(* CODESYS project CodesysTest
   Author: Ben Hess
   Company: Sharp Packaging
   CompiledLibraryCompatibilityVersion: CODESYS V3.5 SP16
   Version: 0.9.20.33
   VersionPostfix: -alpha/master

Project tree, tasks and I/O mapping:
  ElectricMachine : CODESYS Control RTE V3 x64, 3S - Smart Software Solutions GmbH, version 3.5.17.0
    application Application
    Customer_LAN_Adapter : Ethernet, 3S - Smart Software Solutions GmbH, version 3.5.16.0
        settings: IPAddress = [172,20,10,206]; SubnetMask = [255,255,255,0]; GatewayAddress = [172,20,10,1]; MACAddress = [16#D8,16#5E,16#D3,16#E1,16#78,16#F8]; NetworkInterfaceName = 'Customer LAN'; NetworkInterfaceName = "Customer LAN"; SaveCommunicationSettings = FALSE
      ModbusTCP_Slave_Device : ModbusTCP Slave Device, 3S - Smart Software Solutions GmbH, version 4.2.0.0
          input  Application.RemoteComms.modbusInputsToBagger.fillerTrigger : BOOL  // Holding Registers.Holding Registers.Bit0
          input  Application.RemoteComms.modbusInputsToBagger.baggerInhibit : BOOL  // Holding Registers.Holding Registers.Bit1
          input  Application.RemoteComms.modbusInputsToBagger.collisionDetection : BOOL  // Holding Registers.Holding Registers.Bit2
          input  Application.RemoteComms.modbusInputsToBagger.fillerOK : BOOL  // Holding Registers.Holding Registers.Bit3
          input  Application.RemoteComms.modbusInputsToBagger.reverseConveyor : BOOL  // Holding Registers.Holding Registers.Bit4
          input  Application.RemoteComms.modbusInputsToBagger.bagGrabbed : BOOL  // Holding Registers.Holding Registers.Bit5
          input  Application.RemoteComms.modbusInputsToBagger.heartbeat : BOOL  // Holding Registers.Holding Registers.Bit6
          output Application.RemoteComms.modbusOutputsFromBagger.baggerOK : BOOL  // Input Registers.Input Registers.Bit0
          output Application.RemoteComms.modbusOutputsFromBagger.readyForFiller : BOOL  // Input Registers.Input Registers.Bit1
          output Application.RemoteComms.modbusOutputsFromBagger.printerDataReady : BOOL  // Input Registers.Input Registers.Bit2
          output Application.RemoteComms.modbusOutputsFromBagger.waitingForPrinter : BOOL  // Input Registers.Input Registers.Bit3
          output Application.RemoteComms.modbusOutputsFromBagger.cycleComplete : BOOL  // Input Registers.Input Registers.Bit4
          output Application.RemoteComms.modbusOutputsFromBagger.bagMade : BOOL  // Input Registers.Input Registers.Bit5
          output Application.RemoteComms.modbusOutputsFromBagger.bagMadePlusLabelRequired : BOOL  // Input Registers.Input Registers.Bit6
          output Application.RemoteComms.modbusOutputsFromBagger.bagsLow : BOOL  // Input Registers.Input Registers.Bit7
          output Application.RemoteComms.modbusOutputsFromBagger.readyForGrab : BOOL  // Input Registers.Input Registers.Bit8
          output Application.RemoteComms.modbusOutputsFromBagger.runExternalExitConveyor : BOOL  // Input Registers.Input Registers.Bit9
          output Application.RemoteComms.modbusOutputsFromBagger.heartbeatResponse : BOOL  // Input Registers.Input Registers.Bit10
          unmapped channels: Holding Registers, Input Registers
    IO_Connection_Adapter : Ethernet, 3S - Smart Software Solutions GmbH, version 3.5.16.0
        settings: IPAddress = [192,168,10,21]; SubnetMask = [255,255,255,0]; GatewayAddress = [0,0,0,0]; MACAddress = [16#00,16#00,16#00,16#00,16#00,16#00]; NetworkInterfaceName = 'IO Connection'; NetworkInterfaceName = "IO Connection"; SaveCommunicationSettings = FALSE
      EtherNet_IP_Scanner : EtherNet/IP Scanner, 3S - Smart Software Solutions GmbH, order no. 1, version 3.5.16.10
    Machine_LAN_Adapter : Ethernet, 3S - Smart Software Solutions GmbH, version 3.5.16.0
        settings: IPAddress = [192,168,10,20]; SubnetMask = [255,255,255,0]; GatewayAddress = [192,168,10,254]; MACAddress = [16#00,16#00,16#00,16#00,16#00,16#00]; NetworkInterfaceName = 'Machine LAN'; NetworkInterfaceName = "Machine LAN"; SaveCommunicationSettings = FALSE
  Pro18_1174_CodesysDriver : CODESYS Control RTE V3 x64, 3S - Smart Software Solutions GmbH, version 3.5.17.0
    application Application
    Dual_LAN_Card : Ethernet, 3S - Smart Software Solutions GmbH, version 3.5.16.0
        settings: IPAddress = [192,168,10,21]; SubnetMask = [255,255,255,0]; GatewayAddress = [0,0,0,0]; MACAddress = [16#00,16#00,16#00,16#00,16#00,16#00]; NetworkInterfaceName = 'IO Connection'; NetworkInterfaceName = "IO Connection"; SaveCommunicationSettings = FALSE
      EtherNet_IP_Scanner : EtherNet/IP Scanner, 3S - Smart Software Solutions GmbH, order no. 1, version 3.5.16.10
    Ethernet : Ethernet, 3S - Smart Software Solutions GmbH, version 3.5.13.0
        settings: IPAddress = [192,168,10,20]; SubnetMask = [255,255,255,0]; GatewayAddress = [192,168,10,254]; NetworkInterfaceName = 'Machine LAN:2'; NetworkInterfaceName = "Machine LAN:2"; SaveCommunicationSettings = FALSE
      ModbusTCP_Slave_Device : ModbusTCP Slave Device, 3S - Smart Software Solutions GmbH, version 4.2.0.0 (disabled)
          input  Application.RemoteComms.modbusInputsToBagger.fillerTrigger : BOOL  // Holding Registers.Holding Registers.Bit0
          input  Application.RemoteComms.modbusInputsToBagger.baggerInhibit : BOOL  // Holding Registers.Holding Registers.Bit1
          input  Application.RemoteComms.modbusInputsToBagger.collisionDetection : BOOL  // Holding Registers.Holding Registers.Bit2
          input  Application.RemoteComms.modbusInputsToBagger.fillerOK : BOOL  // Holding Registers.Holding Registers.Bit3
          input  Application.RemoteComms.modbusInputsToBagger.reverseConveyor : BOOL  // Holding Registers.Holding Registers.Bit4
          input  Application.RemoteComms.modbusInputsToBagger.bagGrabbed : BOOL  // Holding Registers.Holding Registers.Bit5
          input  Application.RemoteComms.modbusInputsToBagger.heartbeat : BOOL  // Holding Registers.Holding Registers.Bit6
          output Application.RemoteComms.modbusOutputsFromBagger.baggerOK : BOOL  // Input Registers.Input Registers.Bit0
          output Application.RemoteComms.modbusOutputsFromBagger.readyForFiller : BOOL  // Input Registers.Input Registers.Bit1
          output Application.RemoteComms.modbusOutputsFromBagger.printerDataReady : BOOL  // Input Registers.Input Registers.Bit2
          output Application.RemoteComms.modbusOutputsFromBagger.waitingForPrinter : BOOL  // Input Registers.Input Registers.Bit3
          output Application.RemoteComms.modbusOutputsFromBagger.cycleComplete : BOOL  // Input Registers.Input Registers.Bit4
          output Application.RemoteComms.modbusOutputsFromBagger.bagMade : BOOL  // Input Registers.Input Registers.Bit5
          output Application.RemoteComms.modbusOutputsFromBagger.bagMadePlusLabelRequired : BOOL  // Input Registers.Input Registers.Bit6
          output Application.RemoteComms.modbusOutputsFromBagger.bagsLow : BOOL  // Input Registers.Input Registers.Bit7
          output Application.RemoteComms.modbusOutputsFromBagger.readyForGrab : BOOL  // Input Registers.Input Registers.Bit8
          output Application.RemoteComms.modbusOutputsFromBagger.runExternalExitConveyor : BOOL  // Input Registers.Input Registers.Bit9
          output Application.RemoteComms.modbusOutputsFromBagger.heartbeatResponse : BOOL  // Input Registers.Input Registers.Bit10
          unmapped channels: Holding Registers, Input Registers
  Pro18_1174_HilscherCard : Advantech Control x86 RTE V3, Advantech Co., Ltd., order no. 
      , version 3.5.13.0
    application Application
    CIFX_EIP : CIFX-EIP, 3S - Smart Software Solutions GmbH, order no. 1, version 3.5.12.0
        settings: IPAddress = [16#C0,16#A8,16#0A,16#15]; SubnetMask = [16#FF,16#FF,16#FF,16#00]; GatewayAddress = [16#00,16#00,16#00,16#00]; ConfigVersion = 50660608
      Bag_Delivery_EIP_Motor : TSM34IP, Applied Motion Products, Inc, order no. TSM34IP, version Major Revision=16#3, Minor Revision = 16#3
          settings: INITIALIZED = TRUE; IP address of Target = [16#C0,16#A8,16#0A,16#37]; Keying.Check Vendor Code = FALSE; Keying.Check Product Code = FALSE; Keying.Check Major Revision = FALSE; Keying.Check Minor Revision = FALSE; RequiredConfigVersion = 50660864; Number of Connections = 1; Connection Settings.Requested packet intervall = 10000 µs; Connection Settings.OT Connection Parameters = 18502; Connection Settings.TO Connection Parameters = 18490; Connection Settings.Connection Flags = 1056; Connection Settings.Connection Path Size = 8; Connection Settings.Large OT Connection Parameters = 1207959622; Connection Settings.Large TO Connection Parameters = 1207959610; Heartbeat Multiplier = 1; Status Code.ReadOnly = False; Status Code.BitSize = 32; Status Code.DataSize = 4; Alarm Code.ReadOnly = False; Alarm Code.BitSize = 32; Alarm Code.DataSize = 4; Supply Voltage.ReadOnly = False; Supply Voltage.BitSize = 32; Supply Voltage.DataSize = 4; Actual Current.ReadOnly = False; Actual Current.BitSize = 32; Actual Current.DataSize = 4; Drive Temperature.ReadOnly = False; Drive Temperature.BitSize = 32; Drive Temperature.DataSize = 4; Encoder Position.ReadOnly = False; Encoder Position.BitSize = 32; Encoder Position.DataSize = 4; Absolute Position.ReadOnly = False; Absolute Position.BitSize = 32; Absolute Position.DataSize = 4; Position Error.ReadOnly = False; Position Error.BitSize = 32; Position Error.DataSize = 4;
            Actual Velocity.ReadOnly = False; Actual Velocity.BitSize = 32; Actual Velocity.DataSize = 4; Input Status (extended).ReadOnly = False; Input Status (extended).BitSize = 32; Input Status (extended).DataSize = 4; Input Status (main).ReadOnly = False; Input Status (main).BitSize = 32; Input Status (main).DataSize = 4; Output Status.ReadOnly = False; Output Status.BitSize = 32; Output Status.DataSize = 4; Analog Input 1.ReadOnly = False; Analog Input 1.BitSize = 32; Analog Input 1.DataSize = 4; Analog Input 2.ReadOnly = False; Analog Input 2.BitSize = 32; Analog Input 2.DataSize = 4; Command Word.ReadOnly = False; Command Word.BitSize = 32; Command Word.DataSize = 4; Jog Speed.ReadOnly = False; Jog Speed.BitSize = 32; Jog Speed.DataSize = 4; Jog Accel.ReadOnly = False; Jog Accel.BitSize = 32; Jog Accel.DataSize = 4; Jog Decel.ReadOnly = False; Jog Decel.BitSize = 32; Jog Decel.DataSize = 4; Point-to-Point Velocity.ReadOnly = False; Point-to-Point Velocity.BitSize = 32; Point-to-Point Velocity.DataSize = 4; Point-to-Point Acceleration.ReadOnly = False; Point-to-Point Acceleration.BitSize = 32; Point-to-Point Acceleration.DataSize = 4; Point-to-Point Deceleration.ReadOnly = False; Point-to-Point Deceleration.BitSize = 32; Point-to-Point Deceleration.DataSize = 4; Point-to-Point Distance.ReadOnly = False;
            Point-to-Point Distance.BitSize = 32; Point-to-Point Distance.DataSize = 4; Current Command.ReadOnly = False; Current Command.BitSize = 32; Current Command.DataSize = 4; SCL Command Letters.ReadOnly = False; SCL Command Letters.BitSize = 32; SCL Command Letters.DataSize = 4; Data/SCL Register 1.ReadOnly = False; Data/SCL Register 1.BitSize = 32; Data/SCL Register 1.DataSize = 4; Data/SCL Register 2.ReadOnly = False; Data/SCL Register 2.BitSize = 32; Data/SCL Register 2.DataSize = 4; Reserved 1.ReadOnly = False; Reserved 1.BitSize = 32; Reserved 1.DataSize = 4; Reserved 2.ReadOnly = False; Reserved 2.BitSize = 32; Reserved 2.DataSize = 4; Reserved 3.ReadOnly = False; Reserved 3.BitSize = 32; Reserved 3.DataSize = 4; Reserved 4.ReadOnly = False; Reserved 4.BitSize = 32; Reserved 4.DataSize = 4; Status Code.Name = 'Status Code'; Status Code.HelpString = ''; Status Code.ReadOnly = False; Status Code.BitSize = 32; Status Code.DataSize = 4; Status Code.DataType = 'DINT'; Alarm Code.Name = 'Alarm Code'; Alarm Code.HelpString = ''; Alarm Code.ReadOnly = False; Alarm Code.BitSize = 32; Alarm Code.DataSize = 4; Alarm Code.DataType = 'DINT'; Supply Voltage.Name = 'Supply Voltage'; Supply Voltage.HelpString = '';
            Supply Voltage.ReadOnly = False; Supply Voltage.BitSize = 32; Supply Voltage.DataSize = 4; Supply Voltage.DataType = 'DINT'; Actual Current.Name = 'Actual Current'; Actual Current.HelpString = ''; Actual Current.ReadOnly = False; Actual Current.BitSize = 32; Actual Current.DataSize = 4; Actual Current.DataType = 'DINT'; Drive Temperature.Name = 'Drive Temperature'; Drive Temperature.HelpString = ''; Drive Temperature.ReadOnly = False; Drive Temperature.BitSize = 32; Drive Temperature.DataSize = 4; Drive Temperature.DataType = 'DINT'; Encoder Position.Name = 'Encoder Position'; Encoder Position.HelpString = ''; Encoder Position.ReadOnly = False; Encoder Position.BitSize = 32; Encoder Position.DataSize = 4; Encoder Position.DataType = 'DINT'; Absolute Position.Name = 'Absolute Position'; Absolute Position.HelpString = ''; Absolute Position.ReadOnly = False; Absolute Position.BitSize = 32; Absolute Position.DataSize = 4; Absolute Position.DataType = 'DINT'; Position Error.Name = 'Position Error'; Position Error.HelpString = ''; Position Error.ReadOnly = False; Position Error.BitSize = 32; Position Error.DataSize = 4; Position Error.DataType = 'DINT'; Actual Velocity.Name = 'Actual Velocity'; Actual Velocity.HelpString = ''; Actual Velocity.ReadOnly = False; Actual Velocity.BitSize = 32; Actual Velocity.DataSize = 4; Actual Velocity.DataType = 'DINT';
            Input Status (extended).Name = 'Input Status (extended)'; Input Status (extended).HelpString = ''; Input Status (extended).ReadOnly = False; Input Status (extended).BitSize = 32; Input Status (extended).DataSize = 4; Input Status (extended).DataType = 'DINT'; Input Status (main).Name = 'Input Status (main)'; Input Status (main).HelpString = ''; Input Status (main).ReadOnly = False; Input Status (main).BitSize = 32; Input Status (main).DataSize = 4; Input Status (main).DataType = 'DINT'; Output Status.Name = 'Output Status'; Output Status.HelpString = ''; Output Status.ReadOnly = False; Output Status.BitSize = 32; Output Status.DataSize = 4; Output Status.DataType = 'DINT'; Analog Input 1.Name = 'Analog Input 1'; Analog Input 1.HelpString = ''; Analog Input 1.ReadOnly = False; Analog Input 1.BitSize = 32; Analog Input 1.DataSize = 4; Analog Input 1.DataType = 'DINT'; Analog Input 2.Name = 'Analog Input 2'; Analog Input 2.HelpString = ''; Analog Input 2.ReadOnly = False; Analog Input 2.BitSize = 32; Analog Input 2.DataSize = 4; Analog Input 2.DataType = 'DINT'; Command Word.Name = 'Command Word'; Command Word.HelpString = ''; Command Word.ReadOnly = False; Command Word.BitSize = 32; Command Word.DataSize = 4; Command Word.DataType = 'DINT'; Jog Speed.Name = 'Jog Speed'; Jog Speed.HelpString = ''; Jog Speed.ReadOnly = False; Jog Speed.BitSize = 32;
            Jog Speed.DataSize = 4; Jog Speed.DataType = 'DINT'; Jog Accel.Name = 'Jog Accel'; Jog Accel.HelpString = ''; Jog Accel.ReadOnly = False; Jog Accel.BitSize = 32; Jog Accel.DataSize = 4; Jog Accel.DataType = 'DINT'; Jog Decel.Name = 'Jog Decel'; Jog Decel.HelpString = ''; Jog Decel.ReadOnly = False; Jog Decel.BitSize = 32; Jog Decel.DataSize = 4; Jog Decel.DataType = 'DINT'; Point-to-Point Velocity.Name = 'Point-to-Point Velocity'; Point-to-Point Velocity.HelpString = ''; Point-to-Point Velocity.ReadOnly = False; Point-to-Point Velocity.BitSize = 32; Point-to-Point Velocity.DataSize = 4; Point-to-Point Velocity.DataType = 'DINT'; Point-to-Point Acceleration.Name = 'Point-to-Point Acceleration'; Point-to-Point Acceleration.HelpString = ''; Point-to-Point Acceleration.ReadOnly = False; Point-to-Point Acceleration.BitSize = 32; Point-to-Point Acceleration.DataSize = 4; Point-to-Point Acceleration.DataType = 'DINT'; Point-to-Point Deceleration.Name = 'Point-to-Point Deceleration'; Point-to-Point Deceleration.HelpString = ''; Point-to-Point Deceleration.ReadOnly = False; Point-to-Point Deceleration.BitSize = 32; Point-to-Point Deceleration.DataSize = 4; Point-to-Point Deceleration.DataType = 'DINT'; Point-to-Point Distance.Name = 'Point-to-Point Distance'; Point-to-Point Distance.HelpString = ''; Point-to-Point Distance.ReadOnly = False; Point-to-Point Distance.BitSize = 32; Point-to-Point Distance.DataSize = 4; Point-to-Point Distance.DataType = 'DINT'; Current Command.Name = 'Current Command'; Current Command.HelpString = '';
            Current Command.ReadOnly = False; Current Command.BitSize = 32; Current Command.DataSize = 4; Current Command.DataType = 'DINT'; SCL Command Letters.Name = 'SCL Command Letters'; SCL Command Letters.HelpString = ''; SCL Command Letters.ReadOnly = False; SCL Command Letters.BitSize = 32; SCL Command Letters.DataSize = 4; SCL Command Letters.DataType = 'DINT'; Data/SCL Register 1.Name = 'Data/SCL Register 1'; Data/SCL Register 1.HelpString = ''; Data/SCL Register 1.ReadOnly = False; Data/SCL Register 1.BitSize = 32; Data/SCL Register 1.DataSize = 4; Data/SCL Register 1.DataType = 'DINT'; Data/SCL Register 2.Name = 'Data/SCL Register 2'; Data/SCL Register 2.HelpString = ''; Data/SCL Register 2.ReadOnly = False; Data/SCL Register 2.BitSize = 32; Data/SCL Register 2.DataSize = 4; Data/SCL Register 2.DataType = 'DINT'; Reserved 1.Name = 'Reserved 1'; Reserved 1.HelpString = ''; Reserved 1.ReadOnly = False; Reserved 1.BitSize = 32; Reserved 1.DataSize = 4; Reserved 1.DataType = 'DINT'; Reserved 2.Name = 'Reserved 2'; Reserved 2.HelpString = ''; Reserved 2.ReadOnly = False; Reserved 2.BitSize = 32; Reserved 2.DataSize = 4; Reserved 2.DataType = 'DINT'; Reserved 3.Name = 'Reserved 3'; Reserved 3.HelpString = ''; Reserved 3.ReadOnly = False; Reserved 3.BitSize = 32; Reserved 3.DataSize = 4; Reserved 3.DataType = 'DINT';
            Reserved 4.Name = 'Reserved 4'; Reserved 4.HelpString = ''; Reserved 4.ReadOnly = False; Reserved 4.BitSize = 32; Reserved 4.DataSize = 4; Reserved 4.DataType = 'DINT'; ConfigVersion = 50660864
          input  bagDeliveryMotorInputs : DINT  // Status Code
          input  iBagNotPresent : BOOL  // Input Status (main).Bit2
          output bagDeliveryMotorOutputs : DINT  // Command Word
          unmapped channels: Alarm Code, Supply Voltage, Actual Current, Drive Temperature, Encoder Position, Absolute Position, Position Error, Actual Velocity, Input Status (extended), Input Status (main), Output Status, Analog Input 1, Analog Input 2, Jog Speed, Jog Accel, Jog Decel, Point-to-Point Velocity, Point-to-Point Acceleration, Point-to-Point Deceleration, Point-to-Point Distance, Current Command, SCL Command Letters, Data/SCL Register 1, Data/SCL Register 2, Reserved 1, Reserved 2, Reserved 3, Reserved 4
      Bag_Delivery_Rear_Motor : TSM34IP, Applied Motion Products, Inc, order no. TSM34IP, version Major Revision=16#3, Minor Revision = 16#3
          settings: INITIALIZED = TRUE; IP address of Target = [16#C0,16#A8,16#0A,16#38]; MAC address of Target = [16#00,16#00,16#00,16#00,16#00,16#00]; Keying.Check Device Type = FALSE; Keying.Check Vendor Code = FALSE; Keying.Check Product Code = FALSE; Keying.Check Major Revision = FALSE; Keying.Check Minor Revision = FALSE; RequiredConfigVersion = 50660864; Number of Connections = 1; Connection Settings.Requested packet intervall = 10000 µs; Connection Settings.OT Connection Parameters = 18502; Connection Settings.TO Connection Parameters = 18490; Connection Settings.Connection Flags = 1056; Connection Settings.Connection Path Size = 8; Status Code.ReadOnly = False; Status Code.BitSize = 32; Status Code.DataSize = 4; Alarm Code.ReadOnly = False; Alarm Code.BitSize = 32; Alarm Code.DataSize = 4; Supply Voltage.ReadOnly = False; Supply Voltage.BitSize = 32; Supply Voltage.DataSize = 4; Actual Current.ReadOnly = False; Actual Current.BitSize = 32; Actual Current.DataSize = 4; Drive Temperature.ReadOnly = False; Drive Temperature.BitSize = 32; Drive Temperature.DataSize = 4; Encoder Position.ReadOnly = False; Encoder Position.BitSize = 32; Encoder Position.DataSize = 4; Absolute Position.ReadOnly = False; Absolute Position.BitSize = 32; Absolute Position.DataSize = 4; Position Error.ReadOnly = False; Position Error.BitSize = 32; Position Error.DataSize = 4; Actual Velocity.ReadOnly = False;
            Actual Velocity.BitSize = 32; Actual Velocity.DataSize = 4; Input Status (extended).ReadOnly = False; Input Status (extended).BitSize = 32; Input Status (extended).DataSize = 4; Input Status (main).ReadOnly = False; Input Status (main).BitSize = 32; Input Status (main).DataSize = 4; Output Status.ReadOnly = False; Output Status.BitSize = 32; Output Status.DataSize = 4; Analog Input 1.ReadOnly = False; Analog Input 1.BitSize = 32; Analog Input 1.DataSize = 4; Analog Input 2.ReadOnly = False; Analog Input 2.BitSize = 32; Analog Input 2.DataSize = 4; Command Word.ReadOnly = False; Command Word.BitSize = 32; Command Word.DataSize = 4; Jog Speed.ReadOnly = False; Jog Speed.BitSize = 32; Jog Speed.DataSize = 4; Jog Accel.ReadOnly = False; Jog Accel.BitSize = 32; Jog Accel.DataSize = 4; Jog Decel.ReadOnly = False; Jog Decel.BitSize = 32; Jog Decel.DataSize = 4; Point-to-Point Velocity.ReadOnly = False; Point-to-Point Velocity.BitSize = 32; Point-to-Point Velocity.DataSize = 4; Point-to-Point Acceleration.ReadOnly = False; Point-to-Point Acceleration.BitSize = 32; Point-to-Point Acceleration.DataSize = 4; Point-to-Point Deceleration.ReadOnly = False; Point-to-Point Deceleration.BitSize = 32; Point-to-Point Deceleration.DataSize = 4; Point-to-Point Distance.ReadOnly = False; Point-to-Point Distance.BitSize = 32;
            Point-to-Point Distance.DataSize = 4; Current Command.ReadOnly = False; Current Command.BitSize = 32; Current Command.DataSize = 4; SCL Command Letters.ReadOnly = False; SCL Command Letters.BitSize = 32; SCL Command Letters.DataSize = 4; Data/SCL Register 1.ReadOnly = False; Data/SCL Register 1.BitSize = 32; Data/SCL Register 1.DataSize = 4; Data/SCL Register 2.ReadOnly = False; Data/SCL Register 2.BitSize = 32; Data/SCL Register 2.DataSize = 4; Reserved 1.ReadOnly = False; Reserved 1.BitSize = 32; Reserved 1.DataSize = 4; Reserved 2.ReadOnly = False; Reserved 2.BitSize = 32; Reserved 2.DataSize = 4; Reserved 3.ReadOnly = False; Reserved 3.BitSize = 32; Reserved 3.DataSize = 4; Reserved 4.ReadOnly = False; Reserved 4.BitSize = 32; Reserved 4.DataSize = 4; Status Code.Name = 'Status Code'; Status Code.HelpString = ''; Status Code.ReadOnly = False; Status Code.BitSize = 32; Status Code.DataSize = 4; Status Code.DataType = 'DINT'; Alarm Code.Name = 'Alarm Code'; Alarm Code.HelpString = ''; Alarm Code.ReadOnly = False; Alarm Code.BitSize = 32; Alarm Code.DataSize = 4; Alarm Code.DataType = 'DINT'; Supply Voltage.Name = 'Supply Voltage'; Supply Voltage.HelpString = ''; Supply Voltage.ReadOnly = False;
            Supply Voltage.BitSize = 32; Supply Voltage.DataSize = 4; Supply Voltage.DataType = 'DINT'; Actual Current.Name = 'Actual Current'; Actual Current.HelpString = ''; Actual Current.ReadOnly = False; Actual Current.BitSize = 32; Actual Current.DataSize = 4; Actual Current.DataType = 'DINT'; Drive Temperature.Name = 'Drive Temperature'; Drive Temperature.HelpString = ''; Drive Temperature.ReadOnly = False; Drive Temperature.BitSize = 32; Drive Temperature.DataSize = 4; Drive Temperature.DataType = 'DINT'; Encoder Position.Name = 'Encoder Position'; Encoder Position.HelpString = ''; Encoder Position.ReadOnly = False; Encoder Position.BitSize = 32; Encoder Position.DataSize = 4; Encoder Position.DataType = 'DINT'; Absolute Position.Name = 'Absolute Position'; Absolute Position.HelpString = ''; Absolute Position.ReadOnly = False; Absolute Position.BitSize = 32; Absolute Position.DataSize = 4; Absolute Position.DataType = 'DINT'; Position Error.Name = 'Position Error'; Position Error.HelpString = ''; Position Error.ReadOnly = False; Position Error.BitSize = 32; Position Error.DataSize = 4; Position Error.DataType = 'DINT'; Actual Velocity.Name = 'Actual Velocity'; Actual Velocity.HelpString = ''; Actual Velocity.ReadOnly = False; Actual Velocity.BitSize = 32; Actual Velocity.DataSize = 4; Actual Velocity.DataType = 'DINT'; Input Status (extended).Name = 'Input Status (extended)';
            Input Status (extended).HelpString = ''; Input Status (extended).ReadOnly = False; Input Status (extended).BitSize = 32; Input Status (extended).DataSize = 4; Input Status (extended).DataType = 'DINT'; Input Status (main).Name = 'Input Status (main)'; Input Status (main).HelpString = ''; Input Status (main).ReadOnly = False; Input Status (main).BitSize = 32; Input Status (main).DataSize = 4; Input Status (main).DataType = 'DINT'; Output Status.Name = 'Output Status'; Output Status.HelpString = ''; Output Status.ReadOnly = False; Output Status.BitSize = 32; Output Status.DataSize = 4; Output Status.DataType = 'DINT'; Analog Input 1.Name = 'Analog Input 1'; Analog Input 1.HelpString = ''; Analog Input 1.ReadOnly = False; Analog Input 1.BitSize = 32; Analog Input 1.DataSize = 4; Analog Input 1.DataType = 'DINT'; Analog Input 2.Name = 'Analog Input 2'; Analog Input 2.HelpString = ''; Analog Input 2.ReadOnly = False; Analog Input 2.BitSize = 32; Analog Input 2.DataSize = 4; Analog Input 2.DataType = 'DINT'; Command Word.Name = 'Command Word'; Command Word.HelpString = ''; Command Word.ReadOnly = False; Command Word.BitSize = 32; Command Word.DataSize = 4; Command Word.DataType = 'DINT'; Jog Speed.Name = 'Jog Speed'; Jog Speed.HelpString = ''; Jog Speed.ReadOnly = False; Jog Speed.BitSize = 32; Jog Speed.DataSize = 4;
            Jog Speed.DataType = 'DINT'; Jog Accel.Name = 'Jog Accel'; Jog Accel.HelpString = ''; Jog Accel.ReadOnly = False; Jog Accel.BitSize = 32; Jog Accel.DataSize = 4; Jog Accel.DataType = 'DINT'; Jog Decel.Name = 'Jog Decel'; Jog Decel.HelpString = ''; Jog Decel.ReadOnly = False; Jog Decel.BitSize = 32; Jog Decel.DataSize = 4; Jog Decel.DataType = 'DINT'; Point-to-Point Velocity.Name = 'Point-to-Point Velocity'; Point-to-Point Velocity.HelpString = ''; Point-to-Point Velocity.ReadOnly = False; Point-to-Point Velocity.BitSize = 32; Point-to-Point Velocity.DataSize = 4; Point-to-Point Velocity.DataType = 'DINT'; Point-to-Point Acceleration.Name = 'Point-to-Point Acceleration'; Point-to-Point Acceleration.HelpString = ''; Point-to-Point Acceleration.ReadOnly = False; Point-to-Point Acceleration.BitSize = 32; Point-to-Point Acceleration.DataSize = 4; Point-to-Point Acceleration.DataType = 'DINT'; Point-to-Point Deceleration.Name = 'Point-to-Point Deceleration'; Point-to-Point Deceleration.HelpString = ''; Point-to-Point Deceleration.ReadOnly = False; Point-to-Point Deceleration.BitSize = 32; Point-to-Point Deceleration.DataSize = 4; Point-to-Point Deceleration.DataType = 'DINT'; Point-to-Point Distance.Name = 'Point-to-Point Distance'; Point-to-Point Distance.HelpString = ''; Point-to-Point Distance.ReadOnly = False; Point-to-Point Distance.BitSize = 32; Point-to-Point Distance.DataSize = 4; Point-to-Point Distance.DataType = 'DINT'; Current Command.Name = 'Current Command'; Current Command.HelpString = ''; Current Command.ReadOnly = False;
            Current Command.BitSize = 32; Current Command.DataSize = 4; Current Command.DataType = 'DINT'; SCL Command Letters.Name = 'SCL Command Letters'; SCL Command Letters.HelpString = ''; SCL Command Letters.ReadOnly = False; SCL Command Letters.BitSize = 32; SCL Command Letters.DataSize = 4; SCL Command Letters.DataType = 'DINT'; Data/SCL Register 1.Name = 'Data/SCL Register 1'; Data/SCL Register 1.HelpString = ''; Data/SCL Register 1.ReadOnly = False; Data/SCL Register 1.BitSize = 32; Data/SCL Register 1.DataSize = 4; Data/SCL Register 1.DataType = 'DINT'; Data/SCL Register 2.Name = 'Data/SCL Register 2'; Data/SCL Register 2.HelpString = ''; Data/SCL Register 2.ReadOnly = False; Data/SCL Register 2.BitSize = 32; Data/SCL Register 2.DataSize = 4; Data/SCL Register 2.DataType = 'DINT'; Reserved 1.Name = 'Reserved 1'; Reserved 1.HelpString = ''; Reserved 1.ReadOnly = False; Reserved 1.BitSize = 32; Reserved 1.DataSize = 4; Reserved 1.DataType = 'DINT'; Reserved 2.Name = 'Reserved 2'; Reserved 2.HelpString = ''; Reserved 2.ReadOnly = False; Reserved 2.BitSize = 32; Reserved 2.DataSize = 4; Reserved 2.DataType = 'DINT'; Reserved 3.Name = 'Reserved 3'; Reserved 3.HelpString = ''; Reserved 3.ReadOnly = False; Reserved 3.BitSize = 32; Reserved 3.DataSize = 4; Reserved 3.DataType = 'DINT'; Reserved 4.Name = 'Reserved 4';
            Reserved 4.HelpString = ''; Reserved 4.ReadOnly = False; Reserved 4.BitSize = 32; Reserved 4.DataSize = 4; Reserved 4.DataType = 'DINT'; ConfigVersion = 50660864
          input  bagRearMotorInputs AT %ID200 : DINT  // Status Code
          input  iBagTensionFault : BOOL  // Output Status.Bit3
          output bagRearMotorOutputs AT %QD200 : DINT  // Command Word
          unmapped channels: Alarm Code, Supply Voltage, Actual Current, Drive Temperature, Encoder Position, Absolute Position, Position Error, Actual Velocity, Input Status (extended), Input Status (main), Output Status, Analog Input 1, Analog Input 2, Jog Speed, Jog Accel, Jog Decel, Point-to-Point Velocity, Point-to-Point Acceleration, Point-to-Point Deceleration, Point-to-Point Distance, Current Command, SCL Command Letters, Data/SCL Register 1, Data/SCL Register 2, Reserved 1, Reserved 2, Reserved 3, Reserved 4
      DM374_BCV : DataMan 300 Series Reader, Cognex, order no. DMR-3XX-00, version Major Revision=16#1, Minor Revision = 16#5 (disabled)
          settings: INITIALIZED = TRUE; IP address of Target = [16#C0,16#A8,16#0A,16#A3]; Keying.Check Minor Revision = FALSE; RequiredConfigVersion = 50660864; Number of Connections = 1; Connection Settings.Requested packet intervall = 10000 µs; Connection Settings.OT Connection Parameters = 18448; Connection Settings.TO Connection Parameters = 18558; Connection Settings.Connection Flags = 1056; Connection Settings.Connection Path Size = 8; Heartbeat Multiplier = 1; output_param.Name = 'output_param'; output_param.HelpString = ''; output_param.ReadOnly = False; output_param.BitSize = 8; output_param.DataSize = 1; output_param.DataType = 'BYTE'; output_param.ReadOnly = False; output_param.BitSize = 8; output_param.DataSize = 1; input_param.ReadOnly = False; input_param.BitSize = 8; input_param.DataSize = 1; input_param.ReadOnly = False; input_param.BitSize = 8; input_param.DataSize = 1; input_param.ReadOnly = False; input_param.BitSize = 8; input_param.DataSize = 1; input_param.ReadOnly = False; input_param.BitSize = 8; input_param.DataSize = 1; input_param.ReadOnly = False; input_param.BitSize = 8; input_param.DataSize = 1; input_param.ReadOnly = False; input_param.BitSize = 8; input_param.DataSize = 1; input_param.ReadOnly = False; input_param.BitSize = 8;
            input_param.DataSize = 1; input_param.ReadOnly = False; input_param.BitSize = 8; input_param.DataSize = 1; input_param.ReadOnly = False; input_param.BitSize = 8; input_param.DataSize = 1; input_param.ReadOnly = False; input_param.BitSize = 8; input_param.DataSize = 1; input_param.ReadOnly = False; input_param.BitSize = 8; input_param.DataSize = 1; input_param.ReadOnly = False; input_param.BitSize = 8; input_param.DataSize = 1; input_param.ReadOnly = False; input_param.BitSize = 8; input_param.DataSize = 1; input_param.ReadOnly = False; input_param.BitSize = 8; input_param.DataSize = 1; input_param.ReadOnly = False; input_param.BitSize = 8; input_param.DataSize = 1; input_param.ReadOnly = False; input_param.BitSize = 8; input_param.DataSize = 1; input_param.ReadOnly = False; input_param.BitSize = 8; input_param.DataSize = 1; input_param.ReadOnly = False; input_param.BitSize = 8; input_param.DataSize = 1; input_param.ReadOnly = False; input_param.BitSize = 8; input_param.DataSize = 1; input_param.ReadOnly = False; input_param.BitSize = 8; input_param.DataSize = 1;
            input_param.ReadOnly = False; input_param.BitSize = 8; input_param.DataSize = 1; input_param.ReadOnly = False; input_param.BitSize = 8; input_param.DataSize = 1; input_param.ReadOnly = False; input_param.BitSize = 8; input_param.DataSize = 1; input_param.ReadOnly = False; input_param.BitSize = 8; input_param.DataSize = 1; input_param.ReadOnly = False; input_param.BitSize = 8; input_param.DataSize = 1; input_param.ReadOnly = False; input_param.BitSize = 8; input_param.DataSize = 1; input_param.ReadOnly = False; input_param.BitSize = 8; input_param.DataSize = 1; input_param.ReadOnly = False; input_param.BitSize = 8; input_param.DataSize = 1; input_param.ReadOnly = False; input_param.BitSize = 8; input_param.DataSize = 1; input_param.ReadOnly = False; input_param.BitSize = 8; input_param.DataSize = 1; input_param.ReadOnly = False; input_param.BitSize = 8; input_param.DataSize = 1; input_param.ReadOnly = False; input_param.BitSize = 8; input_param.DataSize = 1; input_param.ReadOnly = False; input_param.BitSize = 8; input_param.DataSize = 1; input_param.ReadOnly = False;
            input_param.BitSize = 8; input_param.DataSize = 1; input_param.ReadOnly = False; input_param.BitSize = 8; input_param.DataSize = 1; input_param.ReadOnly = False; input_param.BitSize = 8; input_param.DataSize = 1; input_param.ReadOnly = False; input_param.BitSize = 8; input_param.DataSize = 1; input_param.ReadOnly = False; input_param.BitSize = 8; input_param.DataSize = 1; input_param.ReadOnly = False; input_param.BitSize = 8; input_param.DataSize = 1; input_param.ReadOnly = False; input_param.BitSize = 8; input_param.DataSize = 1; input_param.ReadOnly = False; input_param.BitSize = 8; input_param.DataSize = 1; input_param.ReadOnly = False; input_param.BitSize = 8; input_param.DataSize = 1; input_param.ReadOnly = False; input_param.BitSize = 8; input_param.DataSize = 1; input_param.ReadOnly = False; input_param.BitSize = 8; input_param.DataSize = 1; input_param.ReadOnly = False; input_param.BitSize = 8; input_param.DataSize = 1; input_param.ReadOnly = False; input_param.BitSize = 8; input_param.DataSize = 1; input_param.ReadOnly = False; input_param.BitSize = 8;
            input_param.DataSize = 1; input_param.ReadOnly = False; input_param.BitSize = 8; input_param.DataSize = 1; input_param.ReadOnly = False; input_param.BitSize = 8; input_param.DataSize = 1; input_param.ReadOnly = False; input_param.BitSize = 8; input_param.DataSize = 1; input_param.ReadOnly = False; input_param.BitSize = 8; input_param.DataSize = 1; input_param.ReadOnly = False; input_param.BitSize = 8; input_param.DataSize = 1; input_param.ReadOnly = False; input_param.BitSize = 8; input_param.DataSize = 1; input_param.ReadOnly = False; input_param.BitSize = 8; input_param.DataSize = 1; input_param.ReadOnly = False; input_param.BitSize = 8; input_param.DataSize = 1; input_param.ReadOnly = False; input_param.BitSize = 8; input_param.DataSize = 1; input_param.ReadOnly = False; input_param.BitSize = 8; input_param.DataSize = 1; input_param.ReadOnly = False; input_param.BitSize = 8; input_param.DataSize = 1; input_param.ReadOnly = False; input_param.BitSize = 8; input_param.DataSize = 1; input_param.ReadOnly = False; input_param.BitSize = 8; input_param.DataSize = 1;
            input_param.ReadOnly = False; input_param.BitSize = 8; input_param.DataSize = 1; input_param.ReadOnly = False; input_param.BitSize = 8; input_param.DataSize = 1; input_param.ReadOnly = False; input_param.BitSize = 8; input_param.DataSize = 1; input_param.ReadOnly = False; input_param.BitSize = 8; input_param.DataSize = 1; input_param.ReadOnly = False; input_param.BitSize = 8; input_param.DataSize = 1; input_param.ReadOnly = False; input_param.BitSize = 8; input_param.DataSize = 1; input_param.ReadOnly = False; input_param.BitSize = 8; input_param.DataSize = 1; input_param.ReadOnly = False; input_param.BitSize = 8; input_param.DataSize = 1; input_param.ReadOnly = False; input_param.BitSize = 8; input_param.DataSize = 1; input_param.ReadOnly = False; input_param.BitSize = 8; input_param.DataSize = 1; input_param.ReadOnly = False; input_param.BitSize = 8; input_param.DataSize = 1; input_param.ReadOnly = False; input_param.BitSize = 8; input_param.DataSize = 1; input_param.ReadOnly = False; input_param.BitSize = 8; input_param.DataSize = 1; input_param.ReadOnly = False;
            input_param.BitSize = 8; input_param.DataSize = 1; input_param.ReadOnly = False; input_param.BitSize = 8; input_param.DataSize = 1; input_param.ReadOnly = False; input_param.BitSize = 8; input_param.DataSize = 1; input_param.ReadOnly = False; input_param.BitSize = 8; input_param.DataSize = 1; input_param.ReadOnly = False; input_param.BitSize = 8; input_param.DataSize = 1; input_param.ReadOnly = False; input_param.BitSize = 8; input_param.DataSize = 1; input_param.ReadOnly = False; input_param.BitSize = 8; input_param.DataSize = 1; input_param.ReadOnly = False; input_param.BitSize = 8; input_param.DataSize = 1; input_param.ReadOnly = False; input_param.BitSize = 8; input_param.DataSize = 1; input_param.ReadOnly = False; input_param.BitSize = 8; input_param.DataSize = 1; input_param.ReadOnly = False; input_param.BitSize = 8; input_param.DataSize = 1; input_param.ReadOnly = False; input_param.BitSize = 8; input_param.DataSize = 1; input_param.ReadOnly = False; input_param.BitSize = 8; input_param.DataSize = 1; input_param.ReadOnly = False; input_param.BitSize = 8;
            input_param.DataSize = 1; input_param.ReadOnly = False; input_param.BitSize = 8; input_param.DataSize = 1; input_param.ReadOnly = False; input_param.BitSize = 8; input_param.DataSize = 1; input_param.ReadOnly = False; input_param.BitSize = 8; input_param.DataSize = 1; input_param.ReadOnly = False; input_param.BitSize = 8; input_param.DataSize = 1; input_param.ReadOnly = False; input_param.BitSize = 8; input_param.DataSize = 1; input_param.ReadOnly = False; input_param.BitSize = 8; input_param.DataSize = 1; input_param.ReadOnly = False; input_param.BitSize = 8; input_param.DataSize = 1; input_param.ReadOnly = False; input_param.BitSize = 8; input_param.DataSize = 1; input_param.ReadOnly = False; input_param.BitSize = 8; input_param.DataSize = 1; input_param.ReadOnly = False; input_param.BitSize = 8; input_param.DataSize = 1; input_param.ReadOnly = False; input_param.BitSize = 8; input_param.DataSize = 1; input_param.ReadOnly = False; input_param.BitSize = 8; input_param.DataSize = 1; input_param.ReadOnly = False; input_param.BitSize = 8; input_param.DataSize = 1;
            input_param.ReadOnly = False; input_param.BitSize = 8; input_param.DataSize = 1; input_param.ReadOnly = False; input_param.BitSize = 8; input_param.DataSize = 1; input_param.ReadOnly = False; input_param.BitSize = 8; input_param.DataSize = 1; input_param.ReadOnly = False; input_param.BitSize = 8; input_param.DataSize = 1; input_param.ReadOnly = False; input_param.BitSize = 8; input_param.DataSize = 1; input_param.ReadOnly = False; input_param.BitSize = 8; input_param.DataSize = 1; input_param.ReadOnly = False; input_param.BitSize = 8; input_param.DataSize = 1; input_param.ReadOnly = False; input_param.BitSize = 8; input_param.DataSize = 1; input_param.ReadOnly = False; input_param.BitSize = 8; input_param.DataSize = 1; input_param.ReadOnly = False; input_param.BitSize = 8; input_param.DataSize = 1; input_param.ReadOnly = False; input_param.BitSize = 8; input_param.DataSize = 1; input_param.ReadOnly = False; input_param.BitSize = 8; input_param.DataSize = 1; input_param.ReadOnly = False; input_param.BitSize = 8; input_param.DataSize = 1; input_param.ReadOnly = False;
            input_param.BitSize = 8; input_param.DataSize = 1; input_param.ReadOnly = False; input_param.BitSize = 8; input_param.DataSize = 1; input_param.ReadOnly = False; input_param.BitSize = 8; input_param.DataSize = 1; input_param.ReadOnly = False; input_param.BitSize = 8; input_param.DataSize = 1; input_param.ReadOnly = False; input_param.BitSize = 8; input_param.DataSize = 1; input_param.ReadOnly = False; input_param.BitSize = 8; input_param.DataSize = 1; input_param.ReadOnly = False; input_param.BitSize = 8; input_param.DataSize = 1; input_param.ReadOnly = False; input_param.BitSize = 8; input_param.DataSize = 1; input_param.ReadOnly = False; input_param.BitSize = 8; input_param.DataSize = 1; input_param.ReadOnly = False; input_param.BitSize = 8; input_param.DataSize = 1; input_param.ReadOnly = False; input_param.BitSize = 8; input_param.DataSize = 1; output_param.ReadOnly = False; output_param.BitSize = 8; output_param.DataSize = 1; output_param.ReadOnly = False; output_param.BitSize = 8; output_param.DataSize = 1; output_param.ReadOnly = False; output_param.BitSize = 8;
            output_param.DataSize = 1; output_param.ReadOnly = False; output_param.BitSize = 8; output_param.DataSize = 1; output_param.ReadOnly = False; output_param.BitSize = 8; output_param.DataSize = 1; output_param.ReadOnly = False; output_param.BitSize = 8; output_param.DataSize = 1; output_param.ReadOnly = False; output_param.BitSize = 8; output_param.DataSize = 1; output_param.ReadOnly = False; output_param.BitSize = 8; output_param.DataSize = 1; output_param.ReadOnly = False; output_param.BitSize = 8; output_param.DataSize = 1; output_param.ReadOnly = False; output_param.BitSize = 8; output_param.DataSize = 1; input_param.Name = 'input_param'; input_param.HelpString = ''; input_param.ReadOnly = False; input_param.BitSize = 8; input_param.DataSize = 1; input_param.DataType = 'BYTE'; input_param.Name = 'input_param'; input_param.HelpString = ''; input_param.ReadOnly = False; input_param.BitSize = 8; input_param.DataSize = 1; input_param.DataType = 'BYTE'; input_param.Name = 'input_param'; input_param.HelpString = ''; input_param.ReadOnly = False; input_param.BitSize = 8; input_param.DataSize = 1; input_param.DataType = 'BYTE';
            input_param.Name = 'input_param'; input_param.HelpString = ''; input_param.ReadOnly = False; input_param.BitSize = 8; input_param.DataSize = 1; input_param.DataType = 'BYTE'; input_param.Name = 'input_param'; input_param.HelpString = ''; input_param.ReadOnly = False; input_param.BitSize = 8; input_param.DataSize = 1; input_param.DataType = 'BYTE'; input_param.Name = 'input_param'; input_param.HelpString = ''; input_param.ReadOnly = False; input_param.BitSize = 8; input_param.DataSize = 1; input_param.DataType = 'BYTE'; input_param.Name = 'input_param'; input_param.HelpString = ''; input_param.ReadOnly = False; input_param.BitSize = 8; input_param.DataSize = 1; input_param.DataType = 'BYTE'; input_param.Name = 'input_param'; input_param.HelpString = ''; input_param.ReadOnly = False; input_param.BitSize = 8; input_param.DataSize = 1; input_param.DataType = 'BYTE'; input_param.Name = 'input_param'; input_param.HelpString = ''; input_param.ReadOnly = False; input_param.BitSize = 8; input_param.DataSize = 1; input_param.DataType = 'BYTE'; input_param.Name = 'input_param'; input_param.HelpString = ''; input_param.ReadOnly = False; input_param.BitSize = 8;
            input_param.DataSize = 1; input_param.DataType = 'BYTE'; input_param.Name = 'input_param'; input_param.HelpString = ''; input_param.ReadOnly = False; input_param.BitSize = 8; input_param.DataSize = 1; input_param.DataType = 'BYTE'; input_param.Name = 'input_param'; input_param.HelpString = ''; input_param.ReadOnly = False; input_param.BitSize = 8; input_param.DataSize = 1; input_param.DataType = 'BYTE'; input_param.Name = 'input_param'; input_param.HelpString = ''; input_param.ReadOnly = False; input_param.BitSize = 8; input_param.DataSize = 1; input_param.DataType = 'BYTE'; input_param.Name = 'input_param'; input_param.HelpString = ''; input_param.ReadOnly = False; input_param.BitSize = 8; input_param.DataSize = 1; input_param.DataType = 'BYTE'; input_param.Name = 'input_param'; input_param.HelpString = ''; input_param.ReadOnly = False; input_param.BitSize = 8; input_param.DataSize = 1; input_param.DataType = 'BYTE'; input_param.Name = 'input_param'; input_param.HelpString = ''; input_param.ReadOnly = False; input_param.BitSize = 8; input_param.DataSize = 1; input_param.DataType = 'BYTE'; input_param.Name = 'input_param'; input_param.HelpString = '';
            input_param.ReadOnly = False; input_param.BitSize = 8; input_param.DataSize = 1; input_param.DataType = 'BYTE'; input_param.Name = 'input_param'; input_param.HelpString = ''; input_param.ReadOnly = False; input_param.BitSize = 8; input_param.DataSize = 1; input_param.DataType = 'BYTE'; input_param.Name = 'input_param'; input_param.HelpString = ''; input_param.ReadOnly = False; input_param.BitSize = 8; input_param.DataSize = 1; input_param.DataType = 'BYTE'; input_param.Name = 'input_param'; input_param.HelpString = ''; input_param.ReadOnly = False; input_param.BitSize = 8; input_param.DataSize = 1; input_param.DataType = 'BYTE'; input_param.Name = 'input_param'; input_param.HelpString = ''; input_param.ReadOnly = False; input_param.BitSize = 8; input_param.DataSize = 1; input_param.DataType = 'BYTE'; input_param.Name = 'input_param'; input_param.HelpString = ''; input_param.ReadOnly = False; input_param.BitSize = 8; input_param.DataSize = 1; input_param.DataType = 'BYTE'; input_param.Name = 'input_param'; input_param.HelpString = ''; input_param.ReadOnly = False; input_param.BitSize = 8; input_param.DataSize = 1; input_param.DataType = 'BYTE';
            input_param.Name = 'input_param'; input_param.HelpString = ''; input_param.ReadOnly = False; input_param.BitSize = 8; input_param.DataSize = 1; input_param.DataType = 'BYTE'; input_param.Name = 'input_param'; input_param.HelpString = ''; input_param.ReadOnly = False; input_param.BitSize = 8; input_param.DataSize = 1; input_param.DataType = 'BYTE'; input_param.Name = 'input_param'; input_param.HelpString = ''; input_param.ReadOnly = False; input_param.BitSize = 8; input_param.DataSize = 1; input_param.DataType = 'BYTE'; input_param.Name = 'input_param'; input_param.HelpString = ''; input_param.ReadOnly = False; input_param.BitSize = 8; input_param.DataSize = 1; input_param.DataType = 'BYTE'; input_param.Name = 'input_param'; input_param.HelpString = ''; input_param.ReadOnly = False; input_param.BitSize = 8; input_param.DataSize = 1; input_param.DataType = 'BYTE'; input_param.Name = 'input_param'; input_param.HelpString = ''; input_param.ReadOnly = False; input_param.BitSize = 8; input_param.DataSize = 1; input_param.DataType = 'BYTE'; input_param.Name = 'input_param'; input_param.HelpString = ''; input_param.ReadOnly = False; input_param.BitSize = 8;
            input_param.DataSize = 1; input_param.DataType = 'BYTE'; input_param.Name = 'input_param'; input_param.HelpString = ''; input_param.ReadOnly = False; input_param.BitSize = 8; input_param.DataSize = 1; input_param.DataType = 'BYTE'; input_param.Name = 'input_param'; input_param.HelpString = ''; input_param.ReadOnly = False; input_param.BitSize = 8; input_param.DataSize = 1; input_param.DataType = 'BYTE'; input_param.Name = 'input_param'; input_param.HelpString = ''; input_param.ReadOnly = False; input_param.BitSize = 8; input_param.DataSize = 1; input_param.DataType = 'BYTE'; input_param.Name = 'input_param'; input_param.HelpString = ''; input_param.ReadOnly = False; input_param.BitSize = 8; input_param.DataSize = 1; input_param.DataType = 'BYTE'; input_param.Name = 'input_param'; input_param.HelpString = ''; input_param.ReadOnly = False; input_param.BitSize = 8; input_param.DataSize = 1; input_param.DataType = 'BYTE'; input_param.Name = 'input_param'; input_param.HelpString = ''; input_param.ReadOnly = False; input_param.BitSize = 8; input_param.DataSize = 1; input_param.DataType = 'BYTE'; input_param.Name = 'input_param'; input_param.HelpString = '';
            input_param.ReadOnly = False; input_param.BitSize = 8; input_param.DataSize = 1; input_param.DataType = 'BYTE'; input_param.Name = 'input_param'; input_param.HelpString = ''; input_param.ReadOnly = False; input_param.BitSize = 8; input_param.DataSize = 1; input_param.DataType = 'BYTE'; input_param.Name = 'input_param'; input_param.HelpString = ''; input_param.ReadOnly = False; input_param.BitSize = 8; input_param.DataSize = 1; input_param.DataType = 'BYTE'; input_param.Name = 'input_param'; input_param.HelpString = ''; input_param.ReadOnly = False; input_param.BitSize = 8; input_param.DataSize = 1; input_param.DataType = 'BYTE'; input_param.Name = 'input_param'; input_param.HelpString = ''; input_param.ReadOnly = False; input_param.BitSize = 8; input_param.DataSize = 1; input_param.DataType = 'BYTE'; input_param.Name = 'input_param'; input_param.HelpString = ''; input_param.ReadOnly = False; input_param.BitSize = 8; input_param.DataSize = 1; input_param.DataType = 'BYTE'; input_param.Name = 'input_param'; input_param.HelpString = ''; input_param.ReadOnly = False; input_param.BitSize = 8; input_param.DataSize = 1; input_param.DataType = 'BYTE';
            input_param.Name = 'input_param'; input_param.HelpString = ''; input_param.ReadOnly = False; input_param.BitSize = 8; input_param.DataSize = 1; input_param.DataType = 'BYTE'; input_param.Name = 'input_param'; input_param.HelpString = ''; input_param.ReadOnly = False; input_param.BitSize = 8; input_param.DataSize = 1; input_param.DataType = 'BYTE'; input_param.Name = 'input_param'; input_param.HelpString = ''; input_param.ReadOnly = False; input_param.BitSize = 8; input_param.DataSize = 1; input_param.DataType = 'BYTE'; input_param.Name = 'input_param'; input_param.HelpString = ''; input_param.ReadOnly = False; input_param.BitSize = 8; input_param.DataSize = 1; input_param.DataType = 'BYTE'; input_param.Name = 'input_param'; input_param.HelpString = ''; input_param.ReadOnly = False; input_param.BitSize = 8; input_param.DataSize = 1; input_param.DataType = 'BYTE'; input_param.Name = 'input_param'; input_param.HelpString = ''; input_param.ReadOnly = False; input_param.BitSize = 8; input_param.DataSize = 1; input_param.DataType = 'BYTE'; input_param.Name = 'input_param'; input_param.HelpString = ''; input_param.ReadOnly = False; input_param.BitSize = 8;
            input_param.DataSize = 1; input_param.DataType = 'BYTE'; input_param.Name = 'input_param'; input_param.HelpString = ''; input_param.ReadOnly = False; input_param.BitSize = 8; input_param.DataSize = 1; input_param.DataType = 'BYTE'; input_param.Name = 'input_param'; input_param.HelpString = ''; input_param.ReadOnly = False; input_param.BitSize = 8; input_param.DataSize = 1; input_param.DataType = 'BYTE'; input_param.Name = 'input_param'; input_param.HelpString = ''; input_param.ReadOnly = False; input_param.BitSize = 8; input_param.DataSize = 1; input_param.DataType = 'BYTE'; input_param.Name = 'input_param'; input_param.HelpString = ''; input_param.ReadOnly = False; input_param.BitSize = 8; input_param.DataSize = 1; input_param.DataType = 'BYTE'; input_param.Name = 'input_param'; input_param.HelpString = ''; input_param.ReadOnly = False; input_param.BitSize = 8; input_param.DataSize = 1; input_param.DataType = 'BYTE'; input_param.Name = 'input_param'; input_param.HelpString = ''; input_param.ReadOnly = False; input_param.BitSize = 8; input_param.DataSize = 1; input_param.DataType = 'BYTE'; input_param.Name = 'input_param'; input_param.HelpString = '';
            input_param.ReadOnly = False; input_param.BitSize = 8; input_param.DataSize = 1; input_param.DataType = 'BYTE'; input_param.Name = 'input_param'; input_param.HelpString = ''; input_param.ReadOnly = False; input_param.BitSize = 8; input_param.DataSize = 1; input_param.DataType = 'BYTE'; input_param.Name = 'input_param'; input_param.HelpString = ''; input_param.ReadOnly = False; input_param.BitSize = 8; input_param.DataSize = 1; input_param.DataType = 'BYTE'; input_param.Name = 'input_param'; input_param.HelpString = ''; input_param.ReadOnly = False; input_param.BitSize = 8; input_param.DataSize = 1; input_param.DataType = 'BYTE'; input_param.Name = 'input_param'; input_param.HelpString = ''; input_param.ReadOnly = False; input_param.BitSize = 8; input_param.DataSize = 1; input_param.DataType = 'BYTE'; input_param.Name = 'input_param'; input_param.HelpString = ''; input_param.ReadOnly = False; input_param.BitSize = 8; input_param.DataSize = 1; input_param.DataType = 'BYTE'; input_param.Name = 'input_param'; input_param.HelpString = ''; input_param.ReadOnly = False; input_param.BitSize = 8; input_param.DataSize = 1; input_param.DataType = 'BYTE';
            input_param.Name = 'input_param'; input_param.HelpString = ''; input_param.ReadOnly = False; input_param.BitSize = 8; input_param.DataSize = 1; input_param.DataType = 'BYTE'; input_param.Name = 'input_param'; input_param.HelpString = ''; input_param.ReadOnly = False; input_param.BitSize = 8; input_param.DataSize = 1; input_param.DataType = 'BYTE'; input_param.Name = 'input_param'; input_param.HelpString = ''; input_param.ReadOnly = False; input_param.BitSize = 8; input_param.DataSize = 1; input_param.DataType = 'BYTE'; input_param.Name = 'input_param'; input_param.HelpString = ''; input_param.ReadOnly = False; input_param.BitSize = 8; input_param.DataSize = 1; input_param.DataType = 'BYTE'; input_param.Name = 'input_param'; input_param.HelpString = ''; input_param.ReadOnly = False; input_param.BitSize = 8; input_param.DataSize = 1; input_param.DataType = 'BYTE'; input_param.Name = 'input_param'; input_param.HelpString = ''; input_param.ReadOnly = False; input_param.BitSize = 8; input_param.DataSize = 1; input_param.DataType = 'BYTE'; input_param.Name = 'input_param'; input_param.HelpString = ''; input_param.ReadOnly = False; input_param.BitSize = 8;
            input_param.DataSize = 1; input_param.DataType = 'BYTE'; input_param.Name = 'input_param'; input_param.HelpString = ''; input_param.ReadOnly = False; input_param.BitSize = 8; input_param.DataSize = 1; input_param.DataType = 'BYTE'; input_param.Name = 'input_param'; input_param.HelpString = ''; input_param.ReadOnly = False; input_param.BitSize = 8; input_param.DataSize = 1; input_param.DataType = 'BYTE'; input_param.Name = 'input_param'; input_param.HelpString = ''; input_param.ReadOnly = False; input_param.BitSize = 8; input_param.DataSize = 1; input_param.DataType = 'BYTE'; input_param.Name = 'input_param'; input_param.HelpString = ''; input_param.ReadOnly = False; input_param.BitSize = 8; input_param.DataSize = 1; input_param.DataType = 'BYTE'; input_param.Name = 'input_param'; input_param.HelpString = ''; input_param.ReadOnly = False; input_param.BitSize = 8; input_param.DataSize = 1; input_param.DataType = 'BYTE'; input_param.Name = 'input_param'; input_param.HelpString = ''; input_param.ReadOnly = False; input_param.BitSize = 8; input_param.DataSize = 1; input_param.DataType = 'BYTE'; input_param.Name = 'input_param'; input_param.HelpString = '';
            input_param.ReadOnly = False; input_param.BitSize = 8; input_param.DataSize = 1; input_param.DataType = 'BYTE'; input_param.Name = 'input_param'; input_param.HelpString = ''; input_param.ReadOnly = False; input_param.BitSize = 8; input_param.DataSize = 1; input_param.DataType = 'BYTE'; input_param.Name = 'input_param'; input_param.HelpString = ''; input_param.ReadOnly = False; input_param.BitSize = 8; input_param.DataSize = 1; input_param.DataType = 'BYTE'; input_param.Name = 'input_param'; input_param.HelpString = ''; input_param.ReadOnly = False; input_param.BitSize = 8; input_param.DataSize = 1; input_param.DataType = 'BYTE'; input_param.Name = 'input_param'; input_param.HelpString = ''; input_param.ReadOnly = False; input_param.BitSize = 8; input_param.DataSize = 1; input_param.DataType = 'BYTE'; input_param.Name = 'input_param'; input_param.HelpString = ''; input_param.ReadOnly = False; input_param.BitSize = 8; input_param.DataSize = 1; input_param.DataType = 'BYTE'; input_param.Name = 'input_param'; input_param.HelpString = ''; input_param.ReadOnly = False; input_param.BitSize = 8; input_param.DataSize = 1; input_param.DataType = 'BYTE';
            input_param.Name = 'input_param'; input_param.HelpString = ''; input_param.ReadOnly = False; input_param.BitSize = 8; input_param.DataSize = 1; input_param.DataType = 'BYTE'; input_param.Name = 'input_param'; input_param.HelpString = ''; input_param.ReadOnly = False; input_param.BitSize = 8; input_param.DataSize = 1; input_param.DataType = 'BYTE'; input_param.Name = 'input_param'; input_param.HelpString = ''; input_param.ReadOnly = False; input_param.BitSize = 8; input_param.DataSize = 1; input_param.DataType = 'BYTE'; input_param.Name = 'input_param'; input_param.HelpString = ''; input_param.ReadOnly = False; input_param.BitSize = 8; input_param.DataSize = 1; input_param.DataType = 'BYTE'; input_param.Name = 'input_param'; input_param.HelpString = ''; input_param.ReadOnly = False; input_param.BitSize = 8; input_param.DataSize = 1; input_param.DataType = 'BYTE'; input_param.Name = 'input_param'; input_param.HelpString = ''; input_param.ReadOnly = False; input_param.BitSize = 8; input_param.DataSize = 1; input_param.DataType = 'BYTE'; input_param.Name = 'input_param'; input_param.HelpString = ''; input_param.ReadOnly = False; input_param.BitSize = 8;
            input_param.DataSize = 1; input_param.DataType = 'BYTE'; input_param.Name = 'input_param'; input_param.HelpString = ''; input_param.ReadOnly = False; input_param.BitSize = 8; input_param.DataSize = 1; input_param.DataType = 'BYTE'; input_param.Name = 'input_param'; input_param.HelpString = ''; input_param.ReadOnly = False; input_param.BitSize = 8; input_param.DataSize = 1; input_param.DataType = 'BYTE'; input_param.Name = 'input_param'; input_param.HelpString = ''; input_param.ReadOnly = False; input_param.BitSize = 8; input_param.DataSize = 1; input_param.DataType = 'BYTE'; input_param.Name = 'input_param'; input_param.HelpString = ''; input_param.ReadOnly = False; input_param.BitSize = 8; input_param.DataSize = 1; input_param.DataType = 'BYTE'; input_param.Name = 'input_param'; input_param.HelpString = ''; input_param.ReadOnly = False; input_param.BitSize = 8; input_param.DataSize = 1; input_param.DataType = 'BYTE'; input_param.Name = 'input_param'; input_param.HelpString = ''; input_param.ReadOnly = False; input_param.BitSize = 8; input_param.DataSize = 1; input_param.DataType = 'BYTE'; input_param.Name = 'input_param'; input_param.HelpString = '';
            input_param.ReadOnly = False; input_param.BitSize = 8; input_param.DataSize = 1; input_param.DataType = 'BYTE'; input_param.Name = 'input_param'; input_param.HelpString = ''; input_param.ReadOnly = False; input_param.BitSize = 8; input_param.DataSize = 1; input_param.DataType = 'BYTE'; input_param.Name = 'input_param'; input_param.HelpString = ''; input_param.ReadOnly = False; input_param.BitSize = 8; input_param.DataSize = 1; input_param.DataType = 'BYTE'; input_param.Name = 'input_param'; input_param.HelpString = ''; input_param.ReadOnly = False; input_param.BitSize = 8; input_param.DataSize = 1; input_param.DataType = 'BYTE'; input_param.Name = 'input_param'; input_param.HelpString = ''; input_param.ReadOnly = False; input_param.BitSize = 8; input_param.DataSize = 1; input_param.DataType = 'BYTE'; input_param.Name = 'input_param'; input_param.HelpString = ''; input_param.ReadOnly = False; input_param.BitSize = 8; input_param.DataSize = 1; input_param.DataType = 'BYTE'; input_param.Name = 'input_param'; input_param.HelpString = ''; input_param.ReadOnly = False; input_param.BitSize = 8; input_param.DataSize = 1; input_param.DataType = 'BYTE';
            input_param.Name = 'input_param'; input_param.HelpString = ''; input_param.ReadOnly = False; input_param.BitSize = 8; input_param.DataSize = 1; input_param.DataType = 'BYTE'; input_param.Name = 'input_param'; input_param.HelpString = ''; input_param.ReadOnly = False; input_param.BitSize = 8; input_param.DataSize = 1; input_param.DataType = 'BYTE'; input_param.Name = 'input_param'; input_param.HelpString = ''; input_param.ReadOnly = False; input_param.BitSize = 8; input_param.DataSize = 1; input_param.DataType = 'BYTE'; input_param.Name = 'input_param'; input_param.HelpString = ''; input_param.ReadOnly = False; input_param.BitSize = 8; input_param.DataSize = 1; input_param.DataType = 'BYTE'; input_param.Name = 'input_param'; input_param.HelpString = ''; input_param.ReadOnly = False; input_param.BitSize = 8; input_param.DataSize = 1; input_param.DataType = 'BYTE'; input_param.Name = 'input_param'; input_param.HelpString = ''; input_param.ReadOnly = False; input_param.BitSize = 8; input_param.DataSize = 1; input_param.DataType = 'BYTE'; input_param.Name = 'input_param'; input_param.HelpString = ''; input_param.ReadOnly = False; input_param.BitSize = 8;
            input_param.DataSize = 1; input_param.DataType = 'BYTE'; input_param.Name = 'input_param'; input_param.HelpString = ''; input_param.ReadOnly = False; input_param.BitSize = 8; input_param.DataSize = 1; input_param.DataType = 'BYTE'; input_param.Name = 'input_param'; input_param.HelpString = ''; input_param.ReadOnly = False; input_param.BitSize = 8; input_param.DataSize = 1; input_param.DataType = 'BYTE'; input_param.Name = 'input_param'; input_param.HelpString = ''; input_param.ReadOnly = False; input_param.BitSize = 8; input_param.DataSize = 1; input_param.DataType = 'BYTE'; input_param.Name = 'input_param'; input_param.HelpString = ''; input_param.ReadOnly = False; input_param.BitSize = 8; input_param.DataSize = 1; input_param.DataType = 'BYTE'; input_param.Name = 'input_param'; input_param.HelpString = ''; input_param.ReadOnly = False; input_param.BitSize = 8; input_param.DataSize = 1; input_param.DataType = 'BYTE'; input_param.Name = 'input_param'; input_param.HelpString = ''; input_param.ReadOnly = False; input_param.BitSize = 8; input_param.DataSize = 1; input_param.DataType = 'BYTE'; input_param.Name = 'input_param'; input_param.HelpString = '';
            input_param.ReadOnly = False; input_param.BitSize = 8; input_param.DataSize = 1; input_param.DataType = 'BYTE'; input_param.Name = 'input_param'; input_param.HelpString = ''; input_param.ReadOnly = False; input_param.BitSize = 8; input_param.DataSize = 1; input_param.DataType = 'BYTE'; input_param.Name = 'input_param'; input_param.HelpString = ''; input_param.ReadOnly = False; input_param.BitSize = 8; input_param.DataSize = 1; input_param.DataType = 'BYTE'; input_param.Name = 'input_param'; input_param.HelpString = ''; input_param.ReadOnly = False; input_param.BitSize = 8; input_param.DataSize = 1; input_param.DataType = 'BYTE'; input_param.Name = 'input_param'; input_param.HelpString = ''; input_param.ReadOnly = False; input_param.BitSize = 8; input_param.DataSize = 1; input_param.DataType = 'BYTE'; input_param.Name = 'input_param'; input_param.HelpString = ''; input_param.ReadOnly = False; input_param.BitSize = 8; input_param.DataSize = 1; input_param.DataType = 'BYTE'; input_param.Name = 'input_param'; input_param.HelpString = ''; input_param.ReadOnly = False; input_param.BitSize = 8; input_param.DataSize = 1; input_param.DataType = 'BYTE';
            input_param.Name = 'input_param'; input_param.HelpString = ''; input_param.ReadOnly = False; input_param.BitSize = 8; input_param.DataSize = 1; input_param.DataType = 'BYTE'; output_param.Name = 'output_param'; output_param.HelpString = ''; output_param.ReadOnly = False; output_param.BitSize = 8; output_param.DataSize = 1; output_param.DataType = 'BYTE'; output_param.Name = 'output_param'; output_param.HelpString = ''; output_param.ReadOnly = False; output_param.BitSize = 8; output_param.DataSize = 1; output_param.DataType = 'BYTE'; output_param.Name = 'output_param'; output_param.HelpString = ''; output_param.ReadOnly = False; output_param.BitSize = 8; output_param.DataSize = 1; output_param.DataType = 'BYTE'; output_param.Name = 'output_param'; output_param.HelpString = ''; output_param.ReadOnly = False; output_param.BitSize = 8; output_param.DataSize = 1; output_param.DataType = 'BYTE'; output_param.Name = 'output_param'; output_param.HelpString = ''; output_param.ReadOnly = False; output_param.BitSize = 8; output_param.DataSize = 1; output_param.DataType = 'BYTE'; output_param.Name = 'output_param'; output_param.HelpString = ''; output_param.ReadOnly = False; output_param.BitSize = 8;
            output_param.DataSize = 1; output_param.DataType = 'BYTE'; output_param.Name = 'output_param'; output_param.HelpString = ''; output_param.ReadOnly = False; output_param.BitSize = 8; output_param.DataSize = 1; output_param.DataType = 'BYTE'; output_param.Name = 'output_param'; output_param.HelpString = ''; output_param.ReadOnly = False; output_param.BitSize = 8; output_param.DataSize = 1; output_param.DataType = 'BYTE'; output_param.Name = 'output_param'; output_param.HelpString = ''; output_param.ReadOnly = False; output_param.BitSize = 8; output_param.DataSize = 1; output_param.DataType = 'BYTE'; output_param.Name = 'output_param'; output_param.HelpString = ''; output_param.ReadOnly = False; output_param.BitSize = 8; output_param.DataSize = 1; output_param.DataType = 'BYTE'; ConfigVersion = 50660864
          input  iBCVInputs : BYTE  // input_param
          output oBCVOutputs : BYTE  // output_param
          unmapped channels: input_param, input_param, input_param, input_param, input_param, input_param, input_param, input_param, input_param, input_param, input_param, input_param, input_param, input_param, input_param, input_param, input_param, input_param, input_param, input_param, input_param, input_param, input_param, input_param, input_param, input_param, input_param, input_param, input_param, input_param, input_param, input_param, input_param, input_param, input_param, input_param, input_param, input_param, input_param, input_param,
            input_param, input_param, input_param, input_param, input_param, input_param, input_param, input_param, input_param, input_param, input_param, input_param, input_param, input_param, input_param, input_param, input_param, input_param, input_param, input_param, input_param, input_param, input_param, input_param, input_param, input_param, input_param, input_param, input_param, input_param, input_param, input_param, input_param, input_param, input_param, input_param, input_param, input_param, input_param, input_param,
            input_param, input_param, input_param, input_param, input_param, input_param, input_param, input_param, input_param, input_param, input_param, input_param, input_param, input_param, input_param, input_param, input_param, input_param, input_param, input_param, input_param, input_param, input_param, input_param, input_param, input_param, input_param, input_param, input_param, input_param, input_param, input_param, input_param, input_param, input_param, input_param, input_param, input_param, input_param, input_param,
            input_param, input_param, input_param, output_param, output_param, output_param, output_param, output_param, output_param, output_param, output_param, output_param
      FestoManifold : CTEU-EP EtherNetIP bus node, Festo AG & Co. KG, order no. CTEU-EP, version Major Revision=16#2, Minor Revision = 16#2
          settings: INITIALIZED = TRUE; IP address of Target = [16#C0,16#A8,16#0A,16#6E]; Keying.Check Vendor Code = FALSE; Keying.Check Product Code = FALSE; Keying.Check Major Revision = FALSE; Keying.Check Minor Revision = FALSE; RequiredConfigVersion = 50660864; Number of Connections = 1; Connection Settings.Requested packet intervall = 10000 µs; Connection Settings.OT Connection Parameters = 18446; Connection Settings.TO Connection Parameters = 18442; Connection Settings.Connection Flags = 1056; Connection Settings.Connection Path Size = 8; Connection Settings.Config#2 Size = 38; Single Port Inputs 8 bytesParam8.ReadOnly = False; Single Port Inputs 8 bytesParam8.BitSize = 8; Single Port Inputs 8 bytesParam8.DataSize = 1; Single Port Inputs 8 bytesParam9.ReadOnly = False; Single Port Inputs 8 bytesParam9.BitSize = 8; Single Port Inputs 8 bytesParam9.DataSize = 1; Single Port Inputs 8 bytesParam10.ReadOnly = False; Single Port Inputs 8 bytesParam10.BitSize = 8; Single Port Inputs 8 bytesParam10.DataSize = 1; Single Port Inputs 8 bytesParam11.ReadOnly = False; Single Port Inputs 8 bytesParam11.BitSize = 8; Single Port Inputs 8 bytesParam11.DataSize = 1; Single Port Inputs 8 bytesParam12.ReadOnly = False; Single Port Inputs 8 bytesParam12.BitSize = 8; Single Port Inputs 8 bytesParam12.DataSize = 1; Single Port Inputs 8 bytesParam13.ReadOnly = False; Single Port Inputs 8 bytesParam13.BitSize = 8; Single Port Inputs 8 bytesParam13.DataSize = 1; Single Port Inputs 8 bytesParam14.ReadOnly = False; Single Port Inputs 8 bytesParam14.BitSize = 8; Single Port Inputs 8 bytesParam14.DataSize = 1; Single Port Inputs 8 bytesParam15.ReadOnly = False; Single Port Inputs 8 bytesParam15.BitSize = 8; Single Port Inputs 8 bytesParam15.DataSize = 1; Single Port Outputs 8bytesParam8.ReadOnly = False; Single Port Outputs 8bytesParam8.BitSize = 8;
            Single Port Outputs 8bytesParam8.DataSize = 1; Single Port Outputs 8bytesParam9.ReadOnly = False; Single Port Outputs 8bytesParam9.BitSize = 8; Single Port Outputs 8bytesParam9.DataSize = 1; Single Port Outputs 8bytesParam10.ReadOnly = False; Single Port Outputs 8bytesParam10.BitSize = 8; Single Port Outputs 8bytesParam10.DataSize = 1; Single Port Outputs 8bytesParam11.ReadOnly = False; Single Port Outputs 8bytesParam11.BitSize = 8; Single Port Outputs 8bytesParam11.DataSize = 1; Single Port Outputs 8bytesParam12.ReadOnly = False; Single Port Outputs 8bytesParam12.BitSize = 8; Single Port Outputs 8bytesParam12.DataSize = 1; Single Port Outputs 8bytesParam13.ReadOnly = False; Single Port Outputs 8bytesParam13.BitSize = 8; Single Port Outputs 8bytesParam13.DataSize = 1; Single Port Outputs 8bytesParam14.ReadOnly = False; Single Port Outputs 8bytesParam14.BitSize = 8; Single Port Outputs 8bytesParam14.DataSize = 1; Single Port Outputs 8bytesParam15.ReadOnly = False; Single Port Outputs 8bytesParam15.BitSize = 8; Single Port Outputs 8bytesParam15.DataSize = 1; Single Port Inputs 8 bytesParam8.Name = 'Single Port Inputs 8 bytesParam8'; Single Port Inputs 8 bytesParam8.HelpString = ''; Single Port Inputs 8 bytesParam8.ReadOnly = False; Single Port Inputs 8 bytesParam8.BitSize = 8; Single Port Inputs 8 bytesParam8.DataSize = 1; Single Port Inputs 8 bytesParam8.DataType = 'BYTE'; Single Port Inputs 8 bytesParam9.Name = 'Single Port Inputs 8 bytesParam9'; Single Port Inputs 8 bytesParam9.HelpString = ''; Single Port Inputs 8 bytesParam9.ReadOnly = False; Single Port Inputs 8 bytesParam9.BitSize = 8; Single Port Inputs 8 bytesParam9.DataSize = 1; Single Port Inputs 8 bytesParam9.DataType = 'BYTE'; Single Port Inputs 8 bytesParam10.Name = 'Single Port Inputs 8 bytesParam10'; Single Port Inputs 8 bytesParam10.HelpString = ''; Single Port Inputs 8 bytesParam10.ReadOnly = False; Single Port Inputs 8 bytesParam10.BitSize = 8; Single Port Inputs 8 bytesParam10.DataSize = 1; Single Port Inputs 8 bytesParam10.DataType = 'BYTE';
            Single Port Inputs 8 bytesParam11.Name = 'Single Port Inputs 8 bytesParam11'; Single Port Inputs 8 bytesParam11.HelpString = ''; Single Port Inputs 8 bytesParam11.ReadOnly = False; Single Port Inputs 8 bytesParam11.BitSize = 8; Single Port Inputs 8 bytesParam11.DataSize = 1; Single Port Inputs 8 bytesParam11.DataType = 'BYTE'; Single Port Inputs 8 bytesParam12.Name = 'Single Port Inputs 8 bytesParam12'; Single Port Inputs 8 bytesParam12.HelpString = ''; Single Port Inputs 8 bytesParam12.ReadOnly = False; Single Port Inputs 8 bytesParam12.BitSize = 8; Single Port Inputs 8 bytesParam12.DataSize = 1; Single Port Inputs 8 bytesParam12.DataType = 'BYTE'; Single Port Inputs 8 bytesParam13.Name = 'Single Port Inputs 8 bytesParam13'; Single Port Inputs 8 bytesParam13.HelpString = ''; Single Port Inputs 8 bytesParam13.ReadOnly = False; Single Port Inputs 8 bytesParam13.BitSize = 8; Single Port Inputs 8 bytesParam13.DataSize = 1; Single Port Inputs 8 bytesParam13.DataType = 'BYTE'; Single Port Inputs 8 bytesParam14.Name = 'Single Port Inputs 8 bytesParam14'; Single Port Inputs 8 bytesParam14.HelpString = ''; Single Port Inputs 8 bytesParam14.ReadOnly = False; Single Port Inputs 8 bytesParam14.BitSize = 8; Single Port Inputs 8 bytesParam14.DataSize = 1; Single Port Inputs 8 bytesParam14.DataType = 'BYTE'; Single Port Inputs 8 bytesParam15.Name = 'Single Port Inputs 8 bytesParam15'; Single Port Inputs 8 bytesParam15.HelpString = ''; Single Port Inputs 8 bytesParam15.ReadOnly = False; Single Port Inputs 8 bytesParam15.BitSize = 8; Single Port Inputs 8 bytesParam15.DataSize = 1; Single Port Inputs 8 bytesParam15.DataType = 'BYTE'; Single Port Outputs 8bytesParam8.Name = 'Single Port Outputs 8bytesParam8'; Single Port Outputs 8bytesParam8.HelpString = ''; Single Port Outputs 8bytesParam8.ReadOnly = False; Single Port Outputs 8bytesParam8.BitSize = 8; Single Port Outputs 8bytesParam8.DataSize = 1; Single Port Outputs 8bytesParam8.DataType = 'BYTE'; Single Port Outputs 8bytesParam9.Name = 'Single Port Outputs 8bytesParam9'; Single Port Outputs 8bytesParam9.HelpString = ''; Single Port Outputs 8bytesParam9.ReadOnly = False; Single Port Outputs 8bytesParam9.BitSize = 8;
            Single Port Outputs 8bytesParam9.DataSize = 1; Single Port Outputs 8bytesParam9.DataType = 'BYTE'; Single Port Outputs 8bytesParam10.Name = 'Single Port Outputs 8bytesParam10'; Single Port Outputs 8bytesParam10.HelpString = ''; Single Port Outputs 8bytesParam10.ReadOnly = False; Single Port Outputs 8bytesParam10.BitSize = 8; Single Port Outputs 8bytesParam10.DataSize = 1; Single Port Outputs 8bytesParam10.DataType = 'BYTE'; Single Port Outputs 8bytesParam11.Name = 'Single Port Outputs 8bytesParam11'; Single Port Outputs 8bytesParam11.HelpString = ''; Single Port Outputs 8bytesParam11.ReadOnly = False; Single Port Outputs 8bytesParam11.BitSize = 8; Single Port Outputs 8bytesParam11.DataSize = 1; Single Port Outputs 8bytesParam11.DataType = 'BYTE'; Single Port Outputs 8bytesParam12.Name = 'Single Port Outputs 8bytesParam12'; Single Port Outputs 8bytesParam12.HelpString = ''; Single Port Outputs 8bytesParam12.ReadOnly = False; Single Port Outputs 8bytesParam12.BitSize = 8; Single Port Outputs 8bytesParam12.DataSize = 1; Single Port Outputs 8bytesParam12.DataType = 'BYTE'; Single Port Outputs 8bytesParam13.Name = 'Single Port Outputs 8bytesParam13'; Single Port Outputs 8bytesParam13.HelpString = ''; Single Port Outputs 8bytesParam13.ReadOnly = False; Single Port Outputs 8bytesParam13.BitSize = 8; Single Port Outputs 8bytesParam13.DataSize = 1; Single Port Outputs 8bytesParam13.DataType = 'BYTE'; Single Port Outputs 8bytesParam14.Name = 'Single Port Outputs 8bytesParam14'; Single Port Outputs 8bytesParam14.HelpString = ''; Single Port Outputs 8bytesParam14.ReadOnly = False; Single Port Outputs 8bytesParam14.BitSize = 8; Single Port Outputs 8bytesParam14.DataSize = 1; Single Port Outputs 8bytesParam14.DataType = 'BYTE'; Single Port Outputs 8bytesParam15.Name = 'Single Port Outputs 8bytesParam15'; Single Port Outputs 8bytesParam15.HelpString = ''; Single Port Outputs 8bytesParam15.ReadOnly = False; Single Port Outputs 8bytesParam15.BitSize = 8; Single Port Outputs 8bytesParam15.DataSize = 1; Single Port Outputs 8bytesParam15.DataType = 'BYTE'; ConfigVersion = 50660864
          output oPBar1Extend : BOOL  // Single Port Outputs 8bytesParam8.Bit0
          output oPbar1Retract : BOOL  // Single Port Outputs 8bytesParam8.Bit1
          output opBar2Extend : BOOL  // Single Port Outputs 8bytesParam8.Bit2
          output opbar2Retract : BOOL  // Single Port Outputs 8bytesParam8.Bit3
          output oSealBarExtend : BOOL  // Single Port Outputs 8bytesParam8.Bit4
          output oSealBarRetract : BOOL  // Single Port Outputs 8bytesParam8.Bit5
          output oLPAOn : BOOL  // Single Port Outputs 8bytesParam8.Bit6
          output oHPAOn : BOOL  // Single Port Outputs 8bytesParam8.Bit7
          output oLoadPlateExtend : BOOL  // Single Port Outputs 8bytesParam9.Bit0
          output oLoadPlateRetract : BOOL  // Single Port Outputs 8bytesParam9.Bit1
          output oBOFUp : BOOL  // Single Port Outputs 8bytesParam9.Bit2
          output oBOFDown : BOOL  // Single Port Outputs 8bytesParam9.Bit3
          output oPrintHeadDown : BOOL  // Single Port Outputs 8bytesParam9.Bit4
          output oPrintHeadUp : BOOL  // Single Port Outputs 8bytesParam9.Bit5
          output oVacOn : BOOL  // Single Port Outputs 8bytesParam9.Bit6
          output oSealFlatUp : BOOL  // Single Port Outputs 8bytesParam10.Bit0
          output oSealFlatDown : BOOL  // Single Port Outputs 8bytesParam10.Bit1
          output oFrontLoadPlateToLoad : BOOL  // Single Port Outputs 8bytesParam10.Bit2
          output oFrontLoadPlateToDischarge : BOOL  // Single Port Outputs 8bytesParam10.Bit3
          output oLoadShelfUp : BOOL  // Single Port Outputs 8bytesParam10.Bit4
          output oLoadShelfDown : BOOL  // Single Port Outputs 8bytesParam10.Bit5
          output oIBDExtend : BOOL  // Single Port Outputs 8bytesParam10.Bit6
          output oIBDRetract : BOOL  // Single Port Outputs 8bytesParam10.Bit7
          output oFunnelOpen : BOOL  // Single Port Outputs 8bytesParam11.Bit0
          output oFunnelClose : BOOL  // Single Port Outputs 8bytesParam11.Bit1
          output oStagingFunnelOpen : BOOL  // Single Port Outputs 8bytesParam11.Bit2
          output oStagingFunnelClose : BOOL  // Single Port Outputs 8bytesParam11.Bit3
          output oIBDExtendWithFunnel : BOOL  // Single Port Outputs 8bytesParam11.Bit6
          output oIBDRetractWithFunnel : BOOL  // Single Port Outputs 8bytesParam11.Bit7
          unmapped channels: Single Port Inputs 8 bytesParam8, Single Port Inputs 8 bytesParam9, Single Port Inputs 8 bytesParam10, Single Port Inputs 8 bytesParam11, Single Port Inputs 8 bytesParam12, Single Port Inputs 8 bytesParam13, Single Port Inputs 8 bytesParam14, Single Port Inputs 8 bytesParam15, Single Port Outputs 8bytesParam8, Single Port Outputs 8bytesParam9, Single Port Outputs 8bytesParam10, Single Port Outputs 8bytesParam11, Single Port Outputs 8bytesParam12, Single Port Outputs 8bytesParam13, Single Port Outputs 8bytesParam14, Single Port Outputs 8bytesParam15
      IBD_Motor : SSM23IP-3EG, Applied Motion Products, Inc, order no. SSM23IP-3EG, version Major Revision=16#3, Minor Revision = 16#3 (disabled)
          settings: INITIALIZED = TRUE; IP address of Target = [16#C0,16#A8,16#0A,16#39]; MAC address of Target = [16#00,16#00,16#00,16#00,16#00,16#00]; Keying.Check Device Type = FALSE; Keying.Check Vendor Code = FALSE; Keying.Check Product Code = FALSE; Keying.Check Major Revision = FALSE; Keying.Check Minor Revision = FALSE; RequiredConfigVersion = 50660864; Number of Connections = 1; Connection Settings.Requested packet intervall = 10000 µs; Connection Settings.OT Connection Parameters = 18502; Connection Settings.TO Connection Parameters = 18490; Connection Settings.Connection Flags = 1056; Connection Settings.Connection Path Size = 8; Status Code.ReadOnly = False; Status Code.BitSize = 32; Status Code.DataSize = 4; Alarm Code.ReadOnly = False; Alarm Code.BitSize = 32; Alarm Code.DataSize = 4; Supply Voltage.ReadOnly = False; Supply Voltage.BitSize = 32; Supply Voltage.DataSize = 4; Actual Current.ReadOnly = False; Actual Current.BitSize = 32; Actual Current.DataSize = 4; Drive Temperature.ReadOnly = False; Drive Temperature.BitSize = 32; Drive Temperature.DataSize = 4; Encoder Position.ReadOnly = False; Encoder Position.BitSize = 32; Encoder Position.DataSize = 4; Absolute Position.ReadOnly = False; Absolute Position.BitSize = 32; Absolute Position.DataSize = 4; Position Error.ReadOnly = False; Position Error.BitSize = 32; Position Error.DataSize = 4; Actual Velocity.ReadOnly = False;
            Actual Velocity.BitSize = 32; Actual Velocity.DataSize = 4; Input Status (extended).ReadOnly = False; Input Status (extended).BitSize = 32; Input Status (extended).DataSize = 4; Input Status (main).ReadOnly = False; Input Status (main).BitSize = 32; Input Status (main).DataSize = 4; Output Status.ReadOnly = False; Output Status.BitSize = 32; Output Status.DataSize = 4; Analog Input 1.ReadOnly = False; Analog Input 1.BitSize = 32; Analog Input 1.DataSize = 4; Analog Input 2.ReadOnly = False; Analog Input 2.BitSize = 32; Analog Input 2.DataSize = 4; Command Word.ReadOnly = False; Command Word.BitSize = 32; Command Word.DataSize = 4; Jog Speed.ReadOnly = False; Jog Speed.BitSize = 32; Jog Speed.DataSize = 4; Jog Accel.ReadOnly = False; Jog Accel.BitSize = 32; Jog Accel.DataSize = 4; Jog Decel.ReadOnly = False; Jog Decel.BitSize = 32; Jog Decel.DataSize = 4; Point-to-Point Velocity.ReadOnly = False; Point-to-Point Velocity.BitSize = 32; Point-to-Point Velocity.DataSize = 4; Point-to-Point Acceleration.ReadOnly = False; Point-to-Point Acceleration.BitSize = 32; Point-to-Point Acceleration.DataSize = 4; Point-to-Point Deceleration.ReadOnly = False; Point-to-Point Deceleration.BitSize = 32; Point-to-Point Deceleration.DataSize = 4; Point-to-Point Distance.ReadOnly = False; Point-to-Point Distance.BitSize = 32;
            Point-to-Point Distance.DataSize = 4; Current Command.ReadOnly = False; Current Command.BitSize = 32; Current Command.DataSize = 4; SCL Command Letters.ReadOnly = False; SCL Command Letters.BitSize = 32; SCL Command Letters.DataSize = 4; Data/SCL Register 1.ReadOnly = False; Data/SCL Register 1.BitSize = 32; Data/SCL Register 1.DataSize = 4; Data/SCL Register 2.ReadOnly = False; Data/SCL Register 2.BitSize = 32; Data/SCL Register 2.DataSize = 4; Continuous Current.ReadOnly = False; Continuous Current.BitSize = 32; Continuous Current.DataSize = 4; Peak Current.ReadOnly = False; Peak Current.BitSize = 32; Peak Current.DataSize = 4; Reserved 3.ReadOnly = False; Reserved 3.BitSize = 32; Reserved 3.DataSize = 4; Reserved 4.ReadOnly = False; Reserved 4.BitSize = 32; Reserved 4.DataSize = 4; Status Code.Name = 'Status Code'; Status Code.HelpString = ''; Status Code.ReadOnly = False; Status Code.BitSize = 32; Status Code.DataSize = 4; Status Code.DataType = 'DINT'; Alarm Code.Name = 'Alarm Code'; Alarm Code.HelpString = ''; Alarm Code.ReadOnly = False; Alarm Code.BitSize = 32; Alarm Code.DataSize = 4; Alarm Code.DataType = 'DINT'; Supply Voltage.Name = 'Supply Voltage'; Supply Voltage.HelpString = ''; Supply Voltage.ReadOnly = False;
            Supply Voltage.BitSize = 32; Supply Voltage.DataSize = 4; Supply Voltage.DataType = 'DINT'; Actual Current.Name = 'Actual Current'; Actual Current.HelpString = ''; Actual Current.ReadOnly = False; Actual Current.BitSize = 32; Actual Current.DataSize = 4; Actual Current.DataType = 'DINT'; Drive Temperature.Name = 'Drive Temperature'; Drive Temperature.HelpString = ''; Drive Temperature.ReadOnly = False; Drive Temperature.BitSize = 32; Drive Temperature.DataSize = 4; Drive Temperature.DataType = 'DINT'; Encoder Position.Name = 'Encoder Position'; Encoder Position.HelpString = ''; Encoder Position.ReadOnly = False; Encoder Position.BitSize = 32; Encoder Position.DataSize = 4; Encoder Position.DataType = 'DINT'; Absolute Position.Name = 'Absolute Position'; Absolute Position.HelpString = ''; Absolute Position.ReadOnly = False; Absolute Position.BitSize = 32; Absolute Position.DataSize = 4; Absolute Position.DataType = 'DINT'; Position Error.Name = 'Position Error'; Position Error.HelpString = ''; Position Error.ReadOnly = False; Position Error.BitSize = 32; Position Error.DataSize = 4; Position Error.DataType = 'DINT'; Actual Velocity.Name = 'Actual Velocity'; Actual Velocity.HelpString = ''; Actual Velocity.ReadOnly = False; Actual Velocity.BitSize = 32; Actual Velocity.DataSize = 4; Actual Velocity.DataType = 'DINT'; Input Status (extended).Name = 'Input Status (extended)';
            Input Status (extended).HelpString = ''; Input Status (extended).ReadOnly = False; Input Status (extended).BitSize = 32; Input Status (extended).DataSize = 4; Input Status (extended).DataType = 'DINT'; Input Status (main).Name = 'Input Status (main)'; Input Status (main).HelpString = ''; Input Status (main).ReadOnly = False; Input Status (main).BitSize = 32; Input Status (main).DataSize = 4; Input Status (main).DataType = 'DINT'; Output Status.Name = 'Output Status'; Output Status.HelpString = ''; Output Status.ReadOnly = False; Output Status.BitSize = 32; Output Status.DataSize = 4; Output Status.DataType = 'DINT'; Analog Input 1.Name = 'Analog Input 1'; Analog Input 1.HelpString = ''; Analog Input 1.ReadOnly = False; Analog Input 1.BitSize = 32; Analog Input 1.DataSize = 4; Analog Input 1.DataType = 'DINT'; Analog Input 2.Name = 'Analog Input 2'; Analog Input 2.HelpString = ''; Analog Input 2.ReadOnly = False; Analog Input 2.BitSize = 32; Analog Input 2.DataSize = 4; Analog Input 2.DataType = 'DINT'; Command Word.Name = 'Command Word'; Command Word.HelpString = ''; Command Word.ReadOnly = False; Command Word.BitSize = 32; Command Word.DataSize = 4; Command Word.DataType = 'DINT'; Jog Speed.Name = 'Jog Speed'; Jog Speed.HelpString = ''; Jog Speed.ReadOnly = False; Jog Speed.BitSize = 32; Jog Speed.DataSize = 4;
            Jog Speed.DataType = 'DINT'; Jog Accel.Name = 'Jog Accel'; Jog Accel.HelpString = ''; Jog Accel.ReadOnly = False; Jog Accel.BitSize = 32; Jog Accel.DataSize = 4; Jog Accel.DataType = 'DINT'; Jog Decel.Name = 'Jog Decel'; Jog Decel.HelpString = ''; Jog Decel.ReadOnly = False; Jog Decel.BitSize = 32; Jog Decel.DataSize = 4; Jog Decel.DataType = 'DINT'; Point-to-Point Velocity.Name = 'Point-to-Point Velocity'; Point-to-Point Velocity.HelpString = ''; Point-to-Point Velocity.ReadOnly = False; Point-to-Point Velocity.BitSize = 32; Point-to-Point Velocity.DataSize = 4; Point-to-Point Velocity.DataType = 'DINT'; Point-to-Point Acceleration.Name = 'Point-to-Point Acceleration'; Point-to-Point Acceleration.HelpString = ''; Point-to-Point Acceleration.ReadOnly = False; Point-to-Point Acceleration.BitSize = 32; Point-to-Point Acceleration.DataSize = 4; Point-to-Point Acceleration.DataType = 'DINT'; Point-to-Point Deceleration.Name = 'Point-to-Point Deceleration'; Point-to-Point Deceleration.HelpString = ''; Point-to-Point Deceleration.ReadOnly = False; Point-to-Point Deceleration.BitSize = 32; Point-to-Point Deceleration.DataSize = 4; Point-to-Point Deceleration.DataType = 'DINT'; Point-to-Point Distance.Name = 'Point-to-Point Distance'; Point-to-Point Distance.HelpString = ''; Point-to-Point Distance.ReadOnly = False; Point-to-Point Distance.BitSize = 32; Point-to-Point Distance.DataSize = 4; Point-to-Point Distance.DataType = 'DINT'; Current Command.Name = 'Current Command'; Current Command.HelpString = ''; Current Command.ReadOnly = False;
            Current Command.BitSize = 32; Current Command.DataSize = 4; Current Command.DataType = 'DINT'; SCL Command Letters.Name = 'SCL Command Letters'; SCL Command Letters.HelpString = ''; SCL Command Letters.ReadOnly = False; SCL Command Letters.BitSize = 32; SCL Command Letters.DataSize = 4; SCL Command Letters.DataType = 'DINT'; Data/SCL Register 1.Name = 'Data/SCL Register 1'; Data/SCL Register 1.HelpString = ''; Data/SCL Register 1.ReadOnly = False; Data/SCL Register 1.BitSize = 32; Data/SCL Register 1.DataSize = 4; Data/SCL Register 1.DataType = 'DINT'; Data/SCL Register 2.Name = 'Data/SCL Register 2'; Data/SCL Register 2.HelpString = ''; Data/SCL Register 2.ReadOnly = False; Data/SCL Register 2.BitSize = 32; Data/SCL Register 2.DataSize = 4; Data/SCL Register 2.DataType = 'DINT'; Continuous Current.Name = 'Continuous Current'; Continuous Current.HelpString = ''; Continuous Current.ReadOnly = False; Continuous Current.BitSize = 32; Continuous Current.DataSize = 4; Continuous Current.DataType = 'DINT'; Peak Current.Name = 'Peak Current'; Peak Current.HelpString = ''; Peak Current.ReadOnly = False; Peak Current.BitSize = 32; Peak Current.DataSize = 4; Peak Current.DataType = 'DINT'; Reserved 3.Name = 'Reserved 3'; Reserved 3.HelpString = ''; Reserved 3.ReadOnly = False; Reserved 3.BitSize = 32; Reserved 3.DataSize = 4; Reserved 3.DataType = 'DINT'; Reserved 4.Name = 'Reserved 4';
            Reserved 4.HelpString = ''; Reserved 4.ReadOnly = False; Reserved 4.BitSize = 32; Reserved 4.DataSize = 4; Reserved 4.DataType = 'DINT'; ConfigVersion = 50660864
          input  iIBDMotorEIP : DINT  // Status Code
          output oIBDMotorEIP : DINT  // Command Word
          unmapped channels: Alarm Code, Supply Voltage, Actual Current, Drive Temperature, Encoder Position, Absolute Position, Position Error, Actual Velocity, Input Status (extended), Input Status (main), Output Status, Analog Input 1, Analog Input 2, Jog Speed, Jog Accel, Jog Decel, Point-to-Point Velocity, Point-to-Point Acceleration, Point-to-Point Deceleration, Point-to-Point Distance, Current Command, SCL Command Letters, Data/SCL Register 1, Data/SCL Register 2, Continuous Current, Peak Current, Reserved 3, Reserved 4
      Infeed_Conveyor_IO : Advantech - ADAM-6150EI, Advantech Co., Ltd., version Major Revision=16#1, Minor Revision = 16#1 (disabled)
          settings: INITIALIZED = TRUE; IP address of Target = [16#C0,16#A8,16#0A,16#46]; Keying.Check Minor Revision = FALSE; RequiredConfigVersion = 50660864; Number of Connections = 1; Connection Settings.Requested packet intervall (µs) = 10000; Connection Settings.OT Connection Parameters = 18440; Connection Settings.TO Connection Parameters = 18436; Connection Settings.Connection Flags = 1056; Connection Settings.Connection Path Size = 8; Heartbeat Multiplier = 1; IO Data (T->O)_Param0.ReadOnly = False; IO Data (T->O)_Param0.BitSize = 8; IO Data (T->O)_Param0.DataSize = 1; IO Data (T->O)_Param1.ReadOnly = False; IO Data (T->O)_Param1.BitSize = 8; IO Data (T->O)_Param1.DataSize = 1; IO Data (O->T)_Param0.ReadOnly = False; IO Data (O->T)_Param0.BitSize = 8; IO Data (O->T)_Param0.DataSize = 1; IO Data (O->T)_Param1.ReadOnly = False; IO Data (O->T)_Param1.BitSize = 8; IO Data (O->T)_Param1.DataSize = 1; IO Data (T->O)_Param0.Name = 'IO Data (T->O)_Param0'; IO Data (T->O)_Param0.HelpString = ''; IO Data (T->O)_Param0.ReadOnly = False; IO Data (T->O)_Param0.BitSize = 8; IO Data (T->O)_Param0.DataSize = 1; IO Data (T->O)_Param0.DataType = 'BYTE'; IO Data (T->O)_Param1.Name = 'IO Data (T->O)_Param1'; IO Data (T->O)_Param1.HelpString = ''; IO Data (T->O)_Param1.ReadOnly = False; IO Data (T->O)_Param1.BitSize = 8; IO Data (T->O)_Param1.DataSize = 1; IO Data (T->O)_Param1.DataType = 'BYTE'; IO Data (O->T)_Param0.Name = 'IO Data (O->T)_Param0'; IO Data (O->T)_Param0.HelpString = ''; IO Data (O->T)_Param0.ReadOnly = False; IO Data (O->T)_Param0.BitSize = 8; IO Data (O->T)_Param0.DataSize = 1;
            IO Data (O->T)_Param0.DataType = 'BYTE'; IO Data (O->T)_Param1.Name = 'IO Data (O->T)_Param1'; IO Data (O->T)_Param1.HelpString = ''; IO Data (O->T)_Param1.ReadOnly = False; IO Data (O->T)_Param1.BitSize = 8; IO Data (O->T)_Param1.DataSize = 1; IO Data (O->T)_Param1.DataType = 'BYTE'; ConfigVersion = 50660864
          input  iInfeedVFDRunning : BOOL  // IO Data (T->O)_Param0.Bit0
          input  iInfeedVFDNotFaulted : BOOL  // IO Data (T->O)_Param0.Bit1
          input  iInfeedFlightSensor : BOOL  // IO Data (T->O)_Param0.Bit4
          output oRunInfeedVFD : BOOL  // IO Data (O->T)_Param1.Bit0
          output oResetInfeedVFD : BOOL  // IO Data (O->T)_Param1.Bit1
          unmapped channels: IO Data (T->O)_Param0, IO Data (T->O)_Param1, IO Data (O->T)_Param0, IO Data (O->T)_Param1
      Keyence_BCV : Generic EtherNet/IP device, 3S - Smart Software Solutions GmbH, version 3.5.15.0 (disabled)
          settings: INITIALIZED = TRUE; IP address of Target = [16#C0,16#A8,16#0A,16#A1]; MAC address of Target = [16#00,16#00,16#00,16#00,16#00,16#00]; Keying.Compatibility Bit = FALSE; RequiredConfigVersion = 50660864; Number of Connections = 1; Connection Settings.Requested packet intervall (µs) = 10000; Connection Settings.OT Connection Parameters = 18514; Connection Settings.TO Connection Parameters = 18606; Connection Settings.Connection Flags = 1056; Connection Settings.Connection Path Size = 8; Connection Path = [16#20,16#04,16#24,16#01,16#2C,16#65,16#2C,16#64]; Input_Param0.ReadOnly = False; Input_Param0.BitSize = 8; Input_Param0.DataSize = 1; Input_Param1.ReadOnly = False; Input_Param1.BitSize = 8; Input_Param1.DataSize = 1; Input_Param2.ReadOnly = False; Input_Param2.BitSize = 8; Input_Param2.DataSize = 1; Input_Param3.ReadOnly = False; Input_Param3.BitSize = 8; Input_Param3.DataSize = 1; Input_Param4.ReadOnly = False; Input_Param4.BitSize = 8; Input_Param4.DataSize = 1; Input_Param5.ReadOnly = False; Input_Param5.BitSize = 8; Input_Param5.DataSize = 1; Input_Param6.ReadOnly = False; Input_Param6.BitSize = 8; Input_Param6.DataSize = 1; Input_Param7.ReadOnly = False; Input_Param7.BitSize = 8; Input_Param7.DataSize = 1; Input_Param8.ReadOnly = False; Input_Param8.BitSize = 8; Input_Param8.DataSize = 1; Input_Param9.ReadOnly = False;
            Input_Param9.BitSize = 8; Input_Param9.DataSize = 1; Input_Param10.ReadOnly = False; Input_Param10.BitSize = 8; Input_Param10.DataSize = 1; Input_Param11.ReadOnly = False; Input_Param11.BitSize = 8; Input_Param11.DataSize = 1; Input_Param12.ReadOnly = False; Input_Param12.BitSize = 8; Input_Param12.DataSize = 1; Input_Param13.ReadOnly = False; Input_Param13.BitSize = 8; Input_Param13.DataSize = 1; Input_Param14.ReadOnly = False; Input_Param14.BitSize = 8; Input_Param14.DataSize = 1; Input_Param15.ReadOnly = False; Input_Param15.BitSize = 8; Input_Param15.DataSize = 1; Input_Param16.ReadOnly = False; Input_Param16.BitSize = 8; Input_Param16.DataSize = 1; Input_Param17.ReadOnly = False; Input_Param17.BitSize = 8; Input_Param17.DataSize = 1; Input_Param18.ReadOnly = False; Input_Param18.BitSize = 8; Input_Param18.DataSize = 1; Input_Param19.ReadOnly = False; Input_Param19.BitSize = 8; Input_Param19.DataSize = 1; Input_Param20.ReadOnly = False; Input_Param20.BitSize = 8; Input_Param20.DataSize = 1; Input_Param21.ReadOnly = False; Input_Param21.BitSize = 8; Input_Param21.DataSize = 1; Input_Param22.ReadOnly = False; Input_Param22.BitSize = 8;
            Input_Param22.DataSize = 1; Input_Param23.ReadOnly = False; Input_Param23.BitSize = 8; Input_Param23.DataSize = 1; Input_Param24.ReadOnly = False; Input_Param24.BitSize = 8; Input_Param24.DataSize = 1; Input_Param25.ReadOnly = False; Input_Param25.BitSize = 8; Input_Param25.DataSize = 1; Input_Param26.ReadOnly = False; Input_Param26.BitSize = 8; Input_Param26.DataSize = 1; Input_Param27.ReadOnly = False; Input_Param27.BitSize = 8; Input_Param27.DataSize = 1; Input_Param28.ReadOnly = False; Input_Param28.BitSize = 8; Input_Param28.DataSize = 1; Input_Param29.ReadOnly = False; Input_Param29.BitSize = 8; Input_Param29.DataSize = 1; Input_Param30.ReadOnly = False; Input_Param30.BitSize = 8; Input_Param30.DataSize = 1; Input_Param31.ReadOnly = False; Input_Param31.BitSize = 8; Input_Param31.DataSize = 1; Input_Param32.ReadOnly = False; Input_Param32.BitSize = 8; Input_Param32.DataSize = 1; Input_Param33.ReadOnly = False; Input_Param33.BitSize = 8; Input_Param33.DataSize = 1; Input_Param34.ReadOnly = False; Input_Param34.BitSize = 8; Input_Param34.DataSize = 1; Input_Param35.ReadOnly = False; Input_Param35.BitSize = 8; Input_Param35.DataSize = 1;
            Input_Param36.ReadOnly = False; Input_Param36.BitSize = 8; Input_Param36.DataSize = 1; Input_Param37.ReadOnly = False; Input_Param37.BitSize = 8; Input_Param37.DataSize = 1; Input_Param38.ReadOnly = False; Input_Param38.BitSize = 8; Input_Param38.DataSize = 1; Input_Param39.ReadOnly = False; Input_Param39.BitSize = 8; Input_Param39.DataSize = 1; Input_Param40.ReadOnly = False; Input_Param40.BitSize = 8; Input_Param40.DataSize = 1; Input_Param41.ReadOnly = False; Input_Param41.BitSize = 8; Input_Param41.DataSize = 1; Input_Param42.ReadOnly = False; Input_Param42.BitSize = 8; Input_Param42.DataSize = 1; Input_Param43.ReadOnly = False; Input_Param43.BitSize = 8; Input_Param43.DataSize = 1; Input_Param44.ReadOnly = False; Input_Param44.BitSize = 8; Input_Param44.DataSize = 1; Input_Param45.ReadOnly = False; Input_Param45.BitSize = 8; Input_Param45.DataSize = 1; Input_Param46.ReadOnly = False; Input_Param46.BitSize = 8; Input_Param46.DataSize = 1; Input_Param47.ReadOnly = False; Input_Param47.BitSize = 8; Input_Param47.DataSize = 1; Input_Param48.ReadOnly = False; Input_Param48.BitSize = 8; Input_Param48.DataSize = 1; Input_Param49.ReadOnly = False;
            Input_Param49.BitSize = 8; Input_Param49.DataSize = 1; Input_Param50.ReadOnly = False; Input_Param50.BitSize = 8; Input_Param50.DataSize = 1; Input_Param51.ReadOnly = False; Input_Param51.BitSize = 8; Input_Param51.DataSize = 1; Input_Param52.ReadOnly = False; Input_Param52.BitSize = 8; Input_Param52.DataSize = 1; Input_Param53.ReadOnly = False; Input_Param53.BitSize = 8; Input_Param53.DataSize = 1; Input_Param54.ReadOnly = False; Input_Param54.BitSize = 8; Input_Param54.DataSize = 1; Input_Param55.ReadOnly = False; Input_Param55.BitSize = 8; Input_Param55.DataSize = 1; Input_Param56.ReadOnly = False; Input_Param56.BitSize = 8; Input_Param56.DataSize = 1; Input_Param57.ReadOnly = False; Input_Param57.BitSize = 8; Input_Param57.DataSize = 1; Input_Param58.ReadOnly = False; Input_Param58.BitSize = 8; Input_Param58.DataSize = 1; Input_Param59.ReadOnly = False; Input_Param59.BitSize = 8; Input_Param59.DataSize = 1; Input_Param60.ReadOnly = False; Input_Param60.BitSize = 8; Input_Param60.DataSize = 1; Input_Param61.ReadOnly = False; Input_Param61.BitSize = 8; Input_Param61.DataSize = 1; Input_Param62.ReadOnly = False; Input_Param62.BitSize = 8;
            Input_Param62.DataSize = 1; Input_Param63.ReadOnly = False; Input_Param63.BitSize = 8; Input_Param63.DataSize = 1; Input_Param64.ReadOnly = False; Input_Param64.BitSize = 8; Input_Param64.DataSize = 1; Input_Param65.ReadOnly = False; Input_Param65.BitSize = 8; Input_Param65.DataSize = 1; Input_Param66.ReadOnly = False; Input_Param66.BitSize = 8; Input_Param66.DataSize = 1; Input_Param67.ReadOnly = False; Input_Param67.BitSize = 8; Input_Param67.DataSize = 1; Input_Param68.ReadOnly = False; Input_Param68.BitSize = 8; Input_Param68.DataSize = 1; Input_Param69.ReadOnly = False; Input_Param69.BitSize = 8; Input_Param69.DataSize = 1; Input_Param70.ReadOnly = False; Input_Param70.BitSize = 8; Input_Param70.DataSize = 1; Input_Param71.ReadOnly = False; Input_Param71.BitSize = 8; Input_Param71.DataSize = 1; Input_Param72.ReadOnly = False; Input_Param72.BitSize = 8; Input_Param72.DataSize = 1; Input_Param73.ReadOnly = False; Input_Param73.BitSize = 8; Input_Param73.DataSize = 1; Input_Param74.ReadOnly = False; Input_Param74.BitSize = 8; Input_Param74.DataSize = 1; Input_Param75.ReadOnly = False; Input_Param75.BitSize = 8; Input_Param75.DataSize = 1;
            Input_Param76.ReadOnly = False; Input_Param76.BitSize = 8; Input_Param76.DataSize = 1; Input_Param77.ReadOnly = False; Input_Param77.BitSize = 8; Input_Param77.DataSize = 1; Input_Param78.ReadOnly = False; Input_Param78.BitSize = 8; Input_Param78.DataSize = 1; Input_Param79.ReadOnly = False; Input_Param79.BitSize = 8; Input_Param79.DataSize = 1; Input_Param80.ReadOnly = False; Input_Param80.BitSize = 8; Input_Param80.DataSize = 1; Input_Param81.ReadOnly = False; Input_Param81.BitSize = 8; Input_Param81.DataSize = 1; Input_Param82.ReadOnly = False; Input_Param82.BitSize = 8; Input_Param82.DataSize = 1; Input_Param83.ReadOnly = False; Input_Param83.BitSize = 8; Input_Param83.DataSize = 1; Input_Param84.ReadOnly = False; Input_Param84.BitSize = 8; Input_Param84.DataSize = 1; Input_Param85.ReadOnly = False; Input_Param85.BitSize = 8; Input_Param85.DataSize = 1; Input_Param86.ReadOnly = False; Input_Param86.BitSize = 8; Input_Param86.DataSize = 1; Input_Param87.ReadOnly = False; Input_Param87.BitSize = 8; Input_Param87.DataSize = 1; Input_Param88.ReadOnly = False; Input_Param88.BitSize = 8; Input_Param88.DataSize = 1; Input_Param89.ReadOnly = False;
            Input_Param89.BitSize = 8; Input_Param89.DataSize = 1; Input_Param90.ReadOnly = False; Input_Param90.BitSize = 8; Input_Param90.DataSize = 1; Input_Param91.ReadOnly = False; Input_Param91.BitSize = 8; Input_Param91.DataSize = 1; Input_Param92.ReadOnly = False; Input_Param92.BitSize = 8; Input_Param92.DataSize = 1; Input_Param93.ReadOnly = False; Input_Param93.BitSize = 8; Input_Param93.DataSize = 1; Input_Param94.ReadOnly = False; Input_Param94.BitSize = 8; Input_Param94.DataSize = 1; Input_Param95.ReadOnly = False; Input_Param95.BitSize = 8; Input_Param95.DataSize = 1; Input_Param96.ReadOnly = False; Input_Param96.BitSize = 8; Input_Param96.DataSize = 1; Input_Param97.ReadOnly = False; Input_Param97.BitSize = 8; Input_Param97.DataSize = 1; Input_Param98.ReadOnly = False; Input_Param98.BitSize = 8; Input_Param98.DataSize = 1; Input_Param99.ReadOnly = False; Input_Param99.BitSize = 8; Input_Param99.DataSize = 1; Input_Param100.ReadOnly = False; Input_Param100.BitSize = 8; Input_Param100.DataSize = 1; Input_Param101.ReadOnly = False; Input_Param101.BitSize = 8; Input_Param101.DataSize = 1; Input_Param102.ReadOnly = False; Input_Param102.BitSize = 8;
            Input_Param102.DataSize = 1; Input_Param103.ReadOnly = False; Input_Param103.BitSize = 8; Input_Param103.DataSize = 1; Input_Param104.ReadOnly = False; Input_Param104.BitSize = 8; Input_Param104.DataSize = 1; Input_Param105.ReadOnly = False; Input_Param105.BitSize = 8; Input_Param105.DataSize = 1; Input_Param106.ReadOnly = False; Input_Param106.BitSize = 8; Input_Param106.DataSize = 1; Input_Param107.ReadOnly = False; Input_Param107.BitSize = 8; Input_Param107.DataSize = 1; Input_Param108.ReadOnly = False; Input_Param108.BitSize = 8; Input_Param108.DataSize = 1; Input_Param109.ReadOnly = False; Input_Param109.BitSize = 8; Input_Param109.DataSize = 1; Input_Param110.ReadOnly = False; Input_Param110.BitSize = 8; Input_Param110.DataSize = 1; Input_Param111.ReadOnly = False; Input_Param111.BitSize = 8; Input_Param111.DataSize = 1; Input_Param112.ReadOnly = False; Input_Param112.BitSize = 8; Input_Param112.DataSize = 1; Input_Param113.ReadOnly = False; Input_Param113.BitSize = 8; Input_Param113.DataSize = 1; Input_Param114.ReadOnly = False; Input_Param114.BitSize = 8; Input_Param114.DataSize = 1; Input_Param115.ReadOnly = False; Input_Param115.BitSize = 8; Input_Param115.DataSize = 1;
            Input_Param116.ReadOnly = False; Input_Param116.BitSize = 8; Input_Param116.DataSize = 1; Input_Param117.ReadOnly = False; Input_Param117.BitSize = 8; Input_Param117.DataSize = 1; Input_Param118.ReadOnly = False; Input_Param118.BitSize = 8; Input_Param118.DataSize = 1; Input_Param119.ReadOnly = False; Input_Param119.BitSize = 8; Input_Param119.DataSize = 1; Input_Param120.ReadOnly = False; Input_Param120.BitSize = 8; Input_Param120.DataSize = 1; Input_Param121.ReadOnly = False; Input_Param121.BitSize = 8; Input_Param121.DataSize = 1; Input_Param122.ReadOnly = False; Input_Param122.BitSize = 8; Input_Param122.DataSize = 1; Input_Param123.ReadOnly = False; Input_Param123.BitSize = 8; Input_Param123.DataSize = 1; Input_Param124.ReadOnly = False; Input_Param124.BitSize = 8; Input_Param124.DataSize = 1; Input_Param125.ReadOnly = False; Input_Param125.BitSize = 8; Input_Param125.DataSize = 1; Input_Param126.ReadOnly = False; Input_Param126.BitSize = 8; Input_Param126.DataSize = 1; Input_Param127.ReadOnly = False; Input_Param127.BitSize = 8; Input_Param127.DataSize = 1; Input_Param128.ReadOnly = False; Input_Param128.BitSize = 8; Input_Param128.DataSize = 1; Input_Param129.ReadOnly = False;
            Input_Param129.BitSize = 8; Input_Param129.DataSize = 1; Input_Param130.ReadOnly = False; Input_Param130.BitSize = 8; Input_Param130.DataSize = 1; Input_Param131.ReadOnly = False; Input_Param131.BitSize = 8; Input_Param131.DataSize = 1; Input_Param132.ReadOnly = False; Input_Param132.BitSize = 8; Input_Param132.DataSize = 1; Input_Param133.ReadOnly = False; Input_Param133.BitSize = 8; Input_Param133.DataSize = 1; Input_Param134.ReadOnly = False; Input_Param134.BitSize = 8; Input_Param134.DataSize = 1; Input_Param135.ReadOnly = False; Input_Param135.BitSize = 8; Input_Param135.DataSize = 1; Input_Param136.ReadOnly = False; Input_Param136.BitSize = 8; Input_Param136.DataSize = 1; Input_Param137.ReadOnly = False; Input_Param137.BitSize = 8; Input_Param137.DataSize = 1; Input_Param138.ReadOnly = False; Input_Param138.BitSize = 8; Input_Param138.DataSize = 1; Input_Param139.ReadOnly = False; Input_Param139.BitSize = 8; Input_Param139.DataSize = 1; Input_Param140.ReadOnly = False; Input_Param140.BitSize = 8; Input_Param140.DataSize = 1; Input_Param141.ReadOnly = False; Input_Param141.BitSize = 8; Input_Param141.DataSize = 1; Input_Param142.ReadOnly = False; Input_Param142.BitSize = 8;
            Input_Param142.DataSize = 1; Input_Param143.ReadOnly = False; Input_Param143.BitSize = 8; Input_Param143.DataSize = 1; Input_Param144.ReadOnly = False; Input_Param144.BitSize = 8; Input_Param144.DataSize = 1; Input_Param145.ReadOnly = False; Input_Param145.BitSize = 8; Input_Param145.DataSize = 1; Input_Param146.ReadOnly = False; Input_Param146.BitSize = 8; Input_Param146.DataSize = 1; Input_Param147.ReadOnly = False; Input_Param147.BitSize = 8; Input_Param147.DataSize = 1; Input_Param148.ReadOnly = False; Input_Param148.BitSize = 8; Input_Param148.DataSize = 1; Input_Param149.ReadOnly = False; Input_Param149.BitSize = 8; Input_Param149.DataSize = 1; Input_Param150.ReadOnly = False; Input_Param150.BitSize = 8; Input_Param150.DataSize = 1; Input_Param151.ReadOnly = False; Input_Param151.BitSize = 8; Input_Param151.DataSize = 1; Input_Param152.ReadOnly = False; Input_Param152.BitSize = 8; Input_Param152.DataSize = 1; Input_Param153.ReadOnly = False; Input_Param153.BitSize = 8; Input_Param153.DataSize = 1; Input_Param154.ReadOnly = False; Input_Param154.BitSize = 8; Input_Param154.DataSize = 1; Input_Param155.ReadOnly = False; Input_Param155.BitSize = 8; Input_Param155.DataSize = 1;
            Input_Param156.ReadOnly = False; Input_Param156.BitSize = 8; Input_Param156.DataSize = 1; Input_Param157.ReadOnly = False; Input_Param157.BitSize = 8; Input_Param157.DataSize = 1; Input_Param158.ReadOnly = False; Input_Param158.BitSize = 8; Input_Param158.DataSize = 1; Input_Param159.ReadOnly = False; Input_Param159.BitSize = 8; Input_Param159.DataSize = 1; Input_Param160.ReadOnly = False; Input_Param160.BitSize = 8; Input_Param160.DataSize = 1; Input_Param161.ReadOnly = False; Input_Param161.BitSize = 8; Input_Param161.DataSize = 1; Input_Param162.ReadOnly = False; Input_Param162.BitSize = 8; Input_Param162.DataSize = 1; Input_Param163.ReadOnly = False; Input_Param163.BitSize = 8; Input_Param163.DataSize = 1; Input_Param164.ReadOnly = False; Input_Param164.BitSize = 8; Input_Param164.DataSize = 1; Input_Param165.ReadOnly = False; Input_Param165.BitSize = 8; Input_Param165.DataSize = 1; Input_Param166.ReadOnly = False; Input_Param166.BitSize = 8; Input_Param166.DataSize = 1; Input_Param167.ReadOnly = False; Input_Param167.BitSize = 8; Input_Param167.DataSize = 1; Input_Param168.ReadOnly = False; Input_Param168.BitSize = 8; Input_Param168.DataSize = 1; Input_Param169.ReadOnly = False;
            Input_Param169.BitSize = 8; Input_Param169.DataSize = 1; Input_Param170.ReadOnly = False; Input_Param170.BitSize = 8; Input_Param170.DataSize = 1; Input_Param171.ReadOnly = False; Input_Param171.BitSize = 8; Input_Param171.DataSize = 1; Output_Param0.ReadOnly = False; Output_Param0.BitSize = 8; Output_Param0.DataSize = 1; Output_Param1.ReadOnly = False; Output_Param1.BitSize = 8; Output_Param1.DataSize = 1; Output_Param2.ReadOnly = False; Output_Param2.BitSize = 8; Output_Param2.DataSize = 1; Output_Param3.ReadOnly = False; Output_Param3.BitSize = 8; Output_Param3.DataSize = 1; Output_Param4.ReadOnly = False; Output_Param4.BitSize = 8; Output_Param4.DataSize = 1; Output_Param5.ReadOnly = False; Output_Param5.BitSize = 8; Output_Param5.DataSize = 1; Output_Param6.ReadOnly = False; Output_Param6.BitSize = 8; Output_Param6.DataSize = 1; Output_Param7.ReadOnly = False; Output_Param7.BitSize = 8; Output_Param7.DataSize = 1; Output_Param8.ReadOnly = False; Output_Param8.BitSize = 8; Output_Param8.DataSize = 1; Output_Param9.ReadOnly = False; Output_Param9.BitSize = 8; Output_Param9.DataSize = 1; Output_Param10.ReadOnly = False; Output_Param10.BitSize = 8;
            Output_Param10.DataSize = 1; Output_Param11.ReadOnly = False; Output_Param11.BitSize = 8; Output_Param11.DataSize = 1; Output_Param12.ReadOnly = False; Output_Param12.BitSize = 8; Output_Param12.DataSize = 1; Output_Param13.ReadOnly = False; Output_Param13.BitSize = 8; Output_Param13.DataSize = 1; Output_Param14.ReadOnly = False; Output_Param14.BitSize = 8; Output_Param14.DataSize = 1; Output_Param15.ReadOnly = False; Output_Param15.BitSize = 8; Output_Param15.DataSize = 1; Output_Param16.ReadOnly = False; Output_Param16.BitSize = 8; Output_Param16.DataSize = 1; Output_Param17.ReadOnly = False; Output_Param17.BitSize = 8; Output_Param17.DataSize = 1; Output_Param18.ReadOnly = False; Output_Param18.BitSize = 8; Output_Param18.DataSize = 1; Output_Param19.ReadOnly = False; Output_Param19.BitSize = 8; Output_Param19.DataSize = 1; Output_Param20.ReadOnly = False; Output_Param20.BitSize = 8; Output_Param20.DataSize = 1; Output_Param21.ReadOnly = False; Output_Param21.BitSize = 8; Output_Param21.DataSize = 1; Output_Param22.ReadOnly = False; Output_Param22.BitSize = 8; Output_Param22.DataSize = 1; Output_Param23.ReadOnly = False; Output_Param23.BitSize = 8; Output_Param23.DataSize = 1;
            Output_Param24.ReadOnly = False; Output_Param24.BitSize = 8; Output_Param24.DataSize = 1; Output_Param25.ReadOnly = False; Output_Param25.BitSize = 8; Output_Param25.DataSize = 1; Output_Param26.ReadOnly = False; Output_Param26.BitSize = 8; Output_Param26.DataSize = 1; Output_Param27.ReadOnly = False; Output_Param27.BitSize = 8; Output_Param27.DataSize = 1; Output_Param28.ReadOnly = False; Output_Param28.BitSize = 8; Output_Param28.DataSize = 1; Output_Param29.ReadOnly = False; Output_Param29.BitSize = 8; Output_Param29.DataSize = 1; Output_Param30.ReadOnly = False; Output_Param30.BitSize = 8; Output_Param30.DataSize = 1; Output_Param31.ReadOnly = False; Output_Param31.BitSize = 8; Output_Param31.DataSize = 1; Output_Param32.ReadOnly = False; Output_Param32.BitSize = 8; Output_Param32.DataSize = 1; Output_Param33.ReadOnly = False; Output_Param33.BitSize = 8; Output_Param33.DataSize = 1; Output_Param34.ReadOnly = False; Output_Param34.BitSize = 8; Output_Param34.DataSize = 1; Output_Param35.ReadOnly = False; Output_Param35.BitSize = 8; Output_Param35.DataSize = 1; Output_Param36.ReadOnly = False; Output_Param36.BitSize = 8; Output_Param36.DataSize = 1; Output_Param37.ReadOnly = False;
            Output_Param37.BitSize = 8; Output_Param37.DataSize = 1; Output_Param38.ReadOnly = False; Output_Param38.BitSize = 8; Output_Param38.DataSize = 1; Output_Param39.ReadOnly = False; Output_Param39.BitSize = 8; Output_Param39.DataSize = 1; Output_Param40.ReadOnly = False; Output_Param40.BitSize = 8; Output_Param40.DataSize = 1; Output_Param41.ReadOnly = False; Output_Param41.BitSize = 8; Output_Param41.DataSize = 1; Output_Param42.ReadOnly = False; Output_Param42.BitSize = 8; Output_Param42.DataSize = 1; Output_Param43.ReadOnly = False; Output_Param43.BitSize = 8; Output_Param43.DataSize = 1; Output_Param44.ReadOnly = False; Output_Param44.BitSize = 8; Output_Param44.DataSize = 1; Output_Param45.ReadOnly = False; Output_Param45.BitSize = 8; Output_Param45.DataSize = 1; Output_Param46.ReadOnly = False; Output_Param46.BitSize = 8; Output_Param46.DataSize = 1; Output_Param47.ReadOnly = False; Output_Param47.BitSize = 8; Output_Param47.DataSize = 1; Output_Param48.ReadOnly = False; Output_Param48.BitSize = 8; Output_Param48.DataSize = 1; Output_Param49.ReadOnly = False; Output_Param49.BitSize = 8; Output_Param49.DataSize = 1; Output_Param50.ReadOnly = False; Output_Param50.BitSize = 8;
            Output_Param50.DataSize = 1; Output_Param51.ReadOnly = False; Output_Param51.BitSize = 8; Output_Param51.DataSize = 1; Output_Param52.ReadOnly = False; Output_Param52.BitSize = 8; Output_Param52.DataSize = 1; Output_Param53.ReadOnly = False; Output_Param53.BitSize = 8; Output_Param53.DataSize = 1; Output_Param54.ReadOnly = False; Output_Param54.BitSize = 8; Output_Param54.DataSize = 1; Output_Param55.ReadOnly = False; Output_Param55.BitSize = 8; Output_Param55.DataSize = 1; Output_Param56.ReadOnly = False; Output_Param56.BitSize = 8; Output_Param56.DataSize = 1; Output_Param57.ReadOnly = False; Output_Param57.BitSize = 8; Output_Param57.DataSize = 1; Output_Param58.ReadOnly = False; Output_Param58.BitSize = 8; Output_Param58.DataSize = 1; Output_Param59.ReadOnly = False; Output_Param59.BitSize = 8; Output_Param59.DataSize = 1; Output_Param60.ReadOnly = False; Output_Param60.BitSize = 8; Output_Param60.DataSize = 1; Output_Param61.ReadOnly = False; Output_Param61.BitSize = 8; Output_Param61.DataSize = 1; Output_Param62.ReadOnly = False; Output_Param62.BitSize = 8; Output_Param62.DataSize = 1; Output_Param63.ReadOnly = False; Output_Param63.BitSize = 8; Output_Param63.DataSize = 1;
            Output_Param64.ReadOnly = False; Output_Param64.BitSize = 8; Output_Param64.DataSize = 1; Output_Param65.ReadOnly = False; Output_Param65.BitSize = 8; Output_Param65.DataSize = 1; Output_Param66.ReadOnly = False; Output_Param66.BitSize = 8; Output_Param66.DataSize = 1; Output_Param67.ReadOnly = False; Output_Param67.BitSize = 8; Output_Param67.DataSize = 1; Output_Param68.ReadOnly = False; Output_Param68.BitSize = 8; Output_Param68.DataSize = 1; Output_Param69.ReadOnly = False; Output_Param69.BitSize = 8; Output_Param69.DataSize = 1; Output_Param70.ReadOnly = False; Output_Param70.BitSize = 8; Output_Param70.DataSize = 1; Output_Param71.ReadOnly = False; Output_Param71.BitSize = 8; Output_Param71.DataSize = 1; Output_Param72.ReadOnly = False; Output_Param72.BitSize = 8; Output_Param72.DataSize = 1; Output_Param73.ReadOnly = False; Output_Param73.BitSize = 8; Output_Param73.DataSize = 1; Output_Param74.ReadOnly = False; Output_Param74.BitSize = 8; Output_Param74.DataSize = 1; Output_Param75.ReadOnly = False; Output_Param75.BitSize = 8; Output_Param75.DataSize = 1; Input_Param0.Name = 'Input_Param0'; Input_Param0.HelpString = ''; Input_Param0.ReadOnly = False; Input_Param0.BitSize = 8;
            Input_Param0.DataSize = 1; Input_Param0.DataType = 'BYTE'; Input_Param1.Name = 'Input_Param1'; Input_Param1.HelpString = ''; Input_Param1.ReadOnly = False; Input_Param1.BitSize = 8; Input_Param1.DataSize = 1; Input_Param1.DataType = 'BYTE'; Input_Param2.Name = 'Input_Param2'; Input_Param2.HelpString = ''; Input_Param2.ReadOnly = False; Input_Param2.BitSize = 8; Input_Param2.DataSize = 1; Input_Param2.DataType = 'BYTE'; Input_Param3.Name = 'Input_Param3'; Input_Param3.HelpString = ''; Input_Param3.ReadOnly = False; Input_Param3.BitSize = 8; Input_Param3.DataSize = 1; Input_Param3.DataType = 'BYTE'; Input_Param4.Name = 'Input_Param4'; Input_Param4.HelpString = ''; Input_Param4.ReadOnly = False; Input_Param4.BitSize = 8; Input_Param4.DataSize = 1; Input_Param4.DataType = 'BYTE'; Input_Param5.Name = 'Input_Param5'; Input_Param5.HelpString = ''; Input_Param5.ReadOnly = False; Input_Param5.BitSize = 8; Input_Param5.DataSize = 1; Input_Param5.DataType = 'BYTE'; Input_Param6.Name = 'Input_Param6'; Input_Param6.HelpString = ''; Input_Param6.ReadOnly = False; Input_Param6.BitSize = 8; Input_Param6.DataSize = 1; Input_Param6.DataType = 'BYTE'; Input_Param7.Name = 'Input_Param7'; Input_Param7.HelpString = '';
            Input_Param7.ReadOnly = False; Input_Param7.BitSize = 8; Input_Param7.DataSize = 1; Input_Param7.DataType = 'BYTE'; Input_Param8.Name = 'Input_Param8'; Input_Param8.HelpString = ''; Input_Param8.ReadOnly = False; Input_Param8.BitSize = 8; Input_Param8.DataSize = 1; Input_Param8.DataType = 'BYTE'; Input_Param9.Name = 'Input_Param9'; Input_Param9.HelpString = ''; Input_Param9.ReadOnly = False; Input_Param9.BitSize = 8; Input_Param9.DataSize = 1; Input_Param9.DataType = 'BYTE'; Input_Param10.Name = 'Input_Param10'; Input_Param10.HelpString = ''; Input_Param10.ReadOnly = False; Input_Param10.BitSize = 8; Input_Param10.DataSize = 1; Input_Param10.DataType = 'BYTE'; Input_Param11.Name = 'Input_Param11'; Input_Param11.HelpString = ''; Input_Param11.ReadOnly = False; Input_Param11.BitSize = 8; Input_Param11.DataSize = 1; Input_Param11.DataType = 'BYTE'; Input_Param12.Name = 'Input_Param12'; Input_Param12.HelpString = ''; Input_Param12.ReadOnly = False; Input_Param12.BitSize = 8; Input_Param12.DataSize = 1; Input_Param12.DataType = 'BYTE'; Input_Param13.Name = 'Input_Param13'; Input_Param13.HelpString = ''; Input_Param13.ReadOnly = False; Input_Param13.BitSize = 8; Input_Param13.DataSize = 1; Input_Param13.DataType = 'BYTE';
            Input_Param14.Name = 'Input_Param14'; Input_Param14.HelpString = ''; Input_Param14.ReadOnly = False; Input_Param14.BitSize = 8; Input_Param14.DataSize = 1; Input_Param14.DataType = 'BYTE'; Input_Param15.Name = 'Input_Param15'; Input_Param15.HelpString = ''; Input_Param15.ReadOnly = False; Input_Param15.BitSize = 8; Input_Param15.DataSize = 1; Input_Param15.DataType = 'BYTE'; Input_Param16.Name = 'Input_Param16'; Input_Param16.HelpString = ''; Input_Param16.ReadOnly = False; Input_Param16.BitSize = 8; Input_Param16.DataSize = 1; Input_Param16.DataType = 'BYTE'; Input_Param17.Name = 'Input_Param17'; Input_Param17.HelpString = ''; Input_Param17.ReadOnly = False; Input_Param17.BitSize = 8; Input_Param17.DataSize = 1; Input_Param17.DataType = 'BYTE'; Input_Param18.Name = 'Input_Param18'; Input_Param18.HelpString = ''; Input_Param18.ReadOnly = False; Input_Param18.BitSize = 8; Input_Param18.DataSize = 1; Input_Param18.DataType = 'BYTE'; Input_Param19.Name = 'Input_Param19'; Input_Param19.HelpString = ''; Input_Param19.ReadOnly = False; Input_Param19.BitSize = 8; Input_Param19.DataSize = 1; Input_Param19.DataType = 'BYTE'; Input_Param20.Name = 'Input_Param20'; Input_Param20.HelpString = ''; Input_Param20.ReadOnly = False; Input_Param20.BitSize = 8;
            Input_Param20.DataSize = 1; Input_Param20.DataType = 'BYTE'; Input_Param21.Name = 'Input_Param21'; Input_Param21.HelpString = ''; Input_Param21.ReadOnly = False; Input_Param21.BitSize = 8; Input_Param21.DataSize = 1; Input_Param21.DataType = 'BYTE'; Input_Param22.Name = 'Input_Param22'; Input_Param22.HelpString = ''; Input_Param22.ReadOnly = False; Input_Param22.BitSize = 8; Input_Param22.DataSize = 1; Input_Param22.DataType = 'BYTE'; Input_Param23.Name = 'Input_Param23'; Input_Param23.HelpString = ''; Input_Param23.ReadOnly = False; Input_Param23.BitSize = 8; Input_Param23.DataSize = 1; Input_Param23.DataType = 'BYTE'; Input_Param24.Name = 'Input_Param24'; Input_Param24.HelpString = ''; Input_Param24.ReadOnly = False; Input_Param24.BitSize = 8; Input_Param24.DataSize = 1; Input_Param24.DataType = 'BYTE'; Input_Param25.Name = 'Input_Param25'; Input_Param25.HelpString = ''; Input_Param25.ReadOnly = False; Input_Param25.BitSize = 8; Input_Param25.DataSize = 1; Input_Param25.DataType = 'BYTE'; Input_Param26.Name = 'Input_Param26'; Input_Param26.HelpString = ''; Input_Param26.ReadOnly = False; Input_Param26.BitSize = 8; Input_Param26.DataSize = 1; Input_Param26.DataType = 'BYTE'; Input_Param27.Name = 'Input_Param27'; Input_Param27.HelpString = '';
            Input_Param27.ReadOnly = False; Input_Param27.BitSize = 8; Input_Param27.DataSize = 1; Input_Param27.DataType = 'BYTE'; Input_Param28.Name = 'Input_Param28'; Input_Param28.HelpString = ''; Input_Param28.ReadOnly = False; Input_Param28.BitSize = 8; Input_Param28.DataSize = 1; Input_Param28.DataType = 'BYTE'; Input_Param29.Name = 'Input_Param29'; Input_Param29.HelpString = ''; Input_Param29.ReadOnly = False; Input_Param29.BitSize = 8; Input_Param29.DataSize = 1; Input_Param29.DataType = 'BYTE'; Input_Param30.Name = 'Input_Param30'; Input_Param30.HelpString = ''; Input_Param30.ReadOnly = False; Input_Param30.BitSize = 8; Input_Param30.DataSize = 1; Input_Param30.DataType = 'BYTE'; Input_Param31.Name = 'Input_Param31'; Input_Param31.HelpString = ''; Input_Param31.ReadOnly = False; Input_Param31.BitSize = 8; Input_Param31.DataSize = 1; Input_Param31.DataType = 'BYTE'; Input_Param32.Name = 'Input_Param32'; Input_Param32.HelpString = ''; Input_Param32.ReadOnly = False; Input_Param32.BitSize = 8; Input_Param32.DataSize = 1; Input_Param32.DataType = 'BYTE'; Input_Param33.Name = 'Input_Param33'; Input_Param33.HelpString = ''; Input_Param33.ReadOnly = False; Input_Param33.BitSize = 8; Input_Param33.DataSize = 1; Input_Param33.DataType = 'BYTE';
            Input_Param34.Name = 'Input_Param34'; Input_Param34.HelpString = ''; Input_Param34.ReadOnly = False; Input_Param34.BitSize = 8; Input_Param34.DataSize = 1; Input_Param34.DataType = 'BYTE'; Input_Param35.Name = 'Input_Param35'; Input_Param35.HelpString = ''; Input_Param35.ReadOnly = False; Input_Param35.BitSize = 8; Input_Param35.DataSize = 1; Input_Param35.DataType = 'BYTE'; Input_Param36.Name = 'Input_Param36'; Input_Param36.HelpString = ''; Input_Param36.ReadOnly = False; Input_Param36.BitSize = 8; Input_Param36.DataSize = 1; Input_Param36.DataType = 'BYTE'; Input_Param37.Name = 'Input_Param37'; Input_Param37.HelpString = ''; Input_Param37.ReadOnly = False; Input_Param37.BitSize = 8; Input_Param37.DataSize = 1; Input_Param37.DataType = 'BYTE'; Input_Param38.Name = 'Input_Param38'; Input_Param38.HelpString = ''; Input_Param38.ReadOnly = False; Input_Param38.BitSize = 8; Input_Param38.DataSize = 1; Input_Param38.DataType = 'BYTE'; Input_Param39.Name = 'Input_Param39'; Input_Param39.HelpString = ''; Input_Param39.ReadOnly = False; Input_Param39.BitSize = 8; Input_Param39.DataSize = 1; Input_Param39.DataType = 'BYTE'; Input_Param40.Name = 'Input_Param40'; Input_Param40.HelpString = ''; Input_Param40.ReadOnly = False; Input_Param40.BitSize = 8;
            Input_Param40.DataSize = 1; Input_Param40.DataType = 'BYTE'; Input_Param41.Name = 'Input_Param41'; Input_Param41.HelpString = ''; Input_Param41.ReadOnly = False; Input_Param41.BitSize = 8; Input_Param41.DataSize = 1; Input_Param41.DataType = 'BYTE'; Input_Param42.Name = 'Input_Param42'; Input_Param42.HelpString = ''; Input_Param42.ReadOnly = False; Input_Param42.BitSize = 8; Input_Param42.DataSize = 1; Input_Param42.DataType = 'BYTE'; Input_Param43.Name = 'Input_Param43'; Input_Param43.HelpString = ''; Input_Param43.ReadOnly = False; Input_Param43.BitSize = 8; Input_Param43.DataSize = 1; Input_Param43.DataType = 'BYTE'; Input_Param44.Name = 'Input_Param44'; Input_Param44.HelpString = ''; Input_Param44.ReadOnly = False; Input_Param44.BitSize = 8; Input_Param44.DataSize = 1; Input_Param44.DataType = 'BYTE'; Input_Param45.Name = 'Input_Param45'; Input_Param45.HelpString = ''; Input_Param45.ReadOnly = False; Input_Param45.BitSize = 8; Input_Param45.DataSize = 1; Input_Param45.DataType = 'BYTE'; Input_Param46.Name = 'Input_Param46'; Input_Param46.HelpString = ''; Input_Param46.ReadOnly = False; Input_Param46.BitSize = 8; Input_Param46.DataSize = 1; Input_Param46.DataType = 'BYTE'; Input_Param47.Name = 'Input_Param47'; Input_Param47.HelpString = '';
            Input_Param47.ReadOnly = False; Input_Param47.BitSize = 8; Input_Param47.DataSize = 1; Input_Param47.DataType = 'BYTE'; Input_Param48.Name = 'Input_Param48'; Input_Param48.HelpString = ''; Input_Param48.ReadOnly = False; Input_Param48.BitSize = 8; Input_Param48.DataSize = 1; Input_Param48.DataType = 'BYTE'; Input_Param49.Name = 'Input_Param49'; Input_Param49.HelpString = ''; Input_Param49.ReadOnly = False; Input_Param49.BitSize = 8; Input_Param49.DataSize = 1; Input_Param49.DataType = 'BYTE'; Input_Param50.Name = 'Input_Param50'; Input_Param50.HelpString = ''; Input_Param50.ReadOnly = False; Input_Param50.BitSize = 8; Input_Param50.DataSize = 1; Input_Param50.DataType = 'BYTE'; Input_Param51.Name = 'Input_Param51'; Input_Param51.HelpString = ''; Input_Param51.ReadOnly = False; Input_Param51.BitSize = 8; Input_Param51.DataSize = 1; Input_Param51.DataType = 'BYTE'; Input_Param52.Name = 'Input_Param52'; Input_Param52.HelpString = ''; Input_Param52.ReadOnly = False; Input_Param52.BitSize = 8; Input_Param52.DataSize = 1; Input_Param52.DataType = 'BYTE'; Input_Param53.Name = 'Input_Param53'; Input_Param53.HelpString = ''; Input_Param53.ReadOnly = False; Input_Param53.BitSize = 8; Input_Param53.DataSize = 1; Input_Param53.DataType = 'BYTE';
            Input_Param54.Name = 'Input_Param54'; Input_Param54.HelpString = ''; Input_Param54.ReadOnly = False; Input_Param54.BitSize = 8; Input_Param54.DataSize = 1; Input_Param54.DataType = 'BYTE'; Input_Param55.Name = 'Input_Param55'; Input_Param55.HelpString = ''; Input_Param55.ReadOnly = False; Input_Param55.BitSize = 8; Input_Param55.DataSize = 1; Input_Param55.DataType = 'BYTE'; Input_Param56.Name = 'Input_Param56'; Input_Param56.HelpString = ''; Input_Param56.ReadOnly = False; Input_Param56.BitSize = 8; Input_Param56.DataSize = 1; Input_Param56.DataType = 'BYTE'; Input_Param57.Name = 'Input_Param57'; Input_Param57.HelpString = ''; Input_Param57.ReadOnly = False; Input_Param57.BitSize = 8; Input_Param57.DataSize = 1; Input_Param57.DataType = 'BYTE'; Input_Param58.Name = 'Input_Param58'; Input_Param58.HelpString = ''; Input_Param58.ReadOnly = False; Input_Param58.BitSize = 8; Input_Param58.DataSize = 1; Input_Param58.DataType = 'BYTE'; Input_Param59.Name = 'Input_Param59'; Input_Param59.HelpString = ''; Input_Param59.ReadOnly = False; Input_Param59.BitSize = 8; Input_Param59.DataSize = 1; Input_Param59.DataType = 'BYTE'; Input_Param60.Name = 'Input_Param60'; Input_Param60.HelpString = ''; Input_Param60.ReadOnly = False; Input_Param60.BitSize = 8;
            Input_Param60.DataSize = 1; Input_Param60.DataType = 'BYTE'; Input_Param61.Name = 'Input_Param61'; Input_Param61.HelpString = ''; Input_Param61.ReadOnly = False; Input_Param61.BitSize = 8; Input_Param61.DataSize = 1; Input_Param61.DataType = 'BYTE'; Input_Param62.Name = 'Input_Param62'; Input_Param62.HelpString = ''; Input_Param62.ReadOnly = False; Input_Param62.BitSize = 8; Input_Param62.DataSize = 1; Input_Param62.DataType = 'BYTE'; Input_Param63.Name = 'Input_Param63'; Input_Param63.HelpString = ''; Input_Param63.ReadOnly = False; Input_Param63.BitSize = 8; Input_Param63.DataSize = 1; Input_Param63.DataType = 'BYTE'; Input_Param64.Name = 'Input_Param64'; Input_Param64.HelpString = ''; Input_Param64.ReadOnly = False; Input_Param64.BitSize = 8; Input_Param64.DataSize = 1; Input_Param64.DataType = 'BYTE'; Input_Param65.Name = 'Input_Param65'; Input_Param65.HelpString = ''; Input_Param65.ReadOnly = False; Input_Param65.BitSize = 8; Input_Param65.DataSize = 1; Input_Param65.DataType = 'BYTE'; Input_Param66.Name = 'Input_Param66'; Input_Param66.HelpString = ''; Input_Param66.ReadOnly = False; Input_Param66.BitSize = 8; Input_Param66.DataSize = 1; Input_Param66.DataType = 'BYTE'; Input_Param67.Name = 'Input_Param67'; Input_Param67.HelpString = '';
            Input_Param67.ReadOnly = False; Input_Param67.BitSize = 8; Input_Param67.DataSize = 1; Input_Param67.DataType = 'BYTE'; Input_Param68.Name = 'Input_Param68'; Input_Param68.HelpString = ''; Input_Param68.ReadOnly = False; Input_Param68.BitSize = 8; Input_Param68.DataSize = 1; Input_Param68.DataType = 'BYTE'; Input_Param69.Name = 'Input_Param69'; Input_Param69.HelpString = ''; Input_Param69.ReadOnly = False; Input_Param69.BitSize = 8; Input_Param69.DataSize = 1; Input_Param69.DataType = 'BYTE'; Input_Param70.Name = 'Input_Param70'; Input_Param70.HelpString = ''; Input_Param70.ReadOnly = False; Input_Param70.BitSize = 8; Input_Param70.DataSize = 1; Input_Param70.DataType = 'BYTE'; Input_Param71.Name = 'Input_Param71'; Input_Param71.HelpString = ''; Input_Param71.ReadOnly = False; Input_Param71.BitSize = 8; Input_Param71.DataSize = 1; Input_Param71.DataType = 'BYTE'; Input_Param72.Name = 'Input_Param72'; Input_Param72.HelpString = ''; Input_Param72.ReadOnly = False; Input_Param72.BitSize = 8; Input_Param72.DataSize = 1; Input_Param72.DataType = 'BYTE'; Input_Param73.Name = 'Input_Param73'; Input_Param73.HelpString = ''; Input_Param73.ReadOnly = False; Input_Param73.BitSize = 8; Input_Param73.DataSize = 1; Input_Param73.DataType = 'BYTE';
            Input_Param74.Name = 'Input_Param74'; Input_Param74.HelpString = ''; Input_Param74.ReadOnly = False; Input_Param74.BitSize = 8; Input_Param74.DataSize = 1; Input_Param74.DataType = 'BYTE'; Input_Param75.Name = 'Input_Param75'; Input_Param75.HelpString = ''; Input_Param75.ReadOnly = False; Input_Param75.BitSize = 8; Input_Param75.DataSize = 1; Input_Param75.DataType = 'BYTE'; Input_Param76.Name = 'Input_Param76'; Input_Param76.HelpString = ''; Input_Param76.ReadOnly = False; Input_Param76.BitSize = 8; Input_Param76.DataSize = 1; Input_Param76.DataType = 'BYTE'; Input_Param77.Name = 'Input_Param77'; Input_Param77.HelpString = ''; Input_Param77.ReadOnly = False; Input_Param77.BitSize = 8; Input_Param77.DataSize = 1; Input_Param77.DataType = 'BYTE'; Input_Param78.Name = 'Input_Param78'; Input_Param78.HelpString = ''; Input_Param78.ReadOnly = False; Input_Param78.BitSize = 8; Input_Param78.DataSize = 1; Input_Param78.DataType = 'BYTE'; Input_Param79.Name = 'Input_Param79'; Input_Param79.HelpString = ''; Input_Param79.ReadOnly = False; Input_Param79.BitSize = 8; Input_Param79.DataSize = 1; Input_Param79.DataType = 'BYTE'; Input_Param80.Name = 'Input_Param80'; Input_Param80.HelpString = ''; Input_Param80.ReadOnly = False; Input_Param80.BitSize = 8;
            Input_Param80.DataSize = 1; Input_Param80.DataType = 'BYTE'; Input_Param81.Name = 'Input_Param81'; Input_Param81.HelpString = ''; Input_Param81.ReadOnly = False; Input_Param81.BitSize = 8; Input_Param81.DataSize = 1; Input_Param81.DataType = 'BYTE'; Input_Param82.Name = 'Input_Param82'; Input_Param82.HelpString = ''; Input_Param82.ReadOnly = False; Input_Param82.BitSize = 8; Input_Param82.DataSize = 1; Input_Param82.DataType = 'BYTE'; Input_Param83.Name = 'Input_Param83'; Input_Param83.HelpString = ''; Input_Param83.ReadOnly = False; Input_Param83.BitSize = 8; Input_Param83.DataSize = 1; Input_Param83.DataType = 'BYTE'; Input_Param84.Name = 'Input_Param84'; Input_Param84.HelpString = ''; Input_Param84.ReadOnly = False; Input_Param84.BitSize = 8; Input_Param84.DataSize = 1; Input_Param84.DataType = 'BYTE'; Input_Param85.Name = 'Input_Param85'; Input_Param85.HelpString = ''; Input_Param85.ReadOnly = False; Input_Param85.BitSize = 8; Input_Param85.DataSize = 1; Input_Param85.DataType = 'BYTE'; Input_Param86.Name = 'Input_Param86'; Input_Param86.HelpString = ''; Input_Param86.ReadOnly = False; Input_Param86.BitSize = 8; Input_Param86.DataSize = 1; Input_Param86.DataType = 'BYTE'; Input_Param87.Name = 'Input_Param87'; Input_Param87.HelpString = '';
            Input_Param87.ReadOnly = False; Input_Param87.BitSize = 8; Input_Param87.DataSize = 1; Input_Param87.DataType = 'BYTE'; Input_Param88.Name = 'Input_Param88'; Input_Param88.HelpString = ''; Input_Param88.ReadOnly = False; Input_Param88.BitSize = 8; Input_Param88.DataSize = 1; Input_Param88.DataType = 'BYTE'; Input_Param89.Name = 'Input_Param89'; Input_Param89.HelpString = ''; Input_Param89.ReadOnly = False; Input_Param89.BitSize = 8; Input_Param89.DataSize = 1; Input_Param89.DataType = 'BYTE'; Input_Param90.Name = 'Input_Param90'; Input_Param90.HelpString = ''; Input_Param90.ReadOnly = False; Input_Param90.BitSize = 8; Input_Param90.DataSize = 1; Input_Param90.DataType = 'BYTE'; Input_Param91.Name = 'Input_Param91'; Input_Param91.HelpString = ''; Input_Param91.ReadOnly = False; Input_Param91.BitSize = 8; Input_Param91.DataSize = 1; Input_Param91.DataType = 'BYTE'; Input_Param92.Name = 'Input_Param92'; Input_Param92.HelpString = ''; Input_Param92.ReadOnly = False; Input_Param92.BitSize = 8; Input_Param92.DataSize = 1; Input_Param92.DataType = 'BYTE'; Input_Param93.Name = 'Input_Param93'; Input_Param93.HelpString = ''; Input_Param93.ReadOnly = False; Input_Param93.BitSize = 8; Input_Param93.DataSize = 1; Input_Param93.DataType = 'BYTE';
            Input_Param94.Name = 'Input_Param94'; Input_Param94.HelpString = ''; Input_Param94.ReadOnly = False; Input_Param94.BitSize = 8; Input_Param94.DataSize = 1; Input_Param94.DataType = 'BYTE'; Input_Param95.Name = 'Input_Param95'; Input_Param95.HelpString = ''; Input_Param95.ReadOnly = False; Input_Param95.BitSize = 8; Input_Param95.DataSize = 1; Input_Param95.DataType = 'BYTE'; Input_Param96.Name = 'Input_Param96'; Input_Param96.HelpString = ''; Input_Param96.ReadOnly = False; Input_Param96.BitSize = 8; Input_Param96.DataSize = 1; Input_Param96.DataType = 'BYTE'; Input_Param97.Name = 'Input_Param97'; Input_Param97.HelpString = ''; Input_Param97.ReadOnly = False; Input_Param97.BitSize = 8; Input_Param97.DataSize = 1; Input_Param97.DataType = 'BYTE'; Input_Param98.Name = 'Input_Param98'; Input_Param98.HelpString = ''; Input_Param98.ReadOnly = False; Input_Param98.BitSize = 8; Input_Param98.DataSize = 1; Input_Param98.DataType = 'BYTE'; Input_Param99.Name = 'Input_Param99'; Input_Param99.HelpString = ''; Input_Param99.ReadOnly = False; Input_Param99.BitSize = 8; Input_Param99.DataSize = 1; Input_Param99.DataType = 'BYTE'; Input_Param100.Name = 'Input_Param100'; Input_Param100.HelpString = ''; Input_Param100.ReadOnly = False; Input_Param100.BitSize = 8;
            Input_Param100.DataSize = 1; Input_Param100.DataType = 'BYTE'; Input_Param101.Name = 'Input_Param101'; Input_Param101.HelpString = ''; Input_Param101.ReadOnly = False; Input_Param101.BitSize = 8; Input_Param101.DataSize = 1; Input_Param101.DataType = 'BYTE'; Input_Param102.Name = 'Input_Param102'; Input_Param102.HelpString = ''; Input_Param102.ReadOnly = False; Input_Param102.BitSize = 8; Input_Param102.DataSize = 1; Input_Param102.DataType = 'BYTE'; Input_Param103.Name = 'Input_Param103'; Input_Param103.HelpString = ''; Input_Param103.ReadOnly = False; Input_Param103.BitSize = 8; Input_Param103.DataSize = 1; Input_Param103.DataType = 'BYTE'; Input_Param104.Name = 'Input_Param104'; Input_Param104.HelpString = ''; Input_Param104.ReadOnly = False; Input_Param104.BitSize = 8; Input_Param104.DataSize = 1; Input_Param104.DataType = 'BYTE'; Input_Param105.Name = 'Input_Param105'; Input_Param105.HelpString = ''; Input_Param105.ReadOnly = False; Input_Param105.BitSize = 8; Input_Param105.DataSize = 1; Input_Param105.DataType = 'BYTE'; Input_Param106.Name = 'Input_Param106'; Input_Param106.HelpString = ''; Input_Param106.ReadOnly = False; Input_Param106.BitSize = 8; Input_Param106.DataSize = 1; Input_Param106.DataType = 'BYTE'; Input_Param107.Name = 'Input_Param107'; Input_Param107.HelpString = '';
            Input_Param107.ReadOnly = False; Input_Param107.BitSize = 8; Input_Param107.DataSize = 1; Input_Param107.DataType = 'BYTE'; Input_Param108.Name = 'Input_Param108'; Input_Param108.HelpString = ''; Input_Param108.ReadOnly = False; Input_Param108.BitSize = 8; Input_Param108.DataSize = 1; Input_Param108.DataType = 'BYTE'; Input_Param109.Name = 'Input_Param109'; Input_Param109.HelpString = ''; Input_Param109.ReadOnly = False; Input_Param109.BitSize = 8; Input_Param109.DataSize = 1; Input_Param109.DataType = 'BYTE'; Input_Param110.Name = 'Input_Param110'; Input_Param110.HelpString = ''; Input_Param110.ReadOnly = False; Input_Param110.BitSize = 8; Input_Param110.DataSize = 1; Input_Param110.DataType = 'BYTE'; Input_Param111.Name = 'Input_Param111'; Input_Param111.HelpString = ''; Input_Param111.ReadOnly = False; Input_Param111.BitSize = 8; Input_Param111.DataSize = 1; Input_Param111.DataType = 'BYTE'; Input_Param112.Name = 'Input_Param112'; Input_Param112.HelpString = ''; Input_Param112.ReadOnly = False; Input_Param112.BitSize = 8; Input_Param112.DataSize = 1; Input_Param112.DataType = 'BYTE'; Input_Param113.Name = 'Input_Param113'; Input_Param113.HelpString = ''; Input_Param113.ReadOnly = False; Input_Param113.BitSize = 8; Input_Param113.DataSize = 1; Input_Param113.DataType = 'BYTE';
            Input_Param114.Name = 'Input_Param114'; Input_Param114.HelpString = ''; Input_Param114.ReadOnly = False; Input_Param114.BitSize = 8; Input_Param114.DataSize = 1; Input_Param114.DataType = 'BYTE'; Input_Param115.Name = 'Input_Param115'; Input_Param115.HelpString = ''; Input_Param115.ReadOnly = False; Input_Param115.BitSize = 8; Input_Param115.DataSize = 1; Input_Param115.DataType = 'BYTE'; Input_Param116.Name = 'Input_Param116'; Input_Param116.HelpString = ''; Input_Param116.ReadOnly = False; Input_Param116.BitSize = 8; Input_Param116.DataSize = 1; Input_Param116.DataType = 'BYTE'; Input_Param117.Name = 'Input_Param117'; Input_Param117.HelpString = ''; Input_Param117.ReadOnly = False; Input_Param117.BitSize = 8; Input_Param117.DataSize = 1; Input_Param117.DataType = 'BYTE'; Input_Param118.Name = 'Input_Param118'; Input_Param118.HelpString = ''; Input_Param118.ReadOnly = False; Input_Param118.BitSize = 8; Input_Param118.DataSize = 1; Input_Param118.DataType = 'BYTE'; Input_Param119.Name = 'Input_Param119'; Input_Param119.HelpString = ''; Input_Param119.ReadOnly = False; Input_Param119.BitSize = 8; Input_Param119.DataSize = 1; Input_Param119.DataType = 'BYTE'; Input_Param120.Name = 'Input_Param120'; Input_Param120.HelpString = ''; Input_Param120.ReadOnly = False; Input_Param120.BitSize = 8;
            Input_Param120.DataSize = 1; Input_Param120.DataType = 'BYTE'; Input_Param121.Name = 'Input_Param121'; Input_Param121.HelpString = ''; Input_Param121.ReadOnly = False; Input_Param121.BitSize = 8; Input_Param121.DataSize = 1; Input_Param121.DataType = 'BYTE'; Input_Param122.Name = 'Input_Param122'; Input_Param122.HelpString = ''; Input_Param122.ReadOnly = False; Input_Param122.BitSize = 8; Input_Param122.DataSize = 1; Input_Param122.DataType = 'BYTE'; Input_Param123.Name = 'Input_Param123'; Input_Param123.HelpString = ''; Input_Param123.ReadOnly = False; Input_Param123.BitSize = 8; Input_Param123.DataSize = 1; Input_Param123.DataType = 'BYTE'; Input_Param124.Name = 'Input_Param124'; Input_Param124.HelpString = ''; Input_Param124.ReadOnly = False; Input_Param124.BitSize = 8; Input_Param124.DataSize = 1; Input_Param124.DataType = 'BYTE'; Input_Param125.Name = 'Input_Param125'; Input_Param125.HelpString = ''; Input_Param125.ReadOnly = False; Input_Param125.BitSize = 8; Input_Param125.DataSize = 1; Input_Param125.DataType = 'BYTE'; Input_Param126.Name = 'Input_Param126'; Input_Param126.HelpString = ''; Input_Param126.ReadOnly = False; Input_Param126.BitSize = 8; Input_Param126.DataSize = 1; Input_Param126.DataType = 'BYTE'; Input_Param127.Name = 'Input_Param127'; Input_Param127.HelpString = '';
            Input_Param127.ReadOnly = False; Input_Param127.BitSize = 8; Input_Param127.DataSize = 1; Input_Param127.DataType = 'BYTE'; Input_Param128.Name = 'Input_Param128'; Input_Param128.HelpString = ''; Input_Param128.ReadOnly = False; Input_Param128.BitSize = 8; Input_Param128.DataSize = 1; Input_Param128.DataType = 'BYTE'; Input_Param129.Name = 'Input_Param129'; Input_Param129.HelpString = ''; Input_Param129.ReadOnly = False; Input_Param129.BitSize = 8; Input_Param129.DataSize = 1; Input_Param129.DataType = 'BYTE'; Input_Param130.Name = 'Input_Param130'; Input_Param130.HelpString = ''; Input_Param130.ReadOnly = False; Input_Param130.BitSize = 8; Input_Param130.DataSize = 1; Input_Param130.DataType = 'BYTE'; Input_Param131.Name = 'Input_Param131'; Input_Param131.HelpString = ''; Input_Param131.ReadOnly = False; Input_Param131.BitSize = 8; Input_Param131.DataSize = 1; Input_Param131.DataType = 'BYTE'; Input_Param132.Name = 'Input_Param132'; Input_Param132.HelpString = ''; Input_Param132.ReadOnly = False; Input_Param132.BitSize = 8; Input_Param132.DataSize = 1; Input_Param132.DataType = 'BYTE'; Input_Param133.Name = 'Input_Param133'; Input_Param133.HelpString = ''; Input_Param133.ReadOnly = False; Input_Param133.BitSize = 8; Input_Param133.DataSize = 1; Input_Param133.DataType = 'BYTE';
            Input_Param134.Name = 'Input_Param134'; Input_Param134.HelpString = ''; Input_Param134.ReadOnly = False; Input_Param134.BitSize = 8; Input_Param134.DataSize = 1; Input_Param134.DataType = 'BYTE'; Input_Param135.Name = 'Input_Param135'; Input_Param135.HelpString = ''; Input_Param135.ReadOnly = False; Input_Param135.BitSize = 8; Input_Param135.DataSize = 1; Input_Param135.DataType = 'BYTE'; Input_Param136.Name = 'Input_Param136'; Input_Param136.HelpString = ''; Input_Param136.ReadOnly = False; Input_Param136.BitSize = 8; Input_Param136.DataSize = 1; Input_Param136.DataType = 'BYTE'; Input_Param137.Name = 'Input_Param137'; Input_Param137.HelpString = ''; Input_Param137.ReadOnly = False; Input_Param137.BitSize = 8; Input_Param137.DataSize = 1; Input_Param137.DataType = 'BYTE'; Input_Param138.Name = 'Input_Param138'; Input_Param138.HelpString = ''; Input_Param138.ReadOnly = False; Input_Param138.BitSize = 8; Input_Param138.DataSize = 1; Input_Param138.DataType = 'BYTE'; Input_Param139.Name = 'Input_Param139'; Input_Param139.HelpString = ''; Input_Param139.ReadOnly = False; Input_Param139.BitSize = 8; Input_Param139.DataSize = 1; Input_Param139.DataType = 'BYTE'; Input_Param140.Name = 'Input_Param140'; Input_Param140.HelpString = ''; Input_Param140.ReadOnly = False; Input_Param140.BitSize = 8;
            Input_Param140.DataSize = 1; Input_Param140.DataType = 'BYTE'; Input_Param141.Name = 'Input_Param141'; Input_Param141.HelpString = ''; Input_Param141.ReadOnly = False; Input_Param141.BitSize = 8; Input_Param141.DataSize = 1; Input_Param141.DataType = 'BYTE'; Input_Param142.Name = 'Input_Param142'; Input_Param142.HelpString = ''; Input_Param142.ReadOnly = False; Input_Param142.BitSize = 8; Input_Param142.DataSize = 1; Input_Param142.DataType = 'BYTE'; Input_Param143.Name = 'Input_Param143'; Input_Param143.HelpString = ''; Input_Param143.ReadOnly = False; Input_Param143.BitSize = 8; Input_Param143.DataSize = 1; Input_Param143.DataType = 'BYTE'; Input_Param144.Name = 'Input_Param144'; Input_Param144.HelpString = ''; Input_Param144.ReadOnly = False; Input_Param144.BitSize = 8; Input_Param144.DataSize = 1; Input_Param144.DataType = 'BYTE'; Input_Param145.Name = 'Input_Param145'; Input_Param145.HelpString = ''; Input_Param145.ReadOnly = False; Input_Param145.BitSize = 8; Input_Param145.DataSize = 1; Input_Param145.DataType = 'BYTE'; Input_Param146.Name = 'Input_Param146'; Input_Param146.HelpString = ''; Input_Param146.ReadOnly = False; Input_Param146.BitSize = 8; Input_Param146.DataSize = 1; Input_Param146.DataType = 'BYTE'; Input_Param147.Name = 'Input_Param147'; Input_Param147.HelpString = '';
            Input_Param147.ReadOnly = False; Input_Param147.BitSize = 8; Input_Param147.DataSize = 1; Input_Param147.DataType = 'BYTE'; Input_Param148.Name = 'Input_Param148'; Input_Param148.HelpString = ''; Input_Param148.ReadOnly = False; Input_Param148.BitSize = 8; Input_Param148.DataSize = 1; Input_Param148.DataType = 'BYTE'; Input_Param149.Name = 'Input_Param149'; Input_Param149.HelpString = ''; Input_Param149.ReadOnly = False; Input_Param149.BitSize = 8; Input_Param149.DataSize = 1; Input_Param149.DataType = 'BYTE'; Input_Param150.Name = 'Input_Param150'; Input_Param150.HelpString = ''; Input_Param150.ReadOnly = False; Input_Param150.BitSize = 8; Input_Param150.DataSize = 1; Input_Param150.DataType = 'BYTE'; Input_Param151.Name = 'Input_Param151'; Input_Param151.HelpString = ''; Input_Param151.ReadOnly = False; Input_Param151.BitSize = 8; Input_Param151.DataSize = 1; Input_Param151.DataType = 'BYTE'; Input_Param152.Name = 'Input_Param152'; Input_Param152.HelpString = ''; Input_Param152.ReadOnly = False; Input_Param152.BitSize = 8; Input_Param152.DataSize = 1; Input_Param152.DataType = 'BYTE'; Input_Param153.Name = 'Input_Param153'; Input_Param153.HelpString = ''; Input_Param153.ReadOnly = False; Input_Param153.BitSize = 8; Input_Param153.DataSize = 1; Input_Param153.DataType = 'BYTE';
            Input_Param154.Name = 'Input_Param154'; Input_Param154.HelpString = ''; Input_Param154.ReadOnly = False; Input_Param154.BitSize = 8; Input_Param154.DataSize = 1; Input_Param154.DataType = 'BYTE'; Input_Param155.Name = 'Input_Param155'; Input_Param155.HelpString = ''; Input_Param155.ReadOnly = False; Input_Param155.BitSize = 8; Input_Param155.DataSize = 1; Input_Param155.DataType = 'BYTE'; Input_Param156.Name = 'Input_Param156'; Input_Param156.HelpString = ''; Input_Param156.ReadOnly = False; Input_Param156.BitSize = 8; Input_Param156.DataSize = 1; Input_Param156.DataType = 'BYTE'; Input_Param157.Name = 'Input_Param157'; Input_Param157.HelpString = ''; Input_Param157.ReadOnly = False; Input_Param157.BitSize = 8; Input_Param157.DataSize = 1; Input_Param157.DataType = 'BYTE'; Input_Param158.Name = 'Input_Param158'; Input_Param158.HelpString = ''; Input_Param158.ReadOnly = False; Input_Param158.BitSize = 8; Input_Param158.DataSize = 1; Input_Param158.DataType = 'BYTE'; Input_Param159.Name = 'Input_Param159'; Input_Param159.HelpString = ''; Input_Param159.ReadOnly = False; Input_Param159.BitSize = 8; Input_Param159.DataSize = 1; Input_Param159.DataType = 'BYTE'; Input_Param160.Name = 'Input_Param160'; Input_Param160.HelpString = ''; Input_Param160.ReadOnly = False; Input_Param160.BitSize = 8;
            Input_Param160.DataSize = 1; Input_Param160.DataType = 'BYTE'; Input_Param161.Name = 'Input_Param161'; Input_Param161.HelpString = ''; Input_Param161.ReadOnly = False; Input_Param161.BitSize = 8; Input_Param161.DataSize = 1; Input_Param161.DataType = 'BYTE'; Input_Param162.Name = 'Input_Param162'; Input_Param162.HelpString = ''; Input_Param162.ReadOnly = False; Input_Param162.BitSize = 8; Input_Param162.DataSize = 1; Input_Param162.DataType = 'BYTE'; Input_Param163.Name = 'Input_Param163'; Input_Param163.HelpString = ''; Input_Param163.ReadOnly = False; Input_Param163.BitSize = 8; Input_Param163.DataSize = 1; Input_Param163.DataType = 'BYTE'; Input_Param164.Name = 'Input_Param164'; Input_Param164.HelpString = ''; Input_Param164.ReadOnly = False; Input_Param164.BitSize = 8; Input_Param164.DataSize = 1; Input_Param164.DataType = 'BYTE'; Input_Param165.Name = 'Input_Param165'; Input_Param165.HelpString = ''; Input_Param165.ReadOnly = False; Input_Param165.BitSize = 8; Input_Param165.DataSize = 1; Input_Param165.DataType = 'BYTE'; Input_Param166.Name = 'Input_Param166'; Input_Param166.HelpString = ''; Input_Param166.ReadOnly = False; Input_Param166.BitSize = 8; Input_Param166.DataSize = 1; Input_Param166.DataType = 'BYTE'; Input_Param167.Name = 'Input_Param167'; Input_Param167.HelpString = '';
            Input_Param167.ReadOnly = False; Input_Param167.BitSize = 8; Input_Param167.DataSize = 1; Input_Param167.DataType = 'BYTE'; Input_Param168.Name = 'Input_Param168'; Input_Param168.HelpString = ''; Input_Param168.ReadOnly = False; Input_Param168.BitSize = 8; Input_Param168.DataSize = 1; Input_Param168.DataType = 'BYTE'; Input_Param169.Name = 'Input_Param169'; Input_Param169.HelpString = ''; Input_Param169.ReadOnly = False; Input_Param169.BitSize = 8; Input_Param169.DataSize = 1; Input_Param169.DataType = 'BYTE'; Input_Param170.Name = 'Input_Param170'; Input_Param170.HelpString = ''; Input_Param170.ReadOnly = False; Input_Param170.BitSize = 8; Input_Param170.DataSize = 1; Input_Param170.DataType = 'BYTE'; Input_Param171.Name = 'Input_Param171'; Input_Param171.HelpString = ''; Input_Param171.ReadOnly = False; Input_Param171.BitSize = 8; Input_Param171.DataSize = 1; Input_Param171.DataType = 'BYTE'; Output_Param0.Name = 'Output_Param0'; Output_Param0.HelpString = ''; Output_Param0.ReadOnly = False; Output_Param0.BitSize = 8; Output_Param0.DataSize = 1; Output_Param0.DataType = 'BYTE'; Output_Param1.Name = 'Output_Param1'; Output_Param1.HelpString = ''; Output_Param1.ReadOnly = False; Output_Param1.BitSize = 8; Output_Param1.DataSize = 1; Output_Param1.DataType = 'BYTE';
            Output_Param2.Name = 'Output_Param2'; Output_Param2.HelpString = ''; Output_Param2.ReadOnly = False; Output_Param2.BitSize = 8; Output_Param2.DataSize = 1; Output_Param2.DataType = 'BYTE'; Output_Param3.Name = 'Output_Param3'; Output_Param3.HelpString = ''; Output_Param3.ReadOnly = False; Output_Param3.BitSize = 8; Output_Param3.DataSize = 1; Output_Param3.DataType = 'BYTE'; Output_Param4.Name = 'Output_Param4'; Output_Param4.HelpString = ''; Output_Param4.ReadOnly = False; Output_Param4.BitSize = 8; Output_Param4.DataSize = 1; Output_Param4.DataType = 'BYTE'; Output_Param5.Name = 'Output_Param5'; Output_Param5.HelpString = ''; Output_Param5.ReadOnly = False; Output_Param5.BitSize = 8; Output_Param5.DataSize = 1; Output_Param5.DataType = 'BYTE'; Output_Param6.Name = 'Output_Param6'; Output_Param6.HelpString = ''; Output_Param6.ReadOnly = False; Output_Param6.BitSize = 8; Output_Param6.DataSize = 1; Output_Param6.DataType = 'BYTE'; Output_Param7.Name = 'Output_Param7'; Output_Param7.HelpString = ''; Output_Param7.ReadOnly = False; Output_Param7.BitSize = 8; Output_Param7.DataSize = 1; Output_Param7.DataType = 'BYTE'; Output_Param8.Name = 'Output_Param8'; Output_Param8.HelpString = ''; Output_Param8.ReadOnly = False; Output_Param8.BitSize = 8;
            Output_Param8.DataSize = 1; Output_Param8.DataType = 'BYTE'; Output_Param9.Name = 'Output_Param9'; Output_Param9.HelpString = ''; Output_Param9.ReadOnly = False; Output_Param9.BitSize = 8; Output_Param9.DataSize = 1; Output_Param9.DataType = 'BYTE'; Output_Param10.Name = 'Output_Param10'; Output_Param10.HelpString = ''; Output_Param10.ReadOnly = False; Output_Param10.BitSize = 8; Output_Param10.DataSize = 1; Output_Param10.DataType = 'BYTE'; Output_Param11.Name = 'Output_Param11'; Output_Param11.HelpString = ''; Output_Param11.ReadOnly = False; Output_Param11.BitSize = 8; Output_Param11.DataSize = 1; Output_Param11.DataType = 'BYTE'; Output_Param12.Name = 'Output_Param12'; Output_Param12.HelpString = ''; Output_Param12.ReadOnly = False; Output_Param12.BitSize = 8; Output_Param12.DataSize = 1; Output_Param12.DataType = 'BYTE'; Output_Param13.Name = 'Output_Param13'; Output_Param13.HelpString = ''; Output_Param13.ReadOnly = False; Output_Param13.BitSize = 8; Output_Param13.DataSize = 1; Output_Param13.DataType = 'BYTE'; Output_Param14.Name = 'Output_Param14'; Output_Param14.HelpString = ''; Output_Param14.ReadOnly = False; Output_Param14.BitSize = 8; Output_Param14.DataSize = 1; Output_Param14.DataType = 'BYTE'; Output_Param15.Name = 'Output_Param15'; Output_Param15.HelpString = '';
            Output_Param15.ReadOnly = False; Output_Param15.BitSize = 8; Output_Param15.DataSize = 1; Output_Param15.DataType = 'BYTE'; Output_Param16.Name = 'Output_Param16'; Output_Param16.HelpString = ''; Output_Param16.ReadOnly = False; Output_Param16.BitSize = 8; Output_Param16.DataSize = 1; Output_Param16.DataType = 'BYTE'; Output_Param17.Name = 'Output_Param17'; Output_Param17.HelpString = ''; Output_Param17.ReadOnly = False; Output_Param17.BitSize = 8; Output_Param17.DataSize = 1; Output_Param17.DataType = 'BYTE'; Output_Param18.Name = 'Output_Param18'; Output_Param18.HelpString = ''; Output_Param18.ReadOnly = False; Output_Param18.BitSize = 8; Output_Param18.DataSize = 1; Output_Param18.DataType = 'BYTE'; Output_Param19.Name = 'Output_Param19'; Output_Param19.HelpString = ''; Output_Param19.ReadOnly = False; Output_Param19.BitSize = 8; Output_Param19.DataSize = 1; Output_Param19.DataType = 'BYTE'; Output_Param20.Name = 'Output_Param20'; Output_Param20.HelpString = ''; Output_Param20.ReadOnly = False; Output_Param20.BitSize = 8; Output_Param20.DataSize = 1; Output_Param20.DataType = 'BYTE'; Output_Param21.Name = 'Output_Param21'; Output_Param21.HelpString = ''; Output_Param21.ReadOnly = False; Output_Param21.BitSize = 8; Output_Param21.DataSize = 1; Output_Param21.DataType = 'BYTE';
            Output_Param22.Name = 'Output_Param22'; Output_Param22.HelpString = ''; Output_Param22.ReadOnly = False; Output_Param22.BitSize = 8; Output_Param22.DataSize = 1; Output_Param22.DataType = 'BYTE'; Output_Param23.Name = 'Output_Param23'; Output_Param23.HelpString = ''; Output_Param23.ReadOnly = False; Output_Param23.BitSize = 8; Output_Param23.DataSize = 1; Output_Param23.DataType = 'BYTE'; Output_Param24.Name = 'Output_Param24'; Output_Param24.HelpString = ''; Output_Param24.ReadOnly = False; Output_Param24.BitSize = 8; Output_Param24.DataSize = 1; Output_Param24.DataType = 'BYTE'; Output_Param25.Name = 'Output_Param25'; Output_Param25.HelpString = ''; Output_Param25.ReadOnly = False; Output_Param25.BitSize = 8; Output_Param25.DataSize = 1; Output_Param25.DataType = 'BYTE'; Output_Param26.Name = 'Output_Param26'; Output_Param26.HelpString = ''; Output_Param26.ReadOnly = False; Output_Param26.BitSize = 8; Output_Param26.DataSize = 1; Output_Param26.DataType = 'BYTE'; Output_Param27.Name = 'Output_Param27'; Output_Param27.HelpString = ''; Output_Param27.ReadOnly = False; Output_Param27.BitSize = 8; Output_Param27.DataSize = 1; Output_Param27.DataType = 'BYTE'; Output_Param28.Name = 'Output_Param28'; Output_Param28.HelpString = ''; Output_Param28.ReadOnly = False; Output_Param28.BitSize = 8;
            Output_Param28.DataSize = 1; Output_Param28.DataType = 'BYTE'; Output_Param29.Name = 'Output_Param29'; Output_Param29.HelpString = ''; Output_Param29.ReadOnly = False; Output_Param29.BitSize = 8; Output_Param29.DataSize = 1; Output_Param29.DataType = 'BYTE'; Output_Param30.Name = 'Output_Param30'; Output_Param30.HelpString = ''; Output_Param30.ReadOnly = False; Output_Param30.BitSize = 8; Output_Param30.DataSize = 1; Output_Param30.DataType = 'BYTE'; Output_Param31.Name = 'Output_Param31'; Output_Param31.HelpString = ''; Output_Param31.ReadOnly = False; Output_Param31.BitSize = 8; Output_Param31.DataSize = 1; Output_Param31.DataType = 'BYTE'; Output_Param32.Name = 'Output_Param32'; Output_Param32.HelpString = ''; Output_Param32.ReadOnly = False; Output_Param32.BitSize = 8; Output_Param32.DataSize = 1; Output_Param32.DataType = 'BYTE'; Output_Param33.Name = 'Output_Param33'; Output_Param33.HelpString = ''; Output_Param33.ReadOnly = False; Output_Param33.BitSize = 8; Output_Param33.DataSize = 1; Output_Param33.DataType = 'BYTE'; Output_Param34.Name = 'Output_Param34'; Output_Param34.HelpString = ''; Output_Param34.ReadOnly = False; Output_Param34.BitSize = 8; Output_Param34.DataSize = 1; Output_Param34.DataType = 'BYTE'; Output_Param35.Name = 'Output_Param35'; Output_Param35.HelpString = '';
            Output_Param35.ReadOnly = False; Output_Param35.BitSize = 8; Output_Param35.DataSize = 1; Output_Param35.DataType = 'BYTE'; Output_Param36.Name = 'Output_Param36'; Output_Param36.HelpString = ''; Output_Param36.ReadOnly = False; Output_Param36.BitSize = 8; Output_Param36.DataSize = 1; Output_Param36.DataType = 'BYTE'; Output_Param37.Name = 'Output_Param37'; Output_Param37.HelpString = ''; Output_Param37.ReadOnly = False; Output_Param37.BitSize = 8; Output_Param37.DataSize = 1; Output_Param37.DataType = 'BYTE'; Output_Param38.Name = 'Output_Param38'; Output_Param38.HelpString = ''; Output_Param38.ReadOnly = False; Output_Param38.BitSize = 8; Output_Param38.DataSize = 1; Output_Param38.DataType = 'BYTE'; Output_Param39.Name = 'Output_Param39'; Output_Param39.HelpString = ''; Output_Param39.ReadOnly = False; Output_Param39.BitSize = 8; Output_Param39.DataSize = 1; Output_Param39.DataType = 'BYTE'; Output_Param40.Name = 'Output_Param40'; Output_Param40.HelpString = ''; Output_Param40.ReadOnly = False; Output_Param40.BitSize = 8; Output_Param40.DataSize = 1; Output_Param40.DataType = 'BYTE'; Output_Param41.Name = 'Output_Param41'; Output_Param41.HelpString = ''; Output_Param41.ReadOnly = False; Output_Param41.BitSize = 8; Output_Param41.DataSize = 1; Output_Param41.DataType = 'BYTE';
            Output_Param42.Name = 'Output_Param42'; Output_Param42.HelpString = ''; Output_Param42.ReadOnly = False; Output_Param42.BitSize = 8; Output_Param42.DataSize = 1; Output_Param42.DataType = 'BYTE'; Output_Param43.Name = 'Output_Param43'; Output_Param43.HelpString = ''; Output_Param43.ReadOnly = False; Output_Param43.BitSize = 8; Output_Param43.DataSize = 1; Output_Param43.DataType = 'BYTE'; Output_Param44.Name = 'Output_Param44'; Output_Param44.HelpString = ''; Output_Param44.ReadOnly = False; Output_Param44.BitSize = 8; Output_Param44.DataSize = 1; Output_Param44.DataType = 'BYTE'; Output_Param45.Name = 'Output_Param45'; Output_Param45.HelpString = ''; Output_Param45.ReadOnly = False; Output_Param45.BitSize = 8; Output_Param45.DataSize = 1; Output_Param45.DataType = 'BYTE'; Output_Param46.Name = 'Output_Param46'; Output_Param46.HelpString = ''; Output_Param46.ReadOnly = False; Output_Param46.BitSize = 8; Output_Param46.DataSize = 1; Output_Param46.DataType = 'BYTE'; Output_Param47.Name = 'Output_Param47'; Output_Param47.HelpString = ''; Output_Param47.ReadOnly = False; Output_Param47.BitSize = 8; Output_Param47.DataSize = 1; Output_Param47.DataType = 'BYTE'; Output_Param48.Name = 'Output_Param48'; Output_Param48.HelpString = ''; Output_Param48.ReadOnly = False; Output_Param48.BitSize = 8;
            Output_Param48.DataSize = 1; Output_Param48.DataType = 'BYTE'; Output_Param49.Name = 'Output_Param49'; Output_Param49.HelpString = ''; Output_Param49.ReadOnly = False; Output_Param49.BitSize = 8; Output_Param49.DataSize = 1; Output_Param49.DataType = 'BYTE'; Output_Param50.Name = 'Output_Param50'; Output_Param50.HelpString = ''; Output_Param50.ReadOnly = False; Output_Param50.BitSize = 8; Output_Param50.DataSize = 1; Output_Param50.DataType = 'BYTE'; Output_Param51.Name = 'Output_Param51'; Output_Param51.HelpString = ''; Output_Param51.ReadOnly = False; Output_Param51.BitSize = 8; Output_Param51.DataSize = 1; Output_Param51.DataType = 'BYTE'; Output_Param52.Name = 'Output_Param52'; Output_Param52.HelpString = ''; Output_Param52.ReadOnly = False; Output_Param52.BitSize = 8; Output_Param52.DataSize = 1; Output_Param52.DataType = 'BYTE'; Output_Param53.Name = 'Output_Param53'; Output_Param53.HelpString = ''; Output_Param53.ReadOnly = False; Output_Param53.BitSize = 8; Output_Param53.DataSize = 1; Output_Param53.DataType = 'BYTE'; Output_Param54.Name = 'Output_Param54'; Output_Param54.HelpString = ''; Output_Param54.ReadOnly = False; Output_Param54.BitSize = 8; Output_Param54.DataSize = 1; Output_Param54.DataType = 'BYTE'; Output_Param55.Name = 'Output_Param55'; Output_Param55.HelpString = '';
            Output_Param55.ReadOnly = False; Output_Param55.BitSize = 8; Output_Param55.DataSize = 1; Output_Param55.DataType = 'BYTE'; Output_Param56.Name = 'Output_Param56'; Output_Param56.HelpString = ''; Output_Param56.ReadOnly = False; Output_Param56.BitSize = 8; Output_Param56.DataSize = 1; Output_Param56.DataType = 'BYTE'; Output_Param57.Name = 'Output_Param57'; Output_Param57.HelpString = ''; Output_Param57.ReadOnly = False; Output_Param57.BitSize = 8; Output_Param57.DataSize = 1; Output_Param57.DataType = 'BYTE'; Output_Param58.Name = 'Output_Param58'; Output_Param58.HelpString = ''; Output_Param58.ReadOnly = False; Output_Param58.BitSize = 8; Output_Param58.DataSize = 1; Output_Param58.DataType = 'BYTE'; Output_Param59.Name = 'Output_Param59'; Output_Param59.HelpString = ''; Output_Param59.ReadOnly = False; Output_Param59.BitSize = 8; Output_Param59.DataSize = 1; Output_Param59.DataType = 'BYTE'; Output_Param60.Name = 'Output_Param60'; Output_Param60.HelpString = ''; Output_Param60.ReadOnly = False; Output_Param60.BitSize = 8; Output_Param60.DataSize = 1; Output_Param60.DataType = 'BYTE'; Output_Param61.Name = 'Output_Param61'; Output_Param61.HelpString = ''; Output_Param61.ReadOnly = False; Output_Param61.BitSize = 8; Output_Param61.DataSize = 1; Output_Param61.DataType = 'BYTE';
            Output_Param62.Name = 'Output_Param62'; Output_Param62.HelpString = ''; Output_Param62.ReadOnly = False; Output_Param62.BitSize = 8; Output_Param62.DataSize = 1; Output_Param62.DataType = 'BYTE'; Output_Param63.Name = 'Output_Param63'; Output_Param63.HelpString = ''; Output_Param63.ReadOnly = False; Output_Param63.BitSize = 8; Output_Param63.DataSize = 1; Output_Param63.DataType = 'BYTE'; Output_Param64.Name = 'Output_Param64'; Output_Param64.HelpString = ''; Output_Param64.ReadOnly = False; Output_Param64.BitSize = 8; Output_Param64.DataSize = 1; Output_Param64.DataType = 'BYTE'; Output_Param65.Name = 'Output_Param65'; Output_Param65.HelpString = ''; Output_Param65.ReadOnly = False; Output_Param65.BitSize = 8; Output_Param65.DataSize = 1; Output_Param65.DataType = 'BYTE'; Output_Param66.Name = 'Output_Param66'; Output_Param66.HelpString = ''; Output_Param66.ReadOnly = False; Output_Param66.BitSize = 8; Output_Param66.DataSize = 1; Output_Param66.DataType = 'BYTE'; Output_Param67.Name = 'Output_Param67'; Output_Param67.HelpString = ''; Output_Param67.ReadOnly = False; Output_Param67.BitSize = 8; Output_Param67.DataSize = 1; Output_Param67.DataType = 'BYTE'; Output_Param68.Name = 'Output_Param68'; Output_Param68.HelpString = ''; Output_Param68.ReadOnly = False; Output_Param68.BitSize = 8;
            Output_Param68.DataSize = 1; Output_Param68.DataType = 'BYTE'; Output_Param69.Name = 'Output_Param69'; Output_Param69.HelpString = ''; Output_Param69.ReadOnly = False; Output_Param69.BitSize = 8; Output_Param69.DataSize = 1; Output_Param69.DataType = 'BYTE'; Output_Param70.Name = 'Output_Param70'; Output_Param70.HelpString = ''; Output_Param70.ReadOnly = False; Output_Param70.BitSize = 8; Output_Param70.DataSize = 1; Output_Param70.DataType = 'BYTE'; Output_Param71.Name = 'Output_Param71'; Output_Param71.HelpString = ''; Output_Param71.ReadOnly = False; Output_Param71.BitSize = 8; Output_Param71.DataSize = 1; Output_Param71.DataType = 'BYTE'; Output_Param72.Name = 'Output_Param72'; Output_Param72.HelpString = ''; Output_Param72.ReadOnly = False; Output_Param72.BitSize = 8; Output_Param72.DataSize = 1; Output_Param72.DataType = 'BYTE'; Output_Param73.Name = 'Output_Param73'; Output_Param73.HelpString = ''; Output_Param73.ReadOnly = False; Output_Param73.BitSize = 8; Output_Param73.DataSize = 1; Output_Param73.DataType = 'BYTE'; Output_Param74.Name = 'Output_Param74'; Output_Param74.HelpString = ''; Output_Param74.ReadOnly = False; Output_Param74.BitSize = 8; Output_Param74.DataSize = 1; Output_Param74.DataType = 'BYTE'; Output_Param75.Name = 'Output_Param75'; Output_Param75.HelpString = '';
            Output_Param75.ReadOnly = False; Output_Param75.BitSize = 8; Output_Param75.DataSize = 1; Output_Param75.DataType = 'BYTE'; ConfigVersion = 50660864
          input  keyenceBCVInputs : BYTE  // Input_Param0
          output keyenceBCVOutputs : BYTE  // Output_Param0
          unmapped channels: Input_Param1, Input_Param2, Input_Param3, Input_Param4, Input_Param5, Input_Param6, Input_Param7, Input_Param8, Input_Param9, Input_Param10, Input_Param11, Input_Param12, Input_Param13, Input_Param14, Input_Param15, Input_Param16, Input_Param17, Input_Param18, Input_Param19, Input_Param20, Input_Param21, Input_Param22, Input_Param23, Input_Param24, Input_Param25, Input_Param26, Input_Param27, Input_Param28, Input_Param29, Input_Param30, Input_Param31, Input_Param32, Input_Param33, Input_Param34, Input_Param35, Input_Param36, Input_Param37, Input_Param38, Input_Param39, Input_Param40,
            Input_Param41, Input_Param42, Input_Param43, Input_Param44, Input_Param45, Input_Param46, Input_Param47, Input_Param48, Input_Param49, Input_Param50, Input_Param51, Input_Param52, Input_Param53, Input_Param54, Input_Param55, Input_Param56, Input_Param57, Input_Param58, Input_Param59, Input_Param60, Input_Param61, Input_Param62, Input_Param63, Input_Param64, Input_Param65, Input_Param66, Input_Param67, Input_Param68, Input_Param69, Input_Param70, Input_Param71, Input_Param72, Input_Param73, Input_Param74, Input_Param75, Input_Param76, Input_Param77, Input_Param78, Input_Param79, Input_Param80,
            Input_Param81, Input_Param82, Input_Param83, Input_Param84, Input_Param85, Input_Param86, Input_Param87, Input_Param88, Input_Param89, Input_Param90, Input_Param91, Input_Param92, Input_Param93, Input_Param94, Input_Param95, Input_Param96, Input_Param97, Input_Param98, Input_Param99, Input_Param100, Input_Param101, Input_Param102, Input_Param103, Input_Param104, Input_Param105, Input_Param106, Input_Param107, Input_Param108, Input_Param109, Input_Param110, Input_Param111, Input_Param112, Input_Param113, Input_Param114, Input_Param115, Input_Param116, Input_Param117, Input_Param118, Input_Param119, Input_Param120,
            Input_Param121, Input_Param122, Input_Param123, Input_Param124, Input_Param125, Input_Param126, Input_Param127, Input_Param128, Input_Param129, Input_Param130, Input_Param131, Input_Param132, Input_Param133, Input_Param134, Input_Param135, Input_Param136, Input_Param137, Input_Param138, Input_Param139, Input_Param140, Input_Param141, Input_Param142, Input_Param143, Input_Param144, Input_Param145, Input_Param146, Input_Param147, Input_Param148, Input_Param149, Input_Param150, Input_Param151, Input_Param152, Input_Param153, Input_Param154, Input_Param155, Input_Param156, Input_Param157, Input_Param158, Input_Param159, Input_Param160,
            Input_Param161, Input_Param162, Input_Param163, Input_Param164, Input_Param165, Input_Param166, Input_Param167, Input_Param168, Input_Param169, Input_Param170, Input_Param171, Output_Param1, Output_Param2, Output_Param3, Output_Param4, Output_Param5, Output_Param6, Output_Param7, Output_Param8, Output_Param9, Output_Param10, Output_Param11, Output_Param12, Output_Param13, Output_Param14, Output_Param15, Output_Param16, Output_Param17, Output_Param18, Output_Param19, Output_Param20, Output_Param21, Output_Param22, Output_Param23, Output_Param24, Output_Param25, Output_Param26, Output_Param27, Output_Param28, Output_Param29,
            Output_Param30, Output_Param31, Output_Param32, Output_Param33, Output_Param34, Output_Param35, Output_Param36, Output_Param37, Output_Param38, Output_Param39, Output_Param40, Output_Param41, Output_Param42, Output_Param43, Output_Param44, Output_Param45, Output_Param46, Output_Param47, Output_Param48, Output_Param49, Output_Param50, Output_Param51, Output_Param52, Output_Param53, Output_Param54, Output_Param55, Output_Param56, Output_Param57, Output_Param58, Output_Param59, Output_Param60, Output_Param61, Output_Param62, Output_Param63, Output_Param64, Output_Param65, Output_Param66, Output_Param67, Output_Param68, Output_Param69,
            Output_Param70, Output_Param71, Output_Param72, Output_Param73, Output_Param74, Output_Param75
      MSFMotor : SSM23IP-3EG, Applied Motion Products, Inc, order no. SSM23IP-3EG, version Major Revision=16#3, Minor Revision = 16#3
          settings: INITIALIZED = TRUE; IP address of Target = [16#C0,16#A8,16#0A,16#35]; Keying.Check Device Type = FALSE; Keying.Check Vendor Code = FALSE; Keying.Check Product Code = FALSE; Keying.Check Major Revision = FALSE; Keying.Check Minor Revision = FALSE; RequiredConfigVersion = 50660864; Number of Connections = 1; Connection Settings.Requested packet intervall = 10000 µs; Connection Settings.OT Connection Parameters = 18502; Connection Settings.TO Connection Parameters = 18490; Connection Settings.Connection Flags = 1056; Connection Settings.Connection Path Size = 8; Connection Settings.Large OT Connection Parameters = 1207959622; Connection Settings.Large TO Connection Parameters = 1207959610; Heartbeat Multiplier = 1; Status Code.ReadOnly = False; Status Code.BitSize = 32; Status Code.DataSize = 4; Alarm Code.ReadOnly = False; Alarm Code.BitSize = 32; Alarm Code.DataSize = 4; Supply Voltage.ReadOnly = False; Supply Voltage.BitSize = 32; Supply Voltage.DataSize = 4; Actual Current.ReadOnly = False; Actual Current.BitSize = 32; Actual Current.DataSize = 4; Drive Temperature.ReadOnly = False; Drive Temperature.BitSize = 32; Drive Temperature.DataSize = 4; Encoder Position.ReadOnly = False; Encoder Position.BitSize = 32; Encoder Position.DataSize = 4; Absolute Position.ReadOnly = False; Absolute Position.BitSize = 32; Absolute Position.DataSize = 4; Position Error.ReadOnly = False; Position Error.BitSize = 32;
            Position Error.DataSize = 4; Actual Velocity.ReadOnly = False; Actual Velocity.BitSize = 32; Actual Velocity.DataSize = 4; Input Status (extended).ReadOnly = False; Input Status (extended).BitSize = 32; Input Status (extended).DataSize = 4; Input Status (main).ReadOnly = False; Input Status (main).BitSize = 32; Input Status (main).DataSize = 4; Output Status.ReadOnly = False; Output Status.BitSize = 32; Output Status.DataSize = 4; Analog Input 1.ReadOnly = False; Analog Input 1.BitSize = 32; Analog Input 1.DataSize = 4; Analog Input 2.ReadOnly = False; Analog Input 2.BitSize = 32; Analog Input 2.DataSize = 4; Command Word.ReadOnly = False; Command Word.BitSize = 32; Command Word.DataSize = 4; Jog Speed.ReadOnly = False; Jog Speed.BitSize = 32; Jog Speed.DataSize = 4; Jog Accel.ReadOnly = False; Jog Accel.BitSize = 32; Jog Accel.DataSize = 4; Jog Decel.ReadOnly = False; Jog Decel.BitSize = 32; Jog Decel.DataSize = 4; Point-to-Point Velocity.ReadOnly = False; Point-to-Point Velocity.BitSize = 32; Point-to-Point Velocity.DataSize = 4; Point-to-Point Acceleration.ReadOnly = False; Point-to-Point Acceleration.BitSize = 32; Point-to-Point Acceleration.DataSize = 4; Point-to-Point Deceleration.ReadOnly = False; Point-to-Point Deceleration.BitSize = 32; Point-to-Point Deceleration.DataSize = 4;
            Point-to-Point Distance.ReadOnly = False; Point-to-Point Distance.BitSize = 32; Point-to-Point Distance.DataSize = 4; Current Command.ReadOnly = False; Current Command.BitSize = 32; Current Command.DataSize = 4; SCL Command Letters.ReadOnly = False; SCL Command Letters.BitSize = 32; SCL Command Letters.DataSize = 4; Data/SCL Register 1.ReadOnly = False; Data/SCL Register 1.BitSize = 32; Data/SCL Register 1.DataSize = 4; Data/SCL Register 2.ReadOnly = False; Data/SCL Register 2.BitSize = 32; Data/SCL Register 2.DataSize = 4; Reserved 1.ReadOnly = False; Reserved 1.BitSize = 32; Reserved 1.DataSize = 4; Reserved 2.ReadOnly = False; Reserved 2.BitSize = 32; Reserved 2.DataSize = 4; Reserved 3.ReadOnly = False; Reserved 3.BitSize = 32; Reserved 3.DataSize = 4; Reserved 4.ReadOnly = False; Reserved 4.BitSize = 32; Reserved 4.DataSize = 4; Status Code.Name = 'Status Code'; Status Code.HelpString = ''; Status Code.ReadOnly = False; Status Code.BitSize = 32; Status Code.DataSize = 4; Status Code.DataType = 'DINT'; Alarm Code.Name = 'Alarm Code'; Alarm Code.HelpString = ''; Alarm Code.ReadOnly = False; Alarm Code.BitSize = 32; Alarm Code.DataSize = 4; Alarm Code.DataType = 'DINT'; Supply Voltage.Name = 'Supply Voltage';
            Supply Voltage.HelpString = ''; Supply Voltage.ReadOnly = False; Supply Voltage.BitSize = 32; Supply Voltage.DataSize = 4; Supply Voltage.DataType = 'DINT'; Actual Current.Name = 'Actual Current'; Actual Current.HelpString = ''; Actual Current.ReadOnly = False; Actual Current.BitSize = 32; Actual Current.DataSize = 4; Actual Current.DataType = 'DINT'; Drive Temperature.Name = 'Drive Temperature'; Drive Temperature.HelpString = ''; Drive Temperature.ReadOnly = False; Drive Temperature.BitSize = 32; Drive Temperature.DataSize = 4; Drive Temperature.DataType = 'DINT'; Encoder Position.Name = 'Encoder Position'; Encoder Position.HelpString = ''; Encoder Position.ReadOnly = False; Encoder Position.BitSize = 32; Encoder Position.DataSize = 4; Encoder Position.DataType = 'DINT'; Absolute Position.Name = 'Absolute Position'; Absolute Position.HelpString = ''; Absolute Position.ReadOnly = False; Absolute Position.BitSize = 32; Absolute Position.DataSize = 4; Absolute Position.DataType = 'DINT'; Position Error.Name = 'Position Error'; Position Error.HelpString = ''; Position Error.ReadOnly = False; Position Error.BitSize = 32; Position Error.DataSize = 4; Position Error.DataType = 'DINT'; Actual Velocity.Name = 'Actual Velocity'; Actual Velocity.HelpString = ''; Actual Velocity.ReadOnly = False; Actual Velocity.BitSize = 32; Actual Velocity.DataSize = 4;
            Actual Velocity.DataType = 'DINT'; Input Status (extended).Name = 'Input Status (extended)'; Input Status (extended).HelpString = ''; Input Status (extended).ReadOnly = False; Input Status (extended).BitSize = 32; Input Status (extended).DataSize = 4; Input Status (extended).DataType = 'DINT'; Input Status (main).Name = 'Input Status (main)'; Input Status (main).HelpString = ''; Input Status (main).ReadOnly = False; Input Status (main).BitSize = 32; Input Status (main).DataSize = 4; Input Status (main).DataType = 'DINT'; Output Status.Name = 'Output Status'; Output Status.HelpString = ''; Output Status.ReadOnly = False; Output Status.BitSize = 32; Output Status.DataSize = 4; Output Status.DataType = 'DINT'; Analog Input 1.Name = 'Analog Input 1'; Analog Input 1.HelpString = ''; Analog Input 1.ReadOnly = False; Analog Input 1.BitSize = 32; Analog Input 1.DataSize = 4; Analog Input 1.DataType = 'DINT'; Analog Input 2.Name = 'Analog Input 2'; Analog Input 2.HelpString = ''; Analog Input 2.ReadOnly = False; Analog Input 2.BitSize = 32; Analog Input 2.DataSize = 4; Analog Input 2.DataType = 'DINT'; Command Word.Name = 'Command Word'; Command Word.HelpString = ''; Command Word.ReadOnly = False; Command Word.BitSize = 32; Command Word.DataSize = 4; Command Word.DataType = 'DINT'; Jog Speed.Name = 'Jog Speed'; Jog Speed.HelpString = ''; Jog Speed.ReadOnly = False;
            Jog Speed.BitSize = 32; Jog Speed.DataSize = 4; Jog Speed.DataType = 'DINT'; Jog Accel.Name = 'Jog Accel'; Jog Accel.HelpString = ''; Jog Accel.ReadOnly = False; Jog Accel.BitSize = 32; Jog Accel.DataSize = 4; Jog Accel.DataType = 'DINT'; Jog Decel.Name = 'Jog Decel'; Jog Decel.HelpString = ''; Jog Decel.ReadOnly = False; Jog Decel.BitSize = 32; Jog Decel.DataSize = 4; Jog Decel.DataType = 'DINT'; Point-to-Point Velocity.Name = 'Point-to-Point Velocity'; Point-to-Point Velocity.HelpString = ''; Point-to-Point Velocity.ReadOnly = False; Point-to-Point Velocity.BitSize = 32; Point-to-Point Velocity.DataSize = 4; Point-to-Point Velocity.DataType = 'DINT'; Point-to-Point Acceleration.Name = 'Point-to-Point Acceleration'; Point-to-Point Acceleration.HelpString = ''; Point-to-Point Acceleration.ReadOnly = False; Point-to-Point Acceleration.BitSize = 32; Point-to-Point Acceleration.DataSize = 4; Point-to-Point Acceleration.DataType = 'DINT'; Point-to-Point Deceleration.Name = 'Point-to-Point Deceleration'; Point-to-Point Deceleration.HelpString = ''; Point-to-Point Deceleration.ReadOnly = False; Point-to-Point Deceleration.BitSize = 32; Point-to-Point Deceleration.DataSize = 4; Point-to-Point Deceleration.DataType = 'DINT'; Point-to-Point Distance.Name = 'Point-to-Point Distance'; Point-to-Point Distance.HelpString = ''; Point-to-Point Distance.ReadOnly = False; Point-to-Point Distance.BitSize = 32; Point-to-Point Distance.DataSize = 4; Point-to-Point Distance.DataType = 'DINT'; Current Command.Name = 'Current Command';
            Current Command.HelpString = ''; Current Command.ReadOnly = False; Current Command.BitSize = 32; Current Command.DataSize = 4; Current Command.DataType = 'DINT'; SCL Command Letters.Name = 'SCL Command Letters'; SCL Command Letters.HelpString = ''; SCL Command Letters.ReadOnly = False; SCL Command Letters.BitSize = 32; SCL Command Letters.DataSize = 4; SCL Command Letters.DataType = 'DINT'; Data/SCL Register 1.Name = 'Data/SCL Register 1'; Data/SCL Register 1.HelpString = ''; Data/SCL Register 1.ReadOnly = False; Data/SCL Register 1.BitSize = 32; Data/SCL Register 1.DataSize = 4; Data/SCL Register 1.DataType = 'DINT'; Data/SCL Register 2.Name = 'Data/SCL Register 2'; Data/SCL Register 2.HelpString = ''; Data/SCL Register 2.ReadOnly = False; Data/SCL Register 2.BitSize = 32; Data/SCL Register 2.DataSize = 4; Data/SCL Register 2.DataType = 'DINT'; Reserved 1.Name = 'Reserved 1'; Reserved 1.HelpString = ''; Reserved 1.ReadOnly = False; Reserved 1.BitSize = 32; Reserved 1.DataSize = 4; Reserved 1.DataType = 'DINT'; Reserved 2.Name = 'Reserved 2'; Reserved 2.HelpString = ''; Reserved 2.ReadOnly = False; Reserved 2.BitSize = 32; Reserved 2.DataSize = 4; Reserved 2.DataType = 'DINT'; Reserved 3.Name = 'Reserved 3'; Reserved 3.HelpString = ''; Reserved 3.ReadOnly = False; Reserved 3.BitSize = 32; Reserved 3.DataSize = 4;
            Reserved 3.DataType = 'DINT'; Reserved 4.Name = 'Reserved 4'; Reserved 4.HelpString = ''; Reserved 4.ReadOnly = False; Reserved 4.BitSize = 32; Reserved 4.DataSize = 4; Reserved 4.DataType = 'DINT'; ConfigVersion = 50660864
          input  sealFlattenerHorizontalMotorInputs : DINT  // Status Code
          output sealFlattenerHorizontalMotorOutputs : DINT  // Command Word
          unmapped channels: Alarm Code, Supply Voltage, Actual Current, Drive Temperature, Encoder Position, Absolute Position, Position Error, Actual Velocity, Input Status (extended), Input Status (main), Output Status, Analog Input 1, Analog Input 2, Jog Speed, Jog Accel, Jog Decel, Point-to-Point Velocity, Point-to-Point Acceleration, Point-to-Point Deceleration, Point-to-Point Distance, Current Command, SCL Command Letters, Data/SCL Register 1, Data/SCL Register 2, Reserved 1, Reserved 2, Reserved 3, Reserved 4
      Panther_PA : WAGO 2759-101 ENIP, WAGO Kontakttechnik GmbH & Co. KG, order no. WagoAppEtherNetIP_Adapter, version Major Revision=16#1, Minor Revision = 16#1 (disabled)
          settings: INITIALIZED = TRUE; IP address of Target = [16#C0,16#A8,16#0A,16#A2]; Keying.Check Minor Revision = FALSE; RequiredConfigVersion = 50660864; Number of Connections = 1; Connection Settings.Requested packet intervall = 10000 µs; Connection Settings.OT Connection Parameters = 18470; Connection Settings.TO Connection Parameters = 18466; Connection Settings.Connection Flags = 1056; Connection Settings.Connection Path Size = 8; Connection Settings.Config#2 Size = 2; Connection Settings.Large OT Connection Parameters = 1207959590; Connection Settings.Large TO Connection Parameters = 1207959586; Configuration Data = [16#00,16#00]; Heartbeat Multiplier = 1; Port 1 Output Data_Param0.ReadOnly = False; Port 1 Output Data_Param0.BitSize = 8; Port 1 Output Data_Param0.DataSize = 1; Port 1 Output Data_Param1.ReadOnly = False; Port 1 Output Data_Param1.BitSize = 8; Port 1 Output Data_Param1.DataSize = 1; Port 1 Output Data_Param2.ReadOnly = False; Port 1 Output Data_Param2.BitSize = 8; Port 1 Output Data_Param2.DataSize = 1; Port 1 Output Data_Param3.ReadOnly = False; Port 1 Output Data_Param3.BitSize = 8; Port 1 Output Data_Param3.DataSize = 1; Port 1 Output Data_Param4.ReadOnly = False; Port 1 Output Data_Param4.BitSize = 8; Port 1 Output Data_Param4.DataSize = 1; Port 1 Output Data_Param5.ReadOnly = False; Port 1 Output Data_Param5.BitSize = 8; Port 1 Output Data_Param5.DataSize = 1; Port 1 Output Data_Param6.ReadOnly = False; Port 1 Output Data_Param6.BitSize = 8; Port 1 Output Data_Param6.DataSize = 1; Port 1 Output Data_Param7.ReadOnly = False; Port 1 Output Data_Param7.BitSize = 8; Port 1 Output Data_Param7.DataSize = 1; Port 1 Output Data_Param8.ReadOnly = False;
            Port 1 Output Data_Param8.BitSize = 8; Port 1 Output Data_Param8.DataSize = 1; Port 1 Output Data_Param9.ReadOnly = False; Port 1 Output Data_Param9.BitSize = 8; Port 1 Output Data_Param9.DataSize = 1; Port 1 Output Data_Param10.ReadOnly = False; Port 1 Output Data_Param10.BitSize = 8; Port 1 Output Data_Param10.DataSize = 1; Port 1 Output Data_Param11.ReadOnly = False; Port 1 Output Data_Param11.BitSize = 8; Port 1 Output Data_Param11.DataSize = 1; Port 1 Output Data_Param12.ReadOnly = False; Port 1 Output Data_Param12.BitSize = 8; Port 1 Output Data_Param12.DataSize = 1; Port 1 Output Data_Param13.ReadOnly = False; Port 1 Output Data_Param13.BitSize = 8; Port 1 Output Data_Param13.DataSize = 1; Port 1 Output Data_Param14.ReadOnly = False; Port 1 Output Data_Param14.BitSize = 8; Port 1 Output Data_Param14.DataSize = 1; Port 1 Output Data_Param15.ReadOnly = False; Port 1 Output Data_Param15.BitSize = 8; Port 1 Output Data_Param15.DataSize = 1; Port 1 Output Data_Param16.ReadOnly = False; Port 1 Output Data_Param16.BitSize = 8; Port 1 Output Data_Param16.DataSize = 1; Port 1 Output Data_Param17.ReadOnly = False; Port 1 Output Data_Param17.BitSize = 8; Port 1 Output Data_Param17.DataSize = 1; Port 1 Output Data_Param18.ReadOnly = False; Port 1 Output Data_Param18.BitSize = 8; Port 1 Output Data_Param18.DataSize = 1; Port 1 Output Data_Param19.ReadOnly = False; Port 1 Output Data_Param19.BitSize = 8; Port 1 Output Data_Param19.DataSize = 1; Port 1 Output Data_Param20.ReadOnly = False; Port 1 Output Data_Param20.BitSize = 8; Port 1 Output Data_Param20.DataSize = 1; Port 1 Output Data_Param21.ReadOnly = False; Port 1 Output Data_Param21.BitSize = 8;
            Port 1 Output Data_Param21.DataSize = 1; Port 1 Output Data_Param22.ReadOnly = False; Port 1 Output Data_Param22.BitSize = 8; Port 1 Output Data_Param22.DataSize = 1; Port 1 Output Data_Param23.ReadOnly = False; Port 1 Output Data_Param23.BitSize = 8; Port 1 Output Data_Param23.DataSize = 1; Port 1 Output Data_Param24.ReadOnly = False; Port 1 Output Data_Param24.BitSize = 8; Port 1 Output Data_Param24.DataSize = 1; Port 1 Output Data_Param25.ReadOnly = False; Port 1 Output Data_Param25.BitSize = 8; Port 1 Output Data_Param25.DataSize = 1; Port 1 Output Data_Param26.ReadOnly = False; Port 1 Output Data_Param26.BitSize = 8; Port 1 Output Data_Param26.DataSize = 1; Port 1 Output Data_Param27.ReadOnly = False; Port 1 Output Data_Param27.BitSize = 8; Port 1 Output Data_Param27.DataSize = 1; Port 1 Output Data_Param28.ReadOnly = False; Port 1 Output Data_Param28.BitSize = 8; Port 1 Output Data_Param28.DataSize = 1; Port 1 Output Data_Param29.ReadOnly = False; Port 1 Output Data_Param29.BitSize = 8; Port 1 Output Data_Param29.DataSize = 1; Port 1 Output Data_Param30.ReadOnly = False; Port 1 Output Data_Param30.BitSize = 8; Port 1 Output Data_Param30.DataSize = 1; Port 1 Output Data_Param31.ReadOnly = False; Port 1 Output Data_Param31.BitSize = 8; Port 1 Output Data_Param31.DataSize = 1; Port 1 Input Data_Param0.ReadOnly = False; Port 1 Input Data_Param0.BitSize = 8; Port 1 Input Data_Param0.DataSize = 1; Port 1 Input Data_Param1.ReadOnly = False; Port 1 Input Data_Param1.BitSize = 8; Port 1 Input Data_Param1.DataSize = 1; Port 1 Input Data_Param2.ReadOnly = False; Port 1 Input Data_Param2.BitSize = 8; Port 1 Input Data_Param2.DataSize = 1;
            Port 1 Input Data_Param3.ReadOnly = False; Port 1 Input Data_Param3.BitSize = 8; Port 1 Input Data_Param3.DataSize = 1; Port 1 Input Data_Param4.ReadOnly = False; Port 1 Input Data_Param4.BitSize = 8; Port 1 Input Data_Param4.DataSize = 1; Port 1 Input Data_Param5.ReadOnly = False; Port 1 Input Data_Param5.BitSize = 8; Port 1 Input Data_Param5.DataSize = 1; Port 1 Input Data_Param6.ReadOnly = False; Port 1 Input Data_Param6.BitSize = 8; Port 1 Input Data_Param6.DataSize = 1; Port 1 Input Data_Param7.ReadOnly = False; Port 1 Input Data_Param7.BitSize = 8; Port 1 Input Data_Param7.DataSize = 1; Port 1 Input Data_Param8.ReadOnly = False; Port 1 Input Data_Param8.BitSize = 8; Port 1 Input Data_Param8.DataSize = 1; Port 1 Input Data_Param9.ReadOnly = False; Port 1 Input Data_Param9.BitSize = 8; Port 1 Input Data_Param9.DataSize = 1; Port 1 Input Data_Param10.ReadOnly = False; Port 1 Input Data_Param10.BitSize = 8; Port 1 Input Data_Param10.DataSize = 1; Port 1 Input Data_Param11.ReadOnly = False; Port 1 Input Data_Param11.BitSize = 8; Port 1 Input Data_Param11.DataSize = 1; Port 1 Input Data_Param12.ReadOnly = False; Port 1 Input Data_Param12.BitSize = 8; Port 1 Input Data_Param12.DataSize = 1; Port 1 Input Data_Param13.ReadOnly = False; Port 1 Input Data_Param13.BitSize = 8; Port 1 Input Data_Param13.DataSize = 1; Port 1 Input Data_Param14.ReadOnly = False; Port 1 Input Data_Param14.BitSize = 8; Port 1 Input Data_Param14.DataSize = 1; Port 1 Input Data_Param15.ReadOnly = False; Port 1 Input Data_Param15.BitSize = 8; Port 1 Input Data_Param15.DataSize = 1; Port 1 Input Data_Param16.ReadOnly = False;
            Port 1 Input Data_Param16.BitSize = 8; Port 1 Input Data_Param16.DataSize = 1; Port 1 Input Data_Param17.ReadOnly = False; Port 1 Input Data_Param17.BitSize = 8; Port 1 Input Data_Param17.DataSize = 1; Port 1 Input Data_Param18.ReadOnly = False; Port 1 Input Data_Param18.BitSize = 8; Port 1 Input Data_Param18.DataSize = 1; Port 1 Input Data_Param19.ReadOnly = False; Port 1 Input Data_Param19.BitSize = 8; Port 1 Input Data_Param19.DataSize = 1; Port 1 Input Data_Param20.ReadOnly = False; Port 1 Input Data_Param20.BitSize = 8; Port 1 Input Data_Param20.DataSize = 1; Port 1 Input Data_Param21.ReadOnly = False; Port 1 Input Data_Param21.BitSize = 8; Port 1 Input Data_Param21.DataSize = 1; Port 1 Input Data_Param22.ReadOnly = False; Port 1 Input Data_Param22.BitSize = 8; Port 1 Input Data_Param22.DataSize = 1; Port 1 Input Data_Param23.ReadOnly = False; Port 1 Input Data_Param23.BitSize = 8; Port 1 Input Data_Param23.DataSize = 1; Port 1 Input Data_Param24.ReadOnly = False; Port 1 Input Data_Param24.BitSize = 8; Port 1 Input Data_Param24.DataSize = 1; Port 1 Input Data_Param25.ReadOnly = False; Port 1 Input Data_Param25.BitSize = 8; Port 1 Input Data_Param25.DataSize = 1; Port 1 Input Data_Param26.ReadOnly = False; Port 1 Input Data_Param26.BitSize = 8; Port 1 Input Data_Param26.DataSize = 1; Port 1 Input Data_Param27.ReadOnly = False; Port 1 Input Data_Param27.BitSize = 8; Port 1 Input Data_Param27.DataSize = 1; Port 1 Input Data_Param28.ReadOnly = False; Port 1 Input Data_Param28.BitSize = 8; Port 1 Input Data_Param28.DataSize = 1; Port 1 Input Data_Param29.ReadOnly = False; Port 1 Input Data_Param29.BitSize = 8;
            Port 1 Input Data_Param29.DataSize = 1; Port 1 Input Data_Param30.ReadOnly = False; Port 1 Input Data_Param30.BitSize = 8; Port 1 Input Data_Param30.DataSize = 1; Port 1 Input Data_Param31.ReadOnly = False; Port 1 Input Data_Param31.BitSize = 8; Port 1 Input Data_Param31.DataSize = 1; Port 1 Output Data_Param0.Name = 'Port 1 Output Data_Param0'; Port 1 Output Data_Param0.HelpString = ''; Port 1 Output Data_Param0.ReadOnly = False; Port 1 Output Data_Param0.BitSize = 8; Port 1 Output Data_Param0.DataSize = 1; Port 1 Output Data_Param0.DataType = 'BYTE'; Port 1 Output Data_Param1.Name = 'Port 1 Output Data_Param1'; Port 1 Output Data_Param1.HelpString = ''; Port 1 Output Data_Param1.ReadOnly = False; Port 1 Output Data_Param1.BitSize = 8; Port 1 Output Data_Param1.DataSize = 1; Port 1 Output Data_Param1.DataType = 'BYTE'; Port 1 Output Data_Param2.Name = 'Port 1 Output Data_Param2'; Port 1 Output Data_Param2.HelpString = ''; Port 1 Output Data_Param2.ReadOnly = False; Port 1 Output Data_Param2.BitSize = 8; Port 1 Output Data_Param2.DataSize = 1; Port 1 Output Data_Param2.DataType = 'BYTE'; Port 1 Output Data_Param3.Name = 'Port 1 Output Data_Param3'; Port 1 Output Data_Param3.HelpString = ''; Port 1 Output Data_Param3.ReadOnly = False; Port 1 Output Data_Param3.BitSize = 8; Port 1 Output Data_Param3.DataSize = 1; Port 1 Output Data_Param3.DataType = 'BYTE'; Port 1 Output Data_Param4.Name = 'Port 1 Output Data_Param4'; Port 1 Output Data_Param4.HelpString = ''; Port 1 Output Data_Param4.ReadOnly = False; Port 1 Output Data_Param4.BitSize = 8; Port 1 Output Data_Param4.DataSize = 1; Port 1 Output Data_Param4.DataType = 'BYTE'; Port 1 Output Data_Param5.Name = 'Port 1 Output Data_Param5'; Port 1 Output Data_Param5.HelpString = ''; Port 1 Output Data_Param5.ReadOnly = False;
            Port 1 Output Data_Param5.BitSize = 8; Port 1 Output Data_Param5.DataSize = 1; Port 1 Output Data_Param5.DataType = 'BYTE'; Port 1 Output Data_Param6.Name = 'Port 1 Output Data_Param6'; Port 1 Output Data_Param6.HelpString = ''; Port 1 Output Data_Param6.ReadOnly = False; Port 1 Output Data_Param6.BitSize = 8; Port 1 Output Data_Param6.DataSize = 1; Port 1 Output Data_Param6.DataType = 'BYTE'; Port 1 Output Data_Param7.Name = 'Port 1 Output Data_Param7'; Port 1 Output Data_Param7.HelpString = ''; Port 1 Output Data_Param7.ReadOnly = False; Port 1 Output Data_Param7.BitSize = 8; Port 1 Output Data_Param7.DataSize = 1; Port 1 Output Data_Param7.DataType = 'BYTE'; Port 1 Output Data_Param8.Name = 'Port 1 Output Data_Param8'; Port 1 Output Data_Param8.HelpString = ''; Port 1 Output Data_Param8.ReadOnly = False; Port 1 Output Data_Param8.BitSize = 8; Port 1 Output Data_Param8.DataSize = 1; Port 1 Output Data_Param8.DataType = 'BYTE'; Port 1 Output Data_Param9.Name = 'Port 1 Output Data_Param9'; Port 1 Output Data_Param9.HelpString = ''; Port 1 Output Data_Param9.ReadOnly = False; Port 1 Output Data_Param9.BitSize = 8; Port 1 Output Data_Param9.DataSize = 1; Port 1 Output Data_Param9.DataType = 'BYTE'; Port 1 Output Data_Param10.Name = 'Port 1 Output Data_Param10'; Port 1 Output Data_Param10.HelpString = ''; Port 1 Output Data_Param10.ReadOnly = False; Port 1 Output Data_Param10.BitSize = 8; Port 1 Output Data_Param10.DataSize = 1; Port 1 Output Data_Param10.DataType = 'BYTE'; Port 1 Output Data_Param11.Name = 'Port 1 Output Data_Param11'; Port 1 Output Data_Param11.HelpString = ''; Port 1 Output Data_Param11.ReadOnly = False; Port 1 Output Data_Param11.BitSize = 8; Port 1 Output Data_Param11.DataSize = 1; Port 1 Output Data_Param11.DataType = 'BYTE'; Port 1 Output Data_Param12.Name = 'Port 1 Output Data_Param12';
            Port 1 Output Data_Param12.HelpString = ''; Port 1 Output Data_Param12.ReadOnly = False; Port 1 Output Data_Param12.BitSize = 8; Port 1 Output Data_Param12.DataSize = 1; Port 1 Output Data_Param12.DataType = 'BYTE'; Port 1 Output Data_Param13.Name = 'Port 1 Output Data_Param13'; Port 1 Output Data_Param13.HelpString = ''; Port 1 Output Data_Param13.ReadOnly = False; Port 1 Output Data_Param13.BitSize = 8; Port 1 Output Data_Param13.DataSize = 1; Port 1 Output Data_Param13.DataType = 'BYTE'; Port 1 Output Data_Param14.Name = 'Port 1 Output Data_Param14'; Port 1 Output Data_Param14.HelpString = ''; Port 1 Output Data_Param14.ReadOnly = False; Port 1 Output Data_Param14.BitSize = 8; Port 1 Output Data_Param14.DataSize = 1; Port 1 Output Data_Param14.DataType = 'BYTE'; Port 1 Output Data_Param15.Name = 'Port 1 Output Data_Param15'; Port 1 Output Data_Param15.HelpString = ''; Port 1 Output Data_Param15.ReadOnly = False; Port 1 Output Data_Param15.BitSize = 8; Port 1 Output Data_Param15.DataSize = 1; Port 1 Output Data_Param15.DataType = 'BYTE'; Port 1 Output Data_Param16.Name = 'Port 1 Output Data_Param16'; Port 1 Output Data_Param16.HelpString = ''; Port 1 Output Data_Param16.ReadOnly = False; Port 1 Output Data_Param16.BitSize = 8; Port 1 Output Data_Param16.DataSize = 1; Port 1 Output Data_Param16.DataType = 'BYTE'; Port 1 Output Data_Param17.Name = 'Port 1 Output Data_Param17'; Port 1 Output Data_Param17.HelpString = ''; Port 1 Output Data_Param17.ReadOnly = False; Port 1 Output Data_Param17.BitSize = 8; Port 1 Output Data_Param17.DataSize = 1; Port 1 Output Data_Param17.DataType = 'BYTE'; Port 1 Output Data_Param18.Name = 'Port 1 Output Data_Param18'; Port 1 Output Data_Param18.HelpString = ''; Port 1 Output Data_Param18.ReadOnly = False; Port 1 Output Data_Param18.BitSize = 8; Port 1 Output Data_Param18.DataSize = 1;
            Port 1 Output Data_Param18.DataType = 'BYTE'; Port 1 Output Data_Param19.Name = 'Port 1 Output Data_Param19'; Port 1 Output Data_Param19.HelpString = ''; Port 1 Output Data_Param19.ReadOnly = False; Port 1 Output Data_Param19.BitSize = 8; Port 1 Output Data_Param19.DataSize = 1; Port 1 Output Data_Param19.DataType = 'BYTE'; Port 1 Output Data_Param20.Name = 'Port 1 Output Data_Param20'; Port 1 Output Data_Param20.HelpString = ''; Port 1 Output Data_Param20.ReadOnly = False; Port 1 Output Data_Param20.BitSize = 8; Port 1 Output Data_Param20.DataSize = 1; Port 1 Output Data_Param20.DataType = 'BYTE'; Port 1 Output Data_Param21.Name = 'Port 1 Output Data_Param21'; Port 1 Output Data_Param21.HelpString = ''; Port 1 Output Data_Param21.ReadOnly = False; Port 1 Output Data_Param21.BitSize = 8; Port 1 Output Data_Param21.DataSize = 1; Port 1 Output Data_Param21.DataType = 'BYTE'; Port 1 Output Data_Param22.Name = 'Port 1 Output Data_Param22'; Port 1 Output Data_Param22.HelpString = ''; Port 1 Output Data_Param22.ReadOnly = False; Port 1 Output Data_Param22.BitSize = 8; Port 1 Output Data_Param22.DataSize = 1; Port 1 Output Data_Param22.DataType = 'BYTE'; Port 1 Output Data_Param23.Name = 'Port 1 Output Data_Param23'; Port 1 Output Data_Param23.HelpString = ''; Port 1 Output Data_Param23.ReadOnly = False; Port 1 Output Data_Param23.BitSize = 8; Port 1 Output Data_Param23.DataSize = 1; Port 1 Output Data_Param23.DataType = 'BYTE'; Port 1 Output Data_Param24.Name = 'Port 1 Output Data_Param24'; Port 1 Output Data_Param24.HelpString = ''; Port 1 Output Data_Param24.ReadOnly = False; Port 1 Output Data_Param24.BitSize = 8; Port 1 Output Data_Param24.DataSize = 1; Port 1 Output Data_Param24.DataType = 'BYTE'; Port 1 Output Data_Param25.Name = 'Port 1 Output Data_Param25'; Port 1 Output Data_Param25.HelpString = ''; Port 1 Output Data_Param25.ReadOnly = False;
            Port 1 Output Data_Param25.BitSize = 8; Port 1 Output Data_Param25.DataSize = 1; Port 1 Output Data_Param25.DataType = 'BYTE'; Port 1 Output Data_Param26.Name = 'Port 1 Output Data_Param26'; Port 1 Output Data_Param26.HelpString = ''; Port 1 Output Data_Param26.ReadOnly = False; Port 1 Output Data_Param26.BitSize = 8; Port 1 Output Data_Param26.DataSize = 1; Port 1 Output Data_Param26.DataType = 'BYTE'; Port 1 Output Data_Param27.Name = 'Port 1 Output Data_Param27'; Port 1 Output Data_Param27.HelpString = ''; Port 1 Output Data_Param27.ReadOnly = False; Port 1 Output Data_Param27.BitSize = 8; Port 1 Output Data_Param27.DataSize = 1; Port 1 Output Data_Param27.DataType = 'BYTE'; Port 1 Output Data_Param28.Name = 'Port 1 Output Data_Param28'; Port 1 Output Data_Param28.HelpString = ''; Port 1 Output Data_Param28.ReadOnly = False; Port 1 Output Data_Param28.BitSize = 8; Port 1 Output Data_Param28.DataSize = 1; Port 1 Output Data_Param28.DataType = 'BYTE'; Port 1 Output Data_Param29.Name = 'Port 1 Output Data_Param29'; Port 1 Output Data_Param29.HelpString = ''; Port 1 Output Data_Param29.ReadOnly = False; Port 1 Output Data_Param29.BitSize = 8; Port 1 Output Data_Param29.DataSize = 1; Port 1 Output Data_Param29.DataType = 'BYTE'; Port 1 Output Data_Param30.Name = 'Port 1 Output Data_Param30'; Port 1 Output Data_Param30.HelpString = ''; Port 1 Output Data_Param30.ReadOnly = False; Port 1 Output Data_Param30.BitSize = 8; Port 1 Output Data_Param30.DataSize = 1; Port 1 Output Data_Param30.DataType = 'BYTE'; Port 1 Output Data_Param31.Name = 'Port 1 Output Data_Param31'; Port 1 Output Data_Param31.HelpString = ''; Port 1 Output Data_Param31.ReadOnly = False; Port 1 Output Data_Param31.BitSize = 8; Port 1 Output Data_Param31.DataSize = 1; Port 1 Output Data_Param31.DataType = 'BYTE'; Port 1 Input Data_Param0.Name = 'Port 1 Input Data_Param0';
            Port 1 Input Data_Param0.HelpString = ''; Port 1 Input Data_Param0.ReadOnly = False; Port 1 Input Data_Param0.BitSize = 8; Port 1 Input Data_Param0.DataSize = 1; Port 1 Input Data_Param0.DataType = 'BYTE'; Port 1 Input Data_Param1.Name = 'Port 1 Input Data_Param1'; Port 1 Input Data_Param1.HelpString = ''; Port 1 Input Data_Param1.ReadOnly = False; Port 1 Input Data_Param1.BitSize = 8; Port 1 Input Data_Param1.DataSize = 1; Port 1 Input Data_Param1.DataType = 'BYTE'; Port 1 Input Data_Param2.Name = 'Port 1 Input Data_Param2'; Port 1 Input Data_Param2.HelpString = ''; Port 1 Input Data_Param2.ReadOnly = False; Port 1 Input Data_Param2.BitSize = 8; Port 1 Input Data_Param2.DataSize = 1; Port 1 Input Data_Param2.DataType = 'BYTE'; Port 1 Input Data_Param3.Name = 'Port 1 Input Data_Param3'; Port 1 Input Data_Param3.HelpString = ''; Port 1 Input Data_Param3.ReadOnly = False; Port 1 Input Data_Param3.BitSize = 8; Port 1 Input Data_Param3.DataSize = 1; Port 1 Input Data_Param3.DataType = 'BYTE'; Port 1 Input Data_Param4.Name = 'Port 1 Input Data_Param4'; Port 1 Input Data_Param4.HelpString = ''; Port 1 Input Data_Param4.ReadOnly = False; Port 1 Input Data_Param4.BitSize = 8; Port 1 Input Data_Param4.DataSize = 1; Port 1 Input Data_Param4.DataType = 'BYTE'; Port 1 Input Data_Param5.Name = 'Port 1 Input Data_Param5'; Port 1 Input Data_Param5.HelpString = ''; Port 1 Input Data_Param5.ReadOnly = False; Port 1 Input Data_Param5.BitSize = 8; Port 1 Input Data_Param5.DataSize = 1; Port 1 Input Data_Param5.DataType = 'BYTE'; Port 1 Input Data_Param6.Name = 'Port 1 Input Data_Param6'; Port 1 Input Data_Param6.HelpString = ''; Port 1 Input Data_Param6.ReadOnly = False; Port 1 Input Data_Param6.BitSize = 8; Port 1 Input Data_Param6.DataSize = 1;
            Port 1 Input Data_Param6.DataType = 'BYTE'; Port 1 Input Data_Param7.Name = 'Port 1 Input Data_Param7'; Port 1 Input Data_Param7.HelpString = ''; Port 1 Input Data_Param7.ReadOnly = False; Port 1 Input Data_Param7.BitSize = 8; Port 1 Input Data_Param7.DataSize = 1; Port 1 Input Data_Param7.DataType = 'BYTE'; Port 1 Input Data_Param8.Name = 'Port 1 Input Data_Param8'; Port 1 Input Data_Param8.HelpString = ''; Port 1 Input Data_Param8.ReadOnly = False; Port 1 Input Data_Param8.BitSize = 8; Port 1 Input Data_Param8.DataSize = 1; Port 1 Input Data_Param8.DataType = 'BYTE'; Port 1 Input Data_Param9.Name = 'Port 1 Input Data_Param9'; Port 1 Input Data_Param9.HelpString = ''; Port 1 Input Data_Param9.ReadOnly = False; Port 1 Input Data_Param9.BitSize = 8; Port 1 Input Data_Param9.DataSize = 1; Port 1 Input Data_Param9.DataType = 'BYTE'; Port 1 Input Data_Param10.Name = 'Port 1 Input Data_Param10'; Port 1 Input Data_Param10.HelpString = ''; Port 1 Input Data_Param10.ReadOnly = False; Port 1 Input Data_Param10.BitSize = 8; Port 1 Input Data_Param10.DataSize = 1; Port 1 Input Data_Param10.DataType = 'BYTE'; Port 1 Input Data_Param11.Name = 'Port 1 Input Data_Param11'; Port 1 Input Data_Param11.HelpString = ''; Port 1 Input Data_Param11.ReadOnly = False; Port 1 Input Data_Param11.BitSize = 8; Port 1 Input Data_Param11.DataSize = 1; Port 1 Input Data_Param11.DataType = 'BYTE'; Port 1 Input Data_Param12.Name = 'Port 1 Input Data_Param12'; Port 1 Input Data_Param12.HelpString = ''; Port 1 Input Data_Param12.ReadOnly = False; Port 1 Input Data_Param12.BitSize = 8; Port 1 Input Data_Param12.DataSize = 1; Port 1 Input Data_Param12.DataType = 'BYTE'; Port 1 Input Data_Param13.Name = 'Port 1 Input Data_Param13'; Port 1 Input Data_Param13.HelpString = ''; Port 1 Input Data_Param13.ReadOnly = False;
            Port 1 Input Data_Param13.BitSize = 8; Port 1 Input Data_Param13.DataSize = 1; Port 1 Input Data_Param13.DataType = 'BYTE'; Port 1 Input Data_Param14.Name = 'Port 1 Input Data_Param14'; Port 1 Input Data_Param14.HelpString = ''; Port 1 Input Data_Param14.ReadOnly = False; Port 1 Input Data_Param14.BitSize = 8; Port 1 Input Data_Param14.DataSize = 1; Port 1 Input Data_Param14.DataType = 'BYTE'; Port 1 Input Data_Param15.Name = 'Port 1 Input Data_Param15'; Port 1 Input Data_Param15.HelpString = ''; Port 1 Input Data_Param15.ReadOnly = False; Port 1 Input Data_Param15.BitSize = 8; Port 1 Input Data_Param15.DataSize = 1; Port 1 Input Data_Param15.DataType = 'BYTE'; Port 1 Input Data_Param16.Name = 'Port 1 Input Data_Param16'; Port 1 Input Data_Param16.HelpString = ''; Port 1 Input Data_Param16.ReadOnly = False; Port 1 Input Data_Param16.BitSize = 8; Port 1 Input Data_Param16.DataSize = 1; Port 1 Input Data_Param16.DataType = 'BYTE'; Port 1 Input Data_Param17.Name = 'Port 1 Input Data_Param17'; Port 1 Input Data_Param17.HelpString = ''; Port 1 Input Data_Param17.ReadOnly = False; Port 1 Input Data_Param17.BitSize = 8; Port 1 Input Data_Param17.DataSize = 1; Port 1 Input Data_Param17.DataType = 'BYTE'; Port 1 Input Data_Param18.Name = 'Port 1 Input Data_Param18'; Port 1 Input Data_Param18.HelpString = ''; Port 1 Input Data_Param18.ReadOnly = False; Port 1 Input Data_Param18.BitSize = 8; Port 1 Input Data_Param18.DataSize = 1; Port 1 Input Data_Param18.DataType = 'BYTE'; Port 1 Input Data_Param19.Name = 'Port 1 Input Data_Param19'; Port 1 Input Data_Param19.HelpString = ''; Port 1 Input Data_Param19.ReadOnly = False; Port 1 Input Data_Param19.BitSize = 8; Port 1 Input Data_Param19.DataSize = 1; Port 1 Input Data_Param19.DataType = 'BYTE'; Port 1 Input Data_Param20.Name = 'Port 1 Input Data_Param20';
            Port 1 Input Data_Param20.HelpString = ''; Port 1 Input Data_Param20.ReadOnly = False; Port 1 Input Data_Param20.BitSize = 8; Port 1 Input Data_Param20.DataSize = 1; Port 1 Input Data_Param20.DataType = 'BYTE'; Port 1 Input Data_Param21.Name = 'Port 1 Input Data_Param21'; Port 1 Input Data_Param21.HelpString = ''; Port 1 Input Data_Param21.ReadOnly = False; Port 1 Input Data_Param21.BitSize = 8; Port 1 Input Data_Param21.DataSize = 1; Port 1 Input Data_Param21.DataType = 'BYTE'; Port 1 Input Data_Param22.Name = 'Port 1 Input Data_Param22'; Port 1 Input Data_Param22.HelpString = ''; Port 1 Input Data_Param22.ReadOnly = False; Port 1 Input Data_Param22.BitSize = 8; Port 1 Input Data_Param22.DataSize = 1; Port 1 Input Data_Param22.DataType = 'BYTE'; Port 1 Input Data_Param23.Name = 'Port 1 Input Data_Param23'; Port 1 Input Data_Param23.HelpString = ''; Port 1 Input Data_Param23.ReadOnly = False; Port 1 Input Data_Param23.BitSize = 8; Port 1 Input Data_Param23.DataSize = 1; Port 1 Input Data_Param23.DataType = 'BYTE'; Port 1 Input Data_Param24.Name = 'Port 1 Input Data_Param24'; Port 1 Input Data_Param24.HelpString = ''; Port 1 Input Data_Param24.ReadOnly = False; Port 1 Input Data_Param24.BitSize = 8; Port 1 Input Data_Param24.DataSize = 1; Port 1 Input Data_Param24.DataType = 'BYTE'; Port 1 Input Data_Param25.Name = 'Port 1 Input Data_Param25'; Port 1 Input Data_Param25.HelpString = ''; Port 1 Input Data_Param25.ReadOnly = False; Port 1 Input Data_Param25.BitSize = 8; Port 1 Input Data_Param25.DataSize = 1; Port 1 Input Data_Param25.DataType = 'BYTE'; Port 1 Input Data_Param26.Name = 'Port 1 Input Data_Param26'; Port 1 Input Data_Param26.HelpString = ''; Port 1 Input Data_Param26.ReadOnly = False; Port 1 Input Data_Param26.BitSize = 8; Port 1 Input Data_Param26.DataSize = 1;
            Port 1 Input Data_Param26.DataType = 'BYTE'; Port 1 Input Data_Param27.Name = 'Port 1 Input Data_Param27'; Port 1 Input Data_Param27.HelpString = ''; Port 1 Input Data_Param27.ReadOnly = False; Port 1 Input Data_Param27.BitSize = 8; Port 1 Input Data_Param27.DataSize = 1; Port 1 Input Data_Param27.DataType = 'BYTE'; Port 1 Input Data_Param28.Name = 'Port 1 Input Data_Param28'; Port 1 Input Data_Param28.HelpString = ''; Port 1 Input Data_Param28.ReadOnly = False; Port 1 Input Data_Param28.BitSize = 8; Port 1 Input Data_Param28.DataSize = 1; Port 1 Input Data_Param28.DataType = 'BYTE'; Port 1 Input Data_Param29.Name = 'Port 1 Input Data_Param29'; Port 1 Input Data_Param29.HelpString = ''; Port 1 Input Data_Param29.ReadOnly = False; Port 1 Input Data_Param29.BitSize = 8; Port 1 Input Data_Param29.DataSize = 1; Port 1 Input Data_Param29.DataType = 'BYTE'; Port 1 Input Data_Param30.Name = 'Port 1 Input Data_Param30'; Port 1 Input Data_Param30.HelpString = ''; Port 1 Input Data_Param30.ReadOnly = False; Port 1 Input Data_Param30.BitSize = 8; Port 1 Input Data_Param30.DataSize = 1; Port 1 Input Data_Param30.DataType = 'BYTE'; Port 1 Input Data_Param31.Name = 'Port 1 Input Data_Param31'; Port 1 Input Data_Param31.HelpString = ''; Port 1 Input Data_Param31.ReadOnly = False; Port 1 Input Data_Param31.BitSize = 8; Port 1 Input Data_Param31.DataSize = 1; Port 1 Input Data_Param31.DataType = 'BYTE'; ConfigVersion = 50660864
          input  iPAPrintEnginePower : BOOL  // Port 1 Output Data_Param0.Bit0
          input  iPAPrintEngineError : BOOL  // Port 1 Output Data_Param0.Bit1
          input  iPARibbonLow : BOOL  // Port 1 Output Data_Param0.Bit2
          input  iPALabelOut : BOOL  // Port 1 Output Data_Param0.Bit3
          input  iPAOnlineDataReady : BOOL  // Port 1 Output Data_Param0.Bit4
          input  iPARibbonOut : BOOL  // Port 1 Output Data_Param0.Bit5
          input  iPAFaulted : BOOL  // Port 1 Output Data_Param0.Bit7
          input  iPACycleComplete : BOOL  // Port 1 Output Data_Param1.Bit0
          input  iPAApplicatorHome : BOOL  // Port 1 Output Data_Param1.Bit1
          input  iPALowLabels : BOOL  // Port 1 Output Data_Param1.Bit2
          input  iPALOTAR : BOOL  // Port 1 Output Data_Param1.Bit3
          input  iPABypassOn : BOOL  // Port 1 Output Data_Param1.Bit6
          input  iPAHeartbeat : BOOL  // Port 1 Output Data_Param1.Bit7
          output oPATrigger1 : BOOL  // Port 1 Input Data_Param0.Bit0
          output oPAReset : BOOL  // Port 1 Input Data_Param0.Bit2
          output oPABypassEnable : BOOL  // Port 1 Input Data_Param0.Bit3
          unmapped channels: Port 1 Output Data_Param0, Port 1 Output Data_Param1, Port 1 Output Data_Param2, Port 1 Output Data_Param3, Port 1 Output Data_Param4, Port 1 Output Data_Param5, Port 1 Output Data_Param6, Port 1 Output Data_Param7, Port 1 Output Data_Param8, Port 1 Output Data_Param9, Port 1 Output Data_Param10, Port 1 Output Data_Param11, Port 1 Output Data_Param12, Port 1 Output Data_Param13, Port 1 Output Data_Param14, Port 1 Output Data_Param15, Port 1 Output Data_Param16, Port 1 Output Data_Param17, Port 1 Output Data_Param18, Port 1 Output Data_Param19, Port 1 Output Data_Param20, Port 1 Output Data_Param21, Port 1 Output Data_Param22, Port 1 Output Data_Param23, Port 1 Output Data_Param24, Port 1 Output Data_Param25, Port 1 Output Data_Param26, Port 1 Output Data_Param27, Port 1 Output Data_Param28, Port 1 Output Data_Param29, Port 1 Output Data_Param30, Port 1 Output Data_Param31, Port 1 Input Data_Param0, Port 1 Input Data_Param1, Port 1 Input Data_Param2, Port 1 Input Data_Param3, Port 1 Input Data_Param4, Port 1 Input Data_Param5, Port 1 Input Data_Param6, Port 1 Input Data_Param7,
            Port 1 Input Data_Param8, Port 1 Input Data_Param9, Port 1 Input Data_Param10, Port 1 Input Data_Param11, Port 1 Input Data_Param12, Port 1 Input Data_Param13, Port 1 Input Data_Param14, Port 1 Input Data_Param15, Port 1 Input Data_Param16, Port 1 Input Data_Param17, Port 1 Input Data_Param18, Port 1 Input Data_Param19, Port 1 Input Data_Param20, Port 1 Input Data_Param21, Port 1 Input Data_Param22, Port 1 Input Data_Param23, Port 1 Input Data_Param24, Port 1 Input Data_Param25, Port 1 Input Data_Param26, Port 1 Input Data_Param27, Port 1 Input Data_Param28, Port 1 Input Data_Param29, Port 1 Input Data_Param30, Port 1 Input Data_Param31
      Pbar_ServoEIP : SSM23IP-3EG, Applied Motion Products, Inc, order no. SSM23IP-3EG, version Major Revision=16#3, Minor Revision = 16#3
          settings: INITIALIZED = TRUE; IP address of Target = [16#C0,16#A8,16#0A,16#34]; Keying.Check Vendor Code = FALSE; Keying.Check Product Code = FALSE; Keying.Check Major Revision = FALSE; Keying.Check Minor Revision = FALSE; RequiredConfigVersion = 50660864; Number of Connections = 1; Connection Settings.Requested packet intervall = 10000 µs; Connection Settings.OT Connection Parameters = 18502; Connection Settings.TO Connection Parameters = 18490; Connection Settings.Connection Flags = 1056; Connection Settings.Connection Path Size = 8; Connection Settings.Large OT Connection Parameters = 1207959622; Connection Settings.Large TO Connection Parameters = 1207959610; Heartbeat Multiplier = 1; Status Code.ReadOnly = False; Status Code.BitSize = 32; Status Code.DataSize = 4; Alarm Code.ReadOnly = False; Alarm Code.BitSize = 32; Alarm Code.DataSize = 4; Supply Voltage.ReadOnly = False; Supply Voltage.BitSize = 32; Supply Voltage.DataSize = 4; Actual Current.ReadOnly = False; Actual Current.BitSize = 32; Actual Current.DataSize = 4; Drive Temperature.ReadOnly = False; Drive Temperature.BitSize = 32; Drive Temperature.DataSize = 4; Encoder Position.ReadOnly = False; Encoder Position.BitSize = 32; Encoder Position.DataSize = 4; Absolute Position.ReadOnly = False; Absolute Position.BitSize = 32; Absolute Position.DataSize = 4; Position Error.ReadOnly = False; Position Error.BitSize = 32; Position Error.DataSize = 4;
            Actual Velocity.ReadOnly = False; Actual Velocity.BitSize = 32; Actual Velocity.DataSize = 4; Input Status (extended).ReadOnly = False; Input Status (extended).BitSize = 32; Input Status (extended).DataSize = 4; Input Status (main).ReadOnly = False; Input Status (main).BitSize = 32; Input Status (main).DataSize = 4; Output Status.ReadOnly = False; Output Status.BitSize = 32; Output Status.DataSize = 4; Analog Input 1.ReadOnly = False; Analog Input 1.BitSize = 32; Analog Input 1.DataSize = 4; Analog Input 2.ReadOnly = False; Analog Input 2.BitSize = 32; Analog Input 2.DataSize = 4; Command Word.ReadOnly = False; Command Word.BitSize = 32; Command Word.DataSize = 4; Jog Speed.ReadOnly = False; Jog Speed.BitSize = 32; Jog Speed.DataSize = 4; Jog Accel.ReadOnly = False; Jog Accel.BitSize = 32; Jog Accel.DataSize = 4; Jog Decel.ReadOnly = False; Jog Decel.BitSize = 32; Jog Decel.DataSize = 4; Point-to-Point Velocity.ReadOnly = False; Point-to-Point Velocity.BitSize = 32; Point-to-Point Velocity.DataSize = 4; Point-to-Point Acceleration.ReadOnly = False; Point-to-Point Acceleration.BitSize = 32; Point-to-Point Acceleration.DataSize = 4; Point-to-Point Deceleration.ReadOnly = False; Point-to-Point Deceleration.BitSize = 32; Point-to-Point Deceleration.DataSize = 4; Point-to-Point Distance.ReadOnly = False;
            Point-to-Point Distance.BitSize = 32; Point-to-Point Distance.DataSize = 4; Current Command.ReadOnly = False; Current Command.BitSize = 32; Current Command.DataSize = 4; SCL Command Letters.ReadOnly = False; SCL Command Letters.BitSize = 32; SCL Command Letters.DataSize = 4; Data/SCL Register 1.ReadOnly = False; Data/SCL Register 1.BitSize = 32; Data/SCL Register 1.DataSize = 4; Data/SCL Register 2.ReadOnly = False; Data/SCL Register 2.BitSize = 32; Data/SCL Register 2.DataSize = 4; Reserved 1.ReadOnly = False; Reserved 1.BitSize = 32; Reserved 1.DataSize = 4; Reserved 2.ReadOnly = False; Reserved 2.BitSize = 32; Reserved 2.DataSize = 4; Reserved 3.ReadOnly = False; Reserved 3.BitSize = 32; Reserved 3.DataSize = 4; Reserved 4.ReadOnly = False; Reserved 4.BitSize = 32; Reserved 4.DataSize = 4; Status Code.Name = 'Status Code'; Status Code.HelpString = ''; Status Code.ReadOnly = False; Status Code.BitSize = 32; Status Code.DataSize = 4; Status Code.DataType = 'DINT'; Alarm Code.Name = 'Alarm Code'; Alarm Code.HelpString = ''; Alarm Code.ReadOnly = False; Alarm Code.BitSize = 32; Alarm Code.DataSize = 4; Alarm Code.DataType = 'DINT'; Supply Voltage.Name = 'Supply Voltage'; Supply Voltage.HelpString = '';
            Supply Voltage.ReadOnly = False; Supply Voltage.BitSize = 32; Supply Voltage.DataSize = 4; Supply Voltage.DataType = 'DINT'; Actual Current.Name = 'Actual Current'; Actual Current.HelpString = ''; Actual Current.ReadOnly = False; Actual Current.BitSize = 32; Actual Current.DataSize = 4; Actual Current.DataType = 'DINT'; Drive Temperature.Name = 'Drive Temperature'; Drive Temperature.HelpString = ''; Drive Temperature.ReadOnly = False; Drive Temperature.BitSize = 32; Drive Temperature.DataSize = 4; Drive Temperature.DataType = 'DINT'; Encoder Position.Name = 'Encoder Position'; Encoder Position.HelpString = ''; Encoder Position.ReadOnly = False; Encoder Position.BitSize = 32; Encoder Position.DataSize = 4; Encoder Position.DataType = 'DINT'; Absolute Position.Name = 'Absolute Position'; Absolute Position.HelpString = ''; Absolute Position.ReadOnly = False; Absolute Position.BitSize = 32; Absolute Position.DataSize = 4; Absolute Position.DataType = 'DINT'; Position Error.Name = 'Position Error'; Position Error.HelpString = ''; Position Error.ReadOnly = False; Position Error.BitSize = 32; Position Error.DataSize = 4; Position Error.DataType = 'DINT'; Actual Velocity.Name = 'Actual Velocity'; Actual Velocity.HelpString = ''; Actual Velocity.ReadOnly = False; Actual Velocity.BitSize = 32; Actual Velocity.DataSize = 4; Actual Velocity.DataType = 'DINT';
            Input Status (extended).Name = 'Input Status (extended)'; Input Status (extended).HelpString = ''; Input Status (extended).ReadOnly = False; Input Status (extended).BitSize = 32; Input Status (extended).DataSize = 4; Input Status (extended).DataType = 'DINT'; Input Status (main).Name = 'Input Status (main)'; Input Status (main).HelpString = ''; Input Status (main).ReadOnly = False; Input Status (main).BitSize = 32; Input Status (main).DataSize = 4; Input Status (main).DataType = 'DINT'; Output Status.Name = 'Output Status'; Output Status.HelpString = ''; Output Status.ReadOnly = False; Output Status.BitSize = 32; Output Status.DataSize = 4; Output Status.DataType = 'DINT'; Analog Input 1.Name = 'Analog Input 1'; Analog Input 1.HelpString = ''; Analog Input 1.ReadOnly = False; Analog Input 1.BitSize = 32; Analog Input 1.DataSize = 4; Analog Input 1.DataType = 'DINT'; Analog Input 2.Name = 'Analog Input 2'; Analog Input 2.HelpString = ''; Analog Input 2.ReadOnly = False; Analog Input 2.BitSize = 32; Analog Input 2.DataSize = 4; Analog Input 2.DataType = 'DINT'; Command Word.Name = 'Command Word'; Command Word.HelpString = ''; Command Word.ReadOnly = False; Command Word.BitSize = 32; Command Word.DataSize = 4; Command Word.DataType = 'DINT'; Jog Speed.Name = 'Jog Speed'; Jog Speed.HelpString = ''; Jog Speed.ReadOnly = False; Jog Speed.BitSize = 32;
            Jog Speed.DataSize = 4; Jog Speed.DataType = 'DINT'; Jog Accel.Name = 'Jog Accel'; Jog Accel.HelpString = ''; Jog Accel.ReadOnly = False; Jog Accel.BitSize = 32; Jog Accel.DataSize = 4; Jog Accel.DataType = 'DINT'; Jog Decel.Name = 'Jog Decel'; Jog Decel.HelpString = ''; Jog Decel.ReadOnly = False; Jog Decel.BitSize = 32; Jog Decel.DataSize = 4; Jog Decel.DataType = 'DINT'; Point-to-Point Velocity.Name = 'Point-to-Point Velocity'; Point-to-Point Velocity.HelpString = ''; Point-to-Point Velocity.ReadOnly = False; Point-to-Point Velocity.BitSize = 32; Point-to-Point Velocity.DataSize = 4; Point-to-Point Velocity.DataType = 'DINT'; Point-to-Point Acceleration.Name = 'Point-to-Point Acceleration'; Point-to-Point Acceleration.HelpString = ''; Point-to-Point Acceleration.ReadOnly = False; Point-to-Point Acceleration.BitSize = 32; Point-to-Point Acceleration.DataSize = 4; Point-to-Point Acceleration.DataType = 'DINT'; Point-to-Point Deceleration.Name = 'Point-to-Point Deceleration'; Point-to-Point Deceleration.HelpString = ''; Point-to-Point Deceleration.ReadOnly = False; Point-to-Point Deceleration.BitSize = 32; Point-to-Point Deceleration.DataSize = 4; Point-to-Point Deceleration.DataType = 'DINT'; Point-to-Point Distance.Name = 'Point-to-Point Distance'; Point-to-Point Distance.HelpString = ''; Point-to-Point Distance.ReadOnly = False; Point-to-Point Distance.BitSize = 32; Point-to-Point Distance.DataSize = 4; Point-to-Point Distance.DataType = 'DINT'; Current Command.Name = 'Current Command'; Current Command.HelpString = '';
            Current Command.ReadOnly = False; Current Command.BitSize = 32; Current Command.DataSize = 4; Current Command.DataType = 'DINT'; SCL Command Letters.Name = 'SCL Command Letters'; SCL Command Letters.HelpString = ''; SCL Command Letters.ReadOnly = False; SCL Command Letters.BitSize = 32; SCL Command Letters.DataSize = 4; SCL Command Letters.DataType = 'DINT'; Data/SCL Register 1.Name = 'Data/SCL Register 1'; Data/SCL Register 1.HelpString = ''; Data/SCL Register 1.ReadOnly = False; Data/SCL Register 1.BitSize = 32; Data/SCL Register 1.DataSize = 4; Data/SCL Register 1.DataType = 'DINT'; Data/SCL Register 2.Name = 'Data/SCL Register 2'; Data/SCL Register 2.HelpString = ''; Data/SCL Register 2.ReadOnly = False; Data/SCL Register 2.BitSize = 32; Data/SCL Register 2.DataSize = 4; Data/SCL Register 2.DataType = 'DINT'; Reserved 1.Name = 'Reserved 1'; Reserved 1.HelpString = ''; Reserved 1.ReadOnly = False; Reserved 1.BitSize = 32; Reserved 1.DataSize = 4; Reserved 1.DataType = 'DINT'; Reserved 2.Name = 'Reserved 2'; Reserved 2.HelpString = ''; Reserved 2.ReadOnly = False; Reserved 2.BitSize = 32; Reserved 2.DataSize = 4; Reserved 2.DataType = 'DINT'; Reserved 3.Name = 'Reserved 3'; Reserved 3.HelpString = ''; Reserved 3.ReadOnly = False; Reserved 3.BitSize = 32; Reserved 3.DataSize = 4; Reserved 3.DataType = 'DINT';
            Reserved 4.Name = 'Reserved 4'; Reserved 4.HelpString = ''; Reserved 4.ReadOnly = False; Reserved 4.BitSize = 32; Reserved 4.DataSize = 4; Reserved 4.DataType = 'DINT'; ConfigVersion = 50660864
          input  jawPasstrhoughMotorInputs : DINT  // Status Code
          input  iPassthroughHomeSensorClear : BOOL  // Input Status (main).Bit2
          output jawPasstrhoughMotorOutputs : DINT  // Command Word
          unmapped channels: Alarm Code, Supply Voltage, Actual Current, Drive Temperature, Encoder Position, Absolute Position, Position Error, Actual Velocity, Input Status (extended), Input Status (main), Output Status, Analog Input 1, Analog Input 2, Jog Speed, Jog Accel, Jog Decel, Point-to-Point Velocity, Point-to-Point Acceleration, Point-to-Point Deceleration, Point-to-Point Distance, Current Command, SCL Command Letters, Data/SCL Register 1, Data/SCL Register 2, Reserved 1, Reserved 2, Reserved 3, Reserved 4
    Ethernet : Ethernet, 3S - Smart Software Solutions GmbH, version 3.5.13.0
        settings: IPAddress = [192,168,10,20]; SubnetMask = [255,255,255,0]; GatewayAddress = [192,168,10,254]; NetworkInterfaceName = 'Machine LAN:2'; NetworkInterfaceName = "Machine LAN:2"; SaveCommunicationSettings = FALSE
      ModbusTCP_Slave_Device : ModbusTCP Slave Device, 3S - Smart Software Solutions GmbH, version 4.2.0.0 (disabled)
          input  Application.RemoteComms.modbusInputsToBagger.fillerTrigger : BOOL  // Holding Registers.Holding Registers.Bit0
          input  Application.RemoteComms.modbusInputsToBagger.baggerInhibit : BOOL  // Holding Registers.Holding Registers.Bit1
          input  Application.RemoteComms.modbusInputsToBagger.collisionDetection : BOOL  // Holding Registers.Holding Registers.Bit2
          input  Application.RemoteComms.modbusInputsToBagger.fillerOK : BOOL  // Holding Registers.Holding Registers.Bit3
          input  Application.RemoteComms.modbusInputsToBagger.reverseConveyor : BOOL  // Holding Registers.Holding Registers.Bit4
          input  Application.RemoteComms.modbusInputsToBagger.bagGrabbed : BOOL  // Holding Registers.Holding Registers.Bit5
          input  Application.RemoteComms.modbusInputsToBagger.heartbeat : BOOL  // Holding Registers.Holding Registers.Bit6
          output Application.RemoteComms.modbusOutputsFromBagger.baggerOK : BOOL  // Input Registers.Input Registers.Bit0
          output Application.RemoteComms.modbusOutputsFromBagger.readyForFiller : BOOL  // Input Registers.Input Registers.Bit1
          output Application.RemoteComms.modbusOutputsFromBagger.printerDataReady : BOOL  // Input Registers.Input Registers.Bit2
          output Application.RemoteComms.modbusOutputsFromBagger.waitingForPrinter : BOOL  // Input Registers.Input Registers.Bit3
          output Application.RemoteComms.modbusOutputsFromBagger.cycleComplete : BOOL  // Input Registers.Input Registers.Bit4
          output Application.RemoteComms.modbusOutputsFromBagger.bagMade : BOOL  // Input Registers.Input Registers.Bit5
          output Application.RemoteComms.modbusOutputsFromBagger.bagMadePlusLabelRequired : BOOL  // Input Registers.Input Registers.Bit6
          output Application.RemoteComms.modbusOutputsFromBagger.bagsLow : BOOL  // Input Registers.Input Registers.Bit7
          output Application.RemoteComms.modbusOutputsFromBagger.readyForGrab : BOOL  // Input Registers.Input Registers.Bit8
          output Application.RemoteComms.modbusOutputsFromBagger.runExternalExitConveyor : BOOL  // Input Registers.Input Registers.Bit9
          output Application.RemoteComms.modbusOutputsFromBagger.heartbeatResponse : BOOL  // Input Registers.Input Registers.Bit10
          unmapped channels: Holding Registers, Input Registers
    System_Diagnosis : System Diagnosis, Advantech Co., Ltd., version 3.5.13.0
        unmapped channels: System Information
  SX_1179_01 : CVS GN-9372(PIO), CREVIS CO.,LTD, order no. GN-9372,PIO, version 3.5.11.3
    application Application
    CVS_G_Series_Rack_ : CVS G-Series(Rack), CREVIS CO.,LTD, version 1.0.0.0
      <Empty>
      <Empty>
      <Empty>
      <Empty>
      <Empty>
      <Empty>
      <Empty>
      <Empty>
      <Empty>
      <Empty>
      <Empty>
      <Empty>
      <Empty>
      <Empty>
      <Empty>
      <Empty>
      <Empty>
      <Empty>
      <Empty>
      <Empty>
      <Empty>
      <Empty>
      <Empty>
      <Empty>
      <Empty>
      <Empty>
      <Empty>
      <Empty>
      <Empty>
      <Empty>
      <Empty>
      <Empty>
      <Empty>
      <Empty>
      <Empty>
      <Empty>
      <Empty>
      <Empty>
      <Empty>
      <Empty>
      <Empty>
      <Empty>
      <Empty>
      <Empty>
      <Empty>
      <Empty>
      <Empty>
      <Empty>
      <Empty>
      <Empty>
      <Empty>
      <Empty>
      <Empty>
      <Empty>
      <Empty>
      <Empty>
      <Empty>
      <Empty>
      <Empty>
      <Empty>
      GT_5231 : GT-5231, CREVIS CO.,LTD, order no. GT-5231, version 1.0.0.0
          settings: Serial Setting = 2#00000101; Data Bit Setting = 60
          input  serialInputs : BYTE  // IN0
          output serialOutputs : BYTE  // OUT0
          unmapped channels: IN1, IN2, IN3, IN4, IN5, IN6, IN7, IN8, IN9, IN10, IN11, IN12, IN13, IN14, IN15, IN16, IN17, IN18, IN19, IN20, IN21, IN22, IN23, IN24, IN25, IN26, IN27, IN28, IN29, IN30, IN31, IN32, IN33, IN34, IN35, IN36, IN37, IN38, IN39, IN40,
            IN41, IN42, IN43, IN44, IN45, IN46, IN47, IN48, IN49, IN50, IN51, IN52, IN53, IN54, IN55, IN56, IN57, IN58, IN59, IN60, IN61, IN62, OUT1, OUT2, OUT3, OUT4, OUT5, OUT6, OUT7, OUT8, OUT9, OUT10, OUT11, OUT12, OUT13, OUT14, OUT15, OUT16, OUT17, OUT18,
            OUT19, OUT20, OUT21, OUT22, OUT23, OUT24, OUT25, OUT26, OUT27, OUT28, OUT29, OUT30, OUT31, OUT32, OUT33, OUT34, OUT35, OUT36, OUT37, OUT38, OUT39, OUT40, OUT41, OUT42, OUT43, OUT44, OUT45, OUT46, OUT47, OUT48, OUT49, OUT50, OUT51, OUT52, OUT53, OUT54, OUT55, OUT56, OUT57, OUT58,
            OUT59, OUT60, OUT61, OUT62
      InputSlot0 : GT-12DF, CREVIS CO.,LTD, order no. GT-12DF, version 1.0.0.0
          input  iJawNotObstructed : BOOL  // IN0.BIT0
          input  iPrinterDataReady : BOOL  // IN0.BIT1
          input  iPrinterBusy : BOOL  // IN0.BIT2
          input  iBagEdgePhotoeye : BOOL  // IN0.BIT3
          input  iCycleStart : BOOL  // IN0.BIT4
          input  iPrintHeadLowered : BOOL  // IN0.BIT5
          input  iJawClosed : BOOL  // IN0.BIT6
          input  iJawNearClosed : BOOL  // IN0.BIT7
          input  iBarcodeOK : BOOL  // IN1.BIT0
          input  iBarcodeNG : BOOL  // IN1.BIT1
          input  iLightCurtain : BOOL  // IN1.BIT2
          input  iFillerTrigger : BOOL  // IN1.BIT3
          input  iLHPalmButton : BOOL  // IN1.BIT4
          input  iRHPalmButton : BOOL  // IN1.BIT5
          input  iTopCoverClosed : BOOL  // IN1.BIT6
          input  iPrinterRibbonEncoder : BOOL  // IN1.BIT7
          unmapped channels: IN0, IN1
      InputSlot2 : GT-12DF, CREVIS CO.,LTD, order no. GT-12DF, version 1.0.0.0
          input  iPrinterServiceRequired : BOOL  // IN0.BIT0
          unmapped channels: IN0, IN1
      OutputSlot1 : GT-226F, CREVIS CO.,LTD, order no. GT-226F, version 1.0.0.0
          output oSealWire : BOOL  // OUT0.BIT0
          output oLowerPrintHead : BOOL  // OUT0.BIT1
          output oRequestPrint : BOOL  // OUT0.BIT2
          output oPrinterRibbonUnwind : BOOL  // OUT0.BIT3
          output oTriggerBCV : BOOL  // OUT0.BIT4
          output oTeachPhotoeye : BOOL  // OUT0.BIT5
          output oRedStackLight : BOOL  // OUT0.BIT6
          output oGreenStackLight : BOOL  // OUT0.BIT7
          output oReadyForFiller : BOOL  // OUT1.BIT0
          output oPalmButton0 : BOOL  // OUT1.BIT1
          output oPalmButton1 : BOOL  // OUT1.BIT2
          unmapped channels: OUT0, OUT1
    Ethernet : Ethernet, 3S - Smart Software Solutions GmbH, version 3.5.11.0
        settings: IPAddress = [192,168,10,20]; SubnetMask = [255,255,255,0]; GatewayAddress = [0,0,0,0]; NetworkInterfaceName = 'Ethernet 0'; NetworkInterfaceName = "Ethernet 0"; SaveCommunicationSettings = TRUE
    Modbus_COM : Modbus COM, 3S - Smart Software Solutions GmbH, version 3.5.11.20
        settings: ComPort = 2
      MBMasterCOMPort : Modbus Master, COM Port, 3S - Smart Software Solutions GmbH, version 3.5.11.20
          settings: TimeBetweenFrames = 5; Auto-restart communication = TRUE
  SX_1179_02 : X2 control 4 - Powerfail, Beijer Electronics Products AB, order no. 
      , version 3.5.13.30
    application Application
    ECATMasterPort1 : EtherCAT Master, 3S - Smart Software Solutions GmbH, version 3.5.13.20
        settings: SlaveAutoRestart = True; NetworkName = 'LAN A'; NetworkName = "LAN A"; SelectNetworkByName = True; SrcAddress1 = 80; SrcAddress2 = 1812439021
      GL_9086_Crevis : GL-9086 EtherCAT Adapter, Crevis, Crevis Co.,Ltd, order no. GL-9086,Crevis, version Revision=16#00010000
          settings: ModularDevice = True; Number of Outputs = 0; Number of Inputs = 0; Number of Infos about Outputs = 0; Number of Infos about Inputs = 0; MDP_InputOffsets = [0,0,0,16]; MDP_OutputOffsets = [0,0,0,0]; Sync.Length = 2; Sync.Length = 4; FMMU.Length = 2; FMMU.Length = 4; Number of RxPDOs of the Slave = 1; Number of TxPDOs of the Slave = 2; DC sync0 cycletime = 4000; DC sync1 cycletime = 4000; RxTxPdo.NumberofExcludes = 0; RxTxPdo.NumberofEntries = 2; RxTxPdo.Index = 16#1601; RxTxPdo.Fixed = True; RxTxPdo.Mandatory = True; RxTxPdo.Virtual = False; RxTxPdo.Sm = 2; RxTxPdo.Su = 0; RxTxPdo.Name = 'Output(s)'; RxTxPdo.DependOnSlot = True; RxTxPdo.DependOnSlotGroup = False; RxTxPdo.OverwrittenByModule = True; Byte0.Index = 16#7010; Byte0.SubIndex = 1; Byte0.Size = 8; Byte0.Offset = 0; Byte0.DependOnSlot = True; Byte0.DependOnSlotGroup = False; Byte1.Index = 16#7010; Byte1.SubIndex = 2; Byte1.Size = 8; Byte1.Offset = 0; Byte1.DependOnSlot = True; Byte1.DependOnSlotGroup = False; RxTxPdo.NumberofExcludes = 0;
            RxTxPdo.NumberofEntries = 2; RxTxPdo.Index = 16#1A00; RxTxPdo.Fixed = True; RxTxPdo.Mandatory = True; RxTxPdo.Virtual = False; RxTxPdo.Sm = 3; RxTxPdo.Su = 0; RxTxPdo.Name = 'Input(s)'; RxTxPdo.DependOnSlot = True; RxTxPdo.DependOnSlotGroup = False; RxTxPdo.OverwrittenByModule = True; Byte0.Index = 16#6000; Byte0.SubIndex = 1; Byte0.Size = 8; Byte0.Offset = 0; Byte0.DependOnSlot = True; Byte0.DependOnSlotGroup = False; Byte1.Index = 16#6000; Byte1.SubIndex = 2; Byte1.Size = 8; Byte1.Offset = 0; Byte1.DependOnSlot = True; Byte1.DependOnSlotGroup = False; RxTxPdo.NumberofExcludes = 0; RxTxPdo.NumberofEntries = 2; RxTxPdo.Index = 16#1A02; RxTxPdo.Fixed = True; RxTxPdo.Mandatory = True; RxTxPdo.Virtual = False; RxTxPdo.Sm = 3; RxTxPdo.Su = 0; RxTxPdo.Name = 'Input(s)'; RxTxPdo.DependOnSlot = True; RxTxPdo.DependOnSlotGroup = False; RxTxPdo.OverwrittenByModule = True; Byte0.Index = 16#6020; Byte0.SubIndex = 1; Byte0.Size = 8; Byte0.Offset = 0; Byte0.DependOnSlot = True;
            Byte0.DependOnSlotGroup = False; Byte1.Index = 16#6020; Byte1.SubIndex = 2; Byte1.Size = 8; Byte1.Offset = 0; Byte1.DependOnSlot = True; Byte1.DependOnSlotGroup = False; Byte0.Name = 'Byte0'; Byte0.DataType = 'USINT'; Byte0.Default = ''; Byte0.Comment = ''; Byte1.Name = 'Byte1'; Byte1.DataType = 'USINT'; Byte1.Default = ''; Byte1.Comment = ''; Byte0.Name = 'Byte0'; Byte0.DataType = 'USINT'; Byte0.Default = ''; Byte0.Comment = ''; Byte1.Name = 'Byte1'; Byte1.DataType = 'USINT'; Byte1.Default = ''; Byte1.Comment = ''; Byte0.Name = 'Byte0'; Byte0.DataType = 'USINT'; Byte0.Default = ''; Byte0.Comment = ''; Byte1.Name = 'Byte1'; Byte1.DataType = 'USINT'; Byte1.Default = ''; Byte1.Comment = ''
    MBCOMPort2 : Modbus COM, 3S - Smart Software Solutions GmbH, version 3.5.11.20
        settings: DataBits = 8; StopBits = 1; ComPort = 2
      MBMasterCOMPort2 : Modbus Master, COM Port, 3S - Smart Software Solutions GmbH, version 3.5.11.20
          settings: Auto-restart communication = TRUE
    MBCOMPort3 : Modbus COM, 3S - Smart Software Solutions GmbH, version 3.5.11.20
        settings: DataBits = 8; StopBits = 1; ComPort = 3
      MBMasterCOMPort3 : Modbus Master, COM Port, 3S - Smart Software Solutions GmbH, version 3.5.11.20
          settings: TimeBetweenFrames = 5; Auto-restart communication = TRUE
  SX_1195 : X2 control 4 - Powerfail, Beijer Electronics Products AB, order no. 
      , version 3.5.13.30
    application Application
    Ethercat_Master : EtherCAT Master, 3S - Smart Software Solutions GmbH, version 3.5.11.10
        settings: SlaveAutoRestart = True; NetworkName = 'LAN A'; NetworkName = "LAN A"; SelectNetworkByName = True; SrcAddress1 = 80; SrcAddress2 = 1812439021
      AZD4A_KED : AZD2A-KED rev0301, ORIENTAL MOTOR CO.,LTD., order no. AZD2A-KED, version Revision=16#00110301
          settings: Number of Outputs = 18; Number of Inputs = 18; Number of Infos about Outputs = 18; Number of Infos about Inputs = 18; EnableExpertSettings = True; Sync.Length = 48; Sync.Length = 48; FMMU.Length = 48; FMMU.Length = 48; Number of RxPDOs of the Slave = 3; Number of TxPDOs of the Slave = 3; DC sync0 cycletime = 4000; DC sync1 cycletime = 4000; RxTxPdo.NumberofExcludes = 0; RxTxPdo.NumberofEntries = 8; RxTxPdo.Index = 16#1600; RxTxPdo.Fixed = False; RxTxPdo.Mandatory = False; RxTxPdo.Virtual = False; RxTxPdo.Sm = 2; RxTxPdo.Su = 0; RxTxPdo.Name = 'Axis1 Receive PDO Mapping 1'; RxTxPdo.DependOnSlot = False; RxTxPdo.DependOnSlotGroup = False; RxTxPdo.OverwrittenByModule = False; Controlword.Index = 16#6040; Controlword.SubIndex = 0; Controlword.Size = 16; Controlword.Offset = 0; Controlword.DependOnSlot = False; Controlword.DependOnSlotGroup = False; Target position.Index = 16#607A; Target position.SubIndex = 0; Target position.Size = 32; Target position.Offset = 0; Target position.DependOnSlot = False; Target position.DependOnSlotGroup = False; Modes of operation.Index = 16#6060; Modes of operation.SubIndex = 0; Modes of operation.Size = 8;
            Modes of operation.Offset = 0; Modes of operation.DependOnSlot = False; Modes of operation.DependOnSlotGroup = False; Profile velocity.Index = 16#6081; Profile velocity.SubIndex = 0; Profile velocity.Size = 32; Profile velocity.Offset = 0; Profile velocity.DependOnSlot = False; Profile velocity.DependOnSlotGroup = False; Profile acceleration.Index = 16#6083; Profile acceleration.SubIndex = 0; Profile acceleration.Size = 32; Profile acceleration.Offset = 0; Profile acceleration.DependOnSlot = False; Profile acceleration.DependOnSlotGroup = False; Profile deceleration.Index = 16#6084; Profile deceleration.SubIndex = 0; Profile deceleration.Size = 32; Profile deceleration.Offset = 0; Profile deceleration.DependOnSlot = False; Profile deceleration.DependOnSlotGroup = False; Axis1 push current.Index = 16#4121; Axis1 push current.SubIndex = 1; Axis1 push current.Size = 16; Axis1 push current.Offset = 0; Axis1 push current.DependOnSlot = False; Axis1 push current.DependOnSlotGroup = False; Axis1 base current.Index = 16#4126; Axis1 base current.SubIndex = 1; Axis1 base current.Size = 16; Axis1 base current.Offset = 0; Axis1 base current.DependOnSlot = False; Axis1 base current.DependOnSlotGroup = False; RxTxPdo.NumberofExcludes = 0; RxTxPdo.NumberofEntries = 8; RxTxPdo.Index = 16#1610; RxTxPdo.Fixed = False; RxTxPdo.Mandatory = False; RxTxPdo.Virtual = False; RxTxPdo.Sm = 2;
            RxTxPdo.Su = 0; RxTxPdo.Name = 'Axis2 Receive PDO Mapping 1'; RxTxPdo.DependOnSlot = False; RxTxPdo.DependOnSlotGroup = False; RxTxPdo.OverwrittenByModule = False; Controlword.Index = 16#6840; Controlword.SubIndex = 0; Controlword.Size = 16; Controlword.Offset = 0; Controlword.DependOnSlot = False; Controlword.DependOnSlotGroup = False; Target position.Index = 16#687A; Target position.SubIndex = 0; Target position.Size = 32; Target position.Offset = 0; Target position.DependOnSlot = False; Target position.DependOnSlotGroup = False; Modes of operation.Index = 16#6860; Modes of operation.SubIndex = 0; Modes of operation.Size = 8; Modes of operation.Offset = 0; Modes of operation.DependOnSlot = False; Modes of operation.DependOnSlotGroup = False; Profile velocity.Index = 16#6881; Profile velocity.SubIndex = 0; Profile velocity.Size = 32; Profile velocity.Offset = 0; Profile velocity.DependOnSlot = False; Profile velocity.DependOnSlotGroup = False; Profile acceleration.Index = 16#6883; Profile acceleration.SubIndex = 0; Profile acceleration.Size = 32; Profile acceleration.Offset = 0; Profile acceleration.DependOnSlot = False; Profile acceleration.DependOnSlotGroup = False; Profile deceleration.Index = 16#6884; Profile deceleration.SubIndex = 0; Profile deceleration.Size = 32; Profile deceleration.Offset = 0; Profile deceleration.DependOnSlot = False;
            Profile deceleration.DependOnSlotGroup = False; Axis2 push current.Index = 16#4121; Axis2 push current.SubIndex = 2; Axis2 push current.Size = 16; Axis2 push current.Offset = 0; Axis2 push current.DependOnSlot = False; Axis2 push current.DependOnSlotGroup = False; Axis2 base current.Index = 16#4126; Axis2 base current.SubIndex = 2; Axis2 base current.Size = 16; Axis2 base current.Offset = 0; Axis2 base current.DependOnSlot = False; Axis2 base current.DependOnSlotGroup = False; RxTxPdo.NumberofExcludes = 0; RxTxPdo.NumberofEntries = 2; RxTxPdo.Index = 16#1700; RxTxPdo.Fixed = False; RxTxPdo.Mandatory = False; RxTxPdo.Virtual = False; RxTxPdo.Sm = 2; RxTxPdo.Su = 0; RxTxPdo.Name = 'Controller Receive PDO Mapping'; RxTxPdo.DependOnSlot = False; RxTxPdo.DependOnSlotGroup = False; Controller command 1.Index = 16#2F01; Controller command 1.SubIndex = 0; Controller command 1.Size = 8; Controller command 1.Offset = 0; Controller command 1.DependOnSlot = False; Controller command 1.DependOnSlotGroup = False; Controller command 2.Index = 16#2F02; Controller command 2.SubIndex = 0; Controller command 2.Size = 8; Controller command 2.Offset = 0; Controller command 2.DependOnSlot = False; Controller command 2.DependOnSlotGroup = False; RxTxPdo.NumberofExcludes = 0; RxTxPdo.NumberofEntries = 8; RxTxPdo.Index = 16#1A00; RxTxPdo.Fixed = False;
            RxTxPdo.Mandatory = False; RxTxPdo.Virtual = False; RxTxPdo.Sm = 3; RxTxPdo.Su = 0; RxTxPdo.Name = 'Axis1 Transmit PDO Mapping 1'; RxTxPdo.DependOnSlot = False; RxTxPdo.DependOnSlotGroup = False; RxTxPdo.OverwrittenByModule = False; Error code.Index = 16#603F; Error code.SubIndex = 0; Error code.Size = 16; Error code.Offset = 0; Error code.DependOnSlot = False; Error code.DependOnSlotGroup = False; Statusword.Index = 16#6041; Statusword.SubIndex = 0; Statusword.Size = 16; Statusword.Offset = 0; Statusword.DependOnSlot = False; Statusword.DependOnSlotGroup = False; Position demand value.Index = 16#6062; Position demand value.SubIndex = 0; Position demand value.Size = 32; Position demand value.Offset = 0; Position demand value.DependOnSlot = False; Position demand value.DependOnSlotGroup = False; Position actual value.Index = 16#6064; Position actual value.SubIndex = 0; Position actual value.Size = 32; Position actual value.Offset = 0; Position actual value.DependOnSlot = False; Position actual value.DependOnSlotGroup = False; Velocity demand value.Index = 16#606B; Velocity demand value.SubIndex = 0; Velocity demand value.Size = 32; Velocity demand value.Offset = 0; Velocity demand value.DependOnSlot = False; Velocity demand value.DependOnSlotGroup = False; Velocity actual value.Index = 16#606C; Velocity actual value.SubIndex = 0;
            Velocity actual value.Size = 32; Velocity actual value.Offset = 0; Velocity actual value.DependOnSlot = False; Velocity actual value.DependOnSlotGroup = False; Modes of operation display.Index = 16#6061; Modes of operation display.SubIndex = 0; Modes of operation display.Size = 8; Modes of operation display.Offset = 0; Modes of operation display.DependOnSlot = False; Modes of operation display.DependOnSlotGroup = False; Axis1 motor temperature.Index = 16#407D; Axis1 motor temperature.SubIndex = 1; Axis1 motor temperature.Size = 16; Axis1 motor temperature.Offset = 0; Axis1 motor temperature.DependOnSlot = False; Axis1 motor temperature.DependOnSlotGroup = False; RxTxPdo.NumberofExcludes = 0; RxTxPdo.NumberofEntries = 8; RxTxPdo.Index = 16#1A10; RxTxPdo.Fixed = False; RxTxPdo.Mandatory = False; RxTxPdo.Virtual = False; RxTxPdo.Sm = 3; RxTxPdo.Su = 0; RxTxPdo.Name = 'Axis2 Transmit PDO Mapping 1'; RxTxPdo.DependOnSlot = False; RxTxPdo.DependOnSlotGroup = False; RxTxPdo.OverwrittenByModule = False; Error code.Index = 16#683F; Error code.SubIndex = 0; Error code.Size = 16; Error code.Offset = 0; Error code.DependOnSlot = False; Error code.DependOnSlotGroup = False; Statusword.Index = 16#6841; Statusword.SubIndex = 0; Statusword.Size = 16; Statusword.Offset = 0; Statusword.DependOnSlot = False; Statusword.DependOnSlotGroup = False;
            Position demand value.Index = 16#6862; Position demand value.SubIndex = 0; Position demand value.Size = 32; Position demand value.Offset = 0; Position demand value.DependOnSlot = False; Position demand value.DependOnSlotGroup = False; Position actual value.Index = 16#6864; Position actual value.SubIndex = 0; Position actual value.Size = 32; Position actual value.Offset = 0; Position actual value.DependOnSlot = False; Position actual value.DependOnSlotGroup = False; Velocity demand value.Index = 16#686B; Velocity demand value.SubIndex = 0; Velocity demand value.Size = 32; Velocity demand value.Offset = 0; Velocity demand value.DependOnSlot = False; Velocity demand value.DependOnSlotGroup = False; Velocity actual value.Index = 16#686C; Velocity actual value.SubIndex = 0; Velocity actual value.Size = 32; Velocity actual value.Offset = 0; Velocity actual value.DependOnSlot = False; Velocity actual value.DependOnSlotGroup = False; Modes of operation display.Index = 16#6861; Modes of operation display.SubIndex = 0; Modes of operation display.Size = 8; Modes of operation display.Offset = 0; Modes of operation display.DependOnSlot = False; Modes of operation display.DependOnSlotGroup = False; Axis2 motor temperature.Index = 16#407D; Axis2 motor temperature.SubIndex = 2; Axis2 motor temperature.Size = 16; Axis2 motor temperature.Offset = 0; Axis2 motor temperature.DependOnSlot = False; Axis2 motor temperature.DependOnSlotGroup = False; RxTxPdo.NumberofExcludes = 0; RxTxPdo.NumberofEntries = 2; RxTxPdo.Index = 16#1B00; RxTxPdo.Fixed = False;
            RxTxPdo.Mandatory = False; RxTxPdo.Virtual = False; RxTxPdo.Sm = 3; RxTxPdo.Su = 0; RxTxPdo.Name = 'Controller Transmit PDO Mapping'; RxTxPdo.DependOnSlot = False; RxTxPdo.DependOnSlotGroup = False; RxTxPdo.OverwrittenByModule = False; Controller status 1.Index = 16#2E31; Controller status 1.SubIndex = 0; Controller status 1.Size = 8; Controller status 1.Offset = 0; Controller status 1.DependOnSlot = False; Controller status 1.DependOnSlotGroup = False; Controller status 2.Index = 16#2E32; Controller status 2.SubIndex = 0; Controller status 2.Size = 8; Controller status 2.Offset = 0; Controller status 2.DependOnSlot = False; Controller status 2.DependOnSlotGroup = False; Controlword.Name = 'Controlword'; Controlword.DataType = 'UINT'; Controlword.Default = ''; Controlword.Comment = ''; Target position.Name = 'Target position'; Target position.DataType = 'DINT'; Target position.Default = ''; Target position.Comment = ''; Modes of operation.Name = 'Modes of operation'; Modes of operation.DataType = 'SINT'; Modes of operation.Default = ''; Modes of operation.Comment = ''; Profile velocity.Name = 'Profile velocity'; Profile velocity.DataType = 'UDINT'; Profile velocity.Default = ''; Profile velocity.Comment = ''; Profile acceleration.Name = 'Profile acceleration'; Profile acceleration.DataType = 'UDINT'; Profile acceleration.Default = ''; Profile acceleration.Comment = '';
            Profile deceleration.Name = 'Profile deceleration'; Profile deceleration.DataType = 'UDINT'; Profile deceleration.Default = ''; Profile deceleration.Comment = ''; Axis1 push current.Name = 'Axis1 push current'; Axis1 push current.DataType = 'INT'; Axis1 push current.Default = ''; Axis1 push current.Comment = ''; Axis1 base current.Name = 'Axis1 base current'; Axis1 base current.DataType = 'INT'; Axis1 base current.Default = ''; Axis1 base current.Comment = ''; Controlword.Name = 'Controlword'; Controlword.DataType = 'UINT'; Controlword.Default = ''; Controlword.Comment = ''; Target position.Name = 'Target position'; Target position.DataType = 'DINT'; Target position.Default = ''; Target position.Comment = ''; Modes of operation.Name = 'Modes of operation'; Modes of operation.DataType = 'SINT'; Modes of operation.Default = ''; Modes of operation.Comment = ''; Profile velocity.Name = 'Profile velocity'; Profile velocity.DataType = 'UDINT'; Profile velocity.Default = ''; Profile velocity.Comment = ''; Profile acceleration.Name = 'Profile acceleration'; Profile acceleration.DataType = 'UDINT'; Profile acceleration.Default = ''; Profile acceleration.Comment = ''; Profile deceleration.Name = 'Profile deceleration'; Profile deceleration.DataType = 'UDINT'; Profile deceleration.Default = ''; Profile deceleration.Comment = ''; Axis2 push current.Name = 'Axis2 push current'; Axis2 push current.DataType = 'INT'; Axis2 push current.Default = ''; Axis2 push current.Comment = '';
            Axis2 base current.Name = 'Axis2 base current'; Axis2 base current.DataType = 'INT'; Axis2 base current.Default = ''; Axis2 base current.Comment = ''; Controller command 1.Name = 'Controller command 1'; Controller command 1.DataType = 'USINT'; Controller command 1.Default = ''; Controller command 1.Comment = ''; Controller command 2.Name = 'Controller command 2'; Controller command 2.DataType = 'USINT'; Controller command 2.Default = ''; Controller command 2.Comment = ''; Error code.Name = 'Error code'; Error code.DataType = 'UINT'; Error code.Default = ''; Error code.Comment = ''; Statusword.Name = 'Statusword'; Statusword.DataType = 'UINT'; Statusword.Default = ''; Statusword.Comment = ''; Position demand value.Name = 'Position demand value'; Position demand value.DataType = 'DINT'; Position demand value.Default = ''; Position demand value.Comment = ''; Position actual value.Name = 'Position actual value'; Position actual value.DataType = 'DINT'; Position actual value.Default = ''; Position actual value.Comment = ''; Velocity demand value.Name = 'Velocity demand value'; Velocity demand value.DataType = 'DINT'; Velocity demand value.Default = ''; Velocity demand value.Comment = ''; Velocity actual value.Name = 'Velocity actual value'; Velocity actual value.DataType = 'DINT'; Velocity actual value.Default = ''; Velocity actual value.Comment = ''; Modes of operation display.Name = 'Modes of operation display'; Modes of operation display.DataType = 'SINT'; Modes of operation display.Default = ''; Modes of operation display.Comment = '';
            Axis1 motor temperature.Name = 'Axis1 motor temperature'; Axis1 motor temperature.DataType = 'INT'; Axis1 motor temperature.Default = ''; Axis1 motor temperature.Comment = ''; Error code.Name = 'Error code'; Error code.DataType = 'UINT'; Error code.Default = ''; Error code.Comment = ''; Statusword.Name = 'Statusword'; Statusword.DataType = 'UINT'; Statusword.Default = ''; Statusword.Comment = ''; Position demand value.Name = 'Position demand value'; Position demand value.DataType = 'DINT'; Position demand value.Default = ''; Position demand value.Comment = ''; Position actual value.Name = 'Position actual value'; Position actual value.DataType = 'DINT'; Position actual value.Default = ''; Position actual value.Comment = ''; Velocity demand value.Name = 'Velocity demand value'; Velocity demand value.DataType = 'DINT'; Velocity demand value.Default = ''; Velocity demand value.Comment = ''; Velocity actual value.Name = 'Velocity actual value'; Velocity actual value.DataType = 'DINT'; Velocity actual value.Default = ''; Velocity actual value.Comment = ''; Modes of operation display.Name = 'Modes of operation display'; Modes of operation display.DataType = 'SINT'; Modes of operation display.Default = ''; Modes of operation display.Comment = ''; Axis2 motor temperature.Name = 'Axis2 motor temperature'; Axis2 motor temperature.DataType = 'INT'; Axis2 motor temperature.Default = ''; Axis2 motor temperature.Comment = ''; Controller status 1.Name = 'Controller status 1'; Controller status 1.DataType = 'USINT'; Controller status 1.Default = ''; Controller status 1.Comment = '';
            Controller status 2.Name = 'Controller status 2'; Controller status 2.DataType = 'USINT'; Controller status 2.Default = ''; Controller status 2.Comment = ''
          output oFrontJawAxisControlword : UINT  // Controlword
          output oFrontJawAxisTargetPosition : DINT  // Target position
          output oFrontJawAxisModesOfOperation : SINT  // Modes of operation
          output oFrontJawAxisProfileVelocity : UDINT  // Profile velocity
          output oFrontJawAxisProfileAcceleration : UDINT  // Profile acceleration
          output oFrontJawAxisProfileDeceleration : UDINT  // Profile deceleration
          output oFrontJawAxisPushCurrent : INT  // Axis1 push current
          output oFrontJawAxisBaseCurrent : INT  // Axis1 base current
          output oFilmFeedAxisControlword : UINT  // Controlword
          output oFilmFeedAxisTargetPosition : DINT  // Target position
          output oFilmFeedAxisModesOfOperation : SINT  // Modes of operation
          output oFilmFeedAxisProfileVelocity : UDINT  // Profile velocity
          output oFilmFeedAxisProfileAcceleration : UDINT  // Profile acceleration
          output oFilmFeedAxisProfileDeceleration : UDINT  // Profile deceleration
          output oFilmFeedAxisPushCurrent : INT  // Axis2 push current
          output oFilmFeedAxisBaseCurrent : INT  // Axis2 base current
          input  iFrontJawAxisErrorcode : UINT  // Error code
          input  iFrontJawAxisStatusword : UINT  // Statusword
          input  iFrontJawAxisPositionDemandValue : DINT  // Position demand value
          input  iFrontJawAxisPositionActualValue : DINT  // Position actual value
          input  iFrontJawAxisVelocityDemandValue : DINT  // Velocity demand value
          input  iFrontJawAxisVelocityActualValue : DINT  // Velocity actual value
          input  iFrontJawAxisModesOfOperationDisplay : SINT  // Modes of operation display
          input  iFrontJawAxisTemperature : INT  // Axis1 motor temperature
          input  iFilmFeedAxisErrorcode : UINT  // Error code
          input  iFilmFeedAxisStatusword : UINT  // Statusword
          input  iFilmFeedAxisPositionDemandValue : DINT  // Position demand value
          input  iFilmFeedAxisPositionActualValue : DINT  // Position actual value
          input  iFilmFeedAxisVelocityDemandValue : DINT  // Velocity demand value
          input  iFilmFeedAxisVelocityActualValue : DINT  // Velocity actual value
          input  iFilmFeedAxisModesOfOperationDisplay : SINT  // Modes of operation display
          input  iFilmFeedAxisTemperature : INT  // Axis2 motor temperature
          unmapped channels: Controller command 1, Controller command 2, Controller status 1, Controller status 2
      Main_IO : AMAX-4830 16-ch Isolated Digital Input/16-ch Isolated Output EtherCAT I/O Module, Advantech Co., Ltd., order no. AMAX-4830, version Revision=16#00000002
          settings: EnableExpertSettings = True; StationAlias = 1001; Optional = False; DeviceIdenticationADO = 0; DeviceIdenticationMode = 0; DC sync0 cycletime = 4000; DC sync1 cycletime = 4000
          output Application.mainIOamax4830Output[0].discreteSignal AT %QX0.0 : BIT  // DO0
          output Application.mainIOamax4830Output[1].discreteSignal : BIT  // DO1
          output Application.mainIOamax4830Output[2].discreteSignal : BIT  // DO2
          output Application.mainIOamax4830Output[3].discreteSignal : BIT  // DO3
          output Application.mainIOamax4830Output[4].discreteSignal : BIT  // DO4
          output Application.mainIOamax4830Output[5].discreteSignal : BIT  // DO5
          output Application.mainIOamax4830Output[6].discreteSignal : BIT  // DO6
          output Application.mainIOamax4830Output[7].discreteSignal : BIT  // DO7
          output Application.mainIOamax4830Output[8].discreteSignal : BIT  // DO8
          output Application.mainIOamax4830Output[9].discreteSignal : BIT  // DO9
          output Application.mainIOamax4830Output[10].discreteSignal : BIT  // DO10
          output Application.mainIOamax4830Output[11].discreteSignal : BIT  // DO11
          output Application.mainIOamax4830Output[12].discreteSignal : BIT  // DO12
          output Application.mainIOamax4830Output[13].discreteSignal : BIT  // DO13
          output Application.mainIOamax4830Output[14].discreteSignal : BIT  // DO14
          output Application.mainIOamax4830Output[15].discreteSignal : BIT  // DO15
          input  Application.mainIOamax4830Input[0].discreteSignal : BIT  // DI0
          input  Application.mainIOamax4830Input[1].discreteSignal : BIT  // DI1
          input  Application.mainIOamax4830Input[2].discreteSignal : BIT  // DI2
          input  Application.mainIOamax4830Input[3].discreteSignal : BIT  // DI3
          input  Application.mainIOamax4830Input[4].discreteSignal : BIT  // DI4
          input  Application.mainIOamax4830Input[5].discreteSignal : BIT  // DI5
          input  Application.mainIOamax4830Input[6].discreteSignal : BIT  // DI6
          input  Application.mainIOamax4830Input[7].discreteSignal : BIT  // DI7
          input  Application.mainIOamax4830Input[8].discreteSignal : BIT  // DI8
          input  Application.mainIOamax4830Input[9].discreteSignal : BIT  // DI9
          input  Application.mainIOamax4830Input[10].discreteSignal : BIT  // DI10
          input  Application.mainIOamax4830Input[11].discreteSignal : BIT  // DI11
          input  Application.mainIOamax4830Input[12].discreteSignal : BIT  // DI12
          input  Application.mainIOamax4830Input[13].discreteSignal : BIT  // DI13
          input  Application.mainIOamax4830Input[14].discreteSignal : BIT  // DI14
          input  Application.mainIOamax4830Input[15].discreteSignal : BIT  // DI15
    MBCOMPort2 : Modbus COM, 3S - Smart Software Solutions GmbH, version 3.5.11.20
        settings: ComPort = 2
      MBMasterCOMPort2 : Modbus Master, COM Port, 3S - Smart Software Solutions GmbH, version 3.5.11.20
          settings: Auto-restart communication = TRUE
  UnitTestRuntime : CODESYS Control Win V3 x64, 3S - Smart Software Solutions GmbH, version 3.5.15.0
  libraries: Standard, 3.5.18.0 (System); SysTime, 3.5.9.0 (System); BASIC, 3.3.3.0 (OSCAT); OMAC PackML State Machine, 1.0.0.0 (3S - Smart Software Solutions GmbH); Time and Date, 3.5.7.0 (3S - Smart Software Solutions GmbH); Test Manager IEC Unit Test, 4.1.0.0 (Intern); CAA Behaviour Model, 3.5.11.0 (CAA Technical Workgroup); FloatingPointUtils, 3.5.9.0 (System)
  Data Types/
    data type DEVICE_MODES
    data type HMIFaultType
    data type LogMessageType
    data type sctMotionProfile
    data type ServiceCommands
    data type uModbusDWORD
    data type UnitTestErrors
    data type Warning
  FBs/
    Components/
      Aux IO/
      Bag Delivery/
      BagOpenFingers/
      BarcodeReaders/
      Collision Detection/
      Cylinders/
      function block FB_AdjustablePneumaticPassthrough [ST]
      function block FB_BaggerHeadRaise [ST]
      function block FB_BaseComponent [ST]
      function block FB_CylinderFeedback [ST]
      function block FB_MonostableMultivibrator [ST]
      function block FB_MurrIO [ST]
      Fillers/
      Funnels/
      IBDs/
      Indication/
      Load Plate/
      Motors/
      Paper/
      PressureBars/
      Printers/
      Seal Area Options/
      Temp Sensors/
    DataHandlers/
      function block FB_ModbusDWORD [ST]
      function block ModbusLongHandlerFB [ST]
    DelayDwellFB/
      data type DELAY_DWELL_STATES
      function block DelayDwellFB [ST]
    Fault/
      function block FB_Fault [ST]
      function block FB_HMIFault [ST]
    function block FB_CycleCounter [ST]: Clear, Increment, SetCount
    function block FB_CylinderLeak [ST]
    function block FB_DeviceTreeEnable [ST]: ManualReconfig
    function block FB_DriveTemp [ST]
    function block FB_FaultHandler [ST]: registerFaultSource
    function block FB_HMILight [ST]: BlinkFast, BlinkSlow, TurnOff, TurnOn
    function block FB_PredictiveMaint [ST]
    function block FB_TCPClient [ST]: ClearLabel, SendLabel
    function block FB_Throughput [ST]
    function block FB_WriteToFile [ST]
    FunctionalAreas/
      function block FB_MOABHead [ST]
      function block FB_MOABHead_Electric [ST]
      data type StateMachine
      data type Substate
    function block GetTime [ST]
    Recipie Manangment/
      function RecallValues [ST]
      function SaveValues [ST]
      function SaveValuesPeriodic [ST]
    function block SerialMotorTestFB [ST]
    Unused/
      function block BagDeliveryFB_BothMotors [ST]
      function block ElectricPressureBarFB [ST]
      function block MotorizedSealFlattenersFB [ST]
      function block PickAndPlaceFB [ST]
      function block PrinterFB [ST]
  Function Blocks/
    Diagnostics/
      function block FB_StateRateTracking [ST]
      data type stateRateKeyPair
    Electric Solenoid/
      function block FB_ElectricSolenoid [ST]
    function block FB_BaseComponent [ST]: Execute, MakeReady, OptionActive, OptionEnabled, OptionInstalled, Ready, Reset, StateString, SterilizeVariables
    function block FB_BaseObject [ST]: FB_Init, InstanceName, RegisterLogger
    function block FB_Delay [ST]: Execute
    FB_Fault/
      Tests/
    function block FB_GetTime [ST]
    function block FB_HMIData [ST]
    function block FB_InternalLogger_1 [ST]: AddLogItem, InstanceName
    function block FB_InternalLogger [ST]: AddLogItem
    function block FB_LoggableBool [ST]
    FB_MachineCounter/
      function block FB_MachineCounter [ST]
      Tests/
    function block FB_MetricConversions [ST]
    FB_MonostableMultivibrator/
      Tests/
    function block FB_ONS [ST]
    function block FB_SimulatedFeedback [ST]
    function block FB_SimulatedFeedbackPhysicalInput [ST]
    function FN_RandomDINT [ST]
    IO/
      function block FB_IOLinkBlock [ST]
      function block FB_Murr16PointCFGIO [ST]
      function block FB_Murr56691_IP20 [ST]
      function block FB_PhysicalAnalogInput [ST]
      function block FB_PhysicalDigitalInput [ST]
      function block FB_PhysicalDigitalOutput [ST]
    Machine Components/
      function block FB_MurrMaster [ST]
    SolenoidValves/
      function block FB_DoubleSolenoidClosedCenterActuator [ST]
      function block FB_DoubleSolenoidOpenCenterActuator [ST]
      function block FB_PneumaticActuator [ST]
      function block FB_SingleSolenoidNormallyRetractedActuator [ST]
      function block FB_SolenoidValve [ST]
      function block FB_SolenoidValveManifold [ST]
      function block FB_VacuumGenerator [ST]
      Tests/
      data type ValveSelection
  Generated Unit Tests/
  Globals/
  global variables Globals
  text list GlobalTextList
  global variables HMIData
  Interfaces/
    interface IComponentStatus: Mode, Ready
    interface IFaultHandler: AddActiveFault, RemoveActiveFault
    interface ISupervisor: MakeReady, NotifyMachineFaulted
  Interfaces/
    interface IAllObjects: InstanceName
    interface IComponent: MakeReady, Ready, Reset, StateString, SterilizeVariables
    interface ICounter: Increment
    interface ICylinder: Extend, ExtendAsserted, IsExtended, IsRetracted, Retract, RetractAsserted
    interface IExecuteAutomatically: Execute
    interface IExhaustable: Exhaust
    interface IExtendLowPressure: ExtendLowPressure, ExtendLPAsserted
    interface IFault: Ack, FaultActive, FaultID, Trigger
    interface IInitializable: Initialize
    interface ILoggable: RegisterLogger
    interface IMachineLogger: AddLogItem
    interface IMachineOption: OptionActive, OptionEnabled, OptionInstalled
    interface IPositionableMotor: CommandAcknowledged, CurrentPosition, HomeNow, HomeRequired, Homing, InPosition, MoveDistance, MoveToPosition, Moving, Stop
    interface IThreePositonCylinder: Exhaust, ExtendLowPressure
  Motion/
    Base/
      function block Axis_REF [ST]
      data type AXIS_STATE
      interface IAxisRef
      function block MC_Base [ST]
      data type MC_ERROR
      data type OP_MODE
    Custom MC/
      function block MC_MoveAbsoluteTorqueLimited [ST]
      function block MC_MoveFinalBagDelivery [ST]
    PLCopen MC/
      function block MC_Halt [ST]
      function block MC_Home [ST]
      function block MC_MoveAbsolute [ST]
      function block MC_MoveRelative [ST]
      function block MC_MoveVelocity [ST]
      function block MC_Power [ST]
      function block MC_Reset [ST]
      function block MC_Stop [ST]
  ObjectHandling/
    function block FB_CollectionHandleMachineComponents [ST]: AddObject, CheckIfAllHomed, CheckIfAllReady, ForceHomeAll, HomeAll, MakeReadyAll, ResetAll, UpdateInfo
    function block FB_CollectionHandlerActiveFaults [ST]: AckAll, AddObject, RemoveObject
    function block FB_CollectionHandlerActiveFaults [ST]: AckAll, AddObject, RemoveObject
    function block FB_CollectionHandlerAll [ST]: AddObject
    function block FB_CollectionHandlerCylinders [ST]: AddObject
    function block FB_CollectionHandlerExecutable [ST]: AddObject, ExecuteAll
    function block FB_CollectionHandlerExecutable [ST]: AddObject, ExecuteAll
    function block FB_CollectionHandlerFaults [ST]: AckAll, AddObject, FaultUpdateForHMI
    function block FB_CollectionHandlerFaults [ST]: AckAll, AddObject
    function block FB_CollectionHandlerInitializable [ST]: AddObject, InitializeAll
    function block FB_CollectionHandlerInitializable [ST]: AddObject, InitializeAll
    function block FB_CollectionHandlerLoggable [ST]: AddObject, RegisterAll
    function block FB_CollectionHandlerLoggable [ST]: AddObject, RegisterAll
    function block FB_CollectionHandlerLogs [ST]: AddObject
    function block FB_CollectionHandlerLogs [ST]: AddObject
    function block FB_CollectionHandlerPositionableMotors [ST]: AddObject
    global variables GlobalObjects
    interface IFault: Ack, Trigger
    interface IResettable
  RemoteComms/
    data type Modbus_Inputs
    data type Modbus_Outputs
    data type OPC_Faults
    data type OPC_Inputs
    data type OPC_Outputs
    global variables RemoteComms
  text list System
  Testing/
    Actuators/
      function block FB_DummyUpDown [ST]
      function block FB_PneumaticVerticalActuator [ST]
      interface ISolenoidValve
      interface IUpDown
    FB_AmazonThroughput/
    FB_AMPMotorSerial/
      function block FB_AMPMotorSerial [ST]
    FB_BannerPalmButton/
      function block FB_BannerPalmButton [ST]
    FB_CrevisSerial/
      data type eSerialStates
      function block FB_CrevisSerial [ST]
    function block FB_MultiUnitTest [ST]: prvAbort, prvCyclicAction, prvResetOutputs, prvStart
    function block FB_PrinterSerial [ST]
    function block FB_Simulation [ST]
    HelperFunctions/
      function CheckIfHomed [ST]
      function CheckIfReady [ST]
      function EnableSimulation [ST]
      function ExhaustIfPossible [ST]
      function ExtendLPIfPossible [ST]
      function HomeIfNeeded [ST]
      function MoveRequested [ST]
      function PostHomeMoveIfNeeded [ST]
    interface ISimulateable: Simulate
    Motors/
      Applied Motion/
      function block FB_AppliedMotionMotor [ST]
      interface IHomable
      interface IPostHomeMove
      Oriental/
      SimMotor/
    function MoveTimeoutCalc [ST]
  text list TextListForCombobox_BagOpenFingersSelection
  text list TextListForCombobox_IntegratedConveyorSelection
  text list TextListForCombobox_LabelPrinterSelection
  text list TextListForCombobox_PackageEjectionSelection
  text list TextListForCombobox_SealFlattenerSelection
  Types/
    data type Alarm
    AuxIO/
    data type CONFIG_VERSIONS
    data type CylinderFaultsType
    data type DEVICE_MODES
    Factoy Selection/
      data type AuxiliaryIOSelection
      data type BagDeflatorSelection
      data type BagOpenFingersSelection
      data type BCVSelection
      data type ExteralConveyorSelection
      data type FeedToSealSelection
      data type FillerSelection
      data type FunnelSelection
      data type IntegratedConveyorSelection
      data type LabelPrinterSelection
      data type LightCurtainsSelection
      data type ModelSelection
      data type PackageEjectionSelection
      data type PalmButtonSelection
      data type SealAreaOptionSelectionEnum
    data type Fault
    data type FaultType
    HMI Types/
      data type PressureBarHMI
    data type IOMasterFaultsType
    data type LoadPlateFaultsType
    data type MAILER_MATERIAL
    data type MODBUS_COMM_TYPE
    data type ModbusLongType
    data type MotorCommFault
    data type ORIENTAL_OPERATION_TYPES
    data type PressureBarFaultsType
    data type PRINT_SPEEDS
    data type QX_PROGRAMS
    data type ServiceCommands
    States/
      data type BAG_DELIVERY_MOVE_STATES
      data type BCR_STATES
      data type EZFEED_STATES_1
      data type FILLER_STATES
      data type GRABBER_STATES
      Head/
      data type JAW_HOMING_STATES
      data type JOG_STATES
      data type MOVE_MODBUS_COMMAND_STATES
      MurrIOMOdule/
      data type OPCODE_MODBUS_COMMAND_STATES
      data type PASSTHROUGH_SERVO_STATES
      data type SOLENOID_TEST_STATES
      data type VACUUM_PICKER_STATES
    data type STEP_SERVO_OPCODES
    data type StepServoFaultsType
  UN00 - Sharp Bagger/
    EM00 - Product Infeed/
      CM00 - Funnel/
      CM01 - Infeed Conveyor/
      CM02 - External Filler/
      CM03 - Operator Interface/
      interface IEM00_Product_Infeed
    EM01 - Bagger Head/
      CM00 - Bag Open Fingers/
      CM01 - Seal Flatteners/
      CM02 - Pressure Bar/
      CM03 - Sealer/
      CM04 - Bag Delivery/
      CM05 - Printer/
      CM06 - Vacuum Bag Open/
      CM07 - IBD/
      CM08 - Barcode Verifier/
      function block EM01_BaggerHead_Automode [ST]
      function block EM01_BaggerHead [ST]
      function block EM01_BaggerHead_MaintMode [ST]
      function block EM01_BaggerHead_Manager [ST]
      interface IEM01_BaggerHead
      States/
      program TestBaggerHead [ST]
    EM02 - Discharge/
      CM00 - Retracting Load Plate/
      CM01 - Exit Conveyor/
      function block EM02_Discharge [ST]
      interface IEM02_Discharge
    function block FB_PackMLStates [ST]: Aborted, Aborting, AbortingDone, Clearing, ClearingDone, Complete
    function block FB_UN00_SharpMachine [ST]
    interface IPackMLStates
    visualisation PackML
    global variables UN00_Globals
  Unused/
    function block FB_SimBasicBagDelivery [ST]
    function block FB_SimBasicPrinter [ST]
    function block FB_SimBasicSealFlatteners [ST]
    function block FB_SimBasicVacuum [ST]
  visualisation VISU_HELPER_Combobox_BagOpenFingersSelection
  visualisation VISU_HELPER_Combobox_IntegratedConveyorSelection
  visualisation VISU_HELPER_Combobox_LabelPrinterSelection
  visualisation VISU_HELPER_Combobox_PackageEjectionSelection
  visualisation VISU_HELPER_Combobox_SealFlattenerSelection
  visualisation VISU_NEW_FB_HMIData
  visualisation VISU_NEW_FB_IOLinkBlock
  visualisation VISU_NEW_FB_Murr16PointCFGIO
  visualisation VISU_NEW_FB_Murr56691_IP20
  visualisation VISU_NEW_FB_PneuBagOpenFingersWithSensors
  visualisation VISU_NEW_FB_PneuBagOpenFingersWithSensorsOLD
  visualisation VISU_NEW_FB_Simulation
  function GetLibVersion [ST]
  function GetLibVersionNumber [ST]
  function GetCompany [ST]
  function GetTextProperty2 [ST]
  function GetTextProperty [ST]
  function GetTitle [ST]
  function GetVersion [ST]
  function GetVersionProperty [ST]
*)

// Data Types/DEVICE_MODES
{attribute 'qualified_only'}
{attribute 'strict'}
TYPE DEVICE_MODES :
(
	Manual := 0,	// Control only from service
	Auto := 1,		// Control only from main Bagger Program
	SemiAuto := 2	// Independent control (like as a test fixture)
);
END_TYPE

// Data Types/HMIFaultType
TYPE HMIFaultType :
STRUCT
	name : STRING;
	active : BOOL;
END_STRUCT
END_TYPE

// Data Types/LogMessageType
TYPE LogMessageType :
STRUCT
	logTime : DATE_AND_TIME;
	logCategory : STRING;
	logMessage : STRING;
END_STRUCT
END_TYPE

// Data Types/sctMotionProfile
TYPE sctMotionProfile :
STRUCT
	velo : REAL;
	accel : REAL;
	decel : REAL;
	current : REAL;
END_STRUCT
END_TYPE

// Data Types/ServiceCommands
TYPE ServiceCommands : 
STRUCT
	extendCommand : BOOL;
	retractCommand : BOOL;
	exhaustCommand : BOOL;
	extendedFeedback : BOOL;
	retractedFeedback : BOOL;
END_STRUCT
END_TYPE

// Data Types/uModbusDWORD
TYPE uModbusDWORD :
UNION
	wWord : ARRAY[0..1] OF WORD;
	dDword : DWORD;
	diDint : DINT;
END_UNION
END_TYPE

// Data Types/UnitTestErrors
{attribute 'qualified_only'}
{attribute 'strict'}
TYPE UnitTestErrors :
(
	Failure,
	Failure2
);
END_TYPE

// Data Types/Warning
TYPE Warning :
STRUCT
	active : BOOL;
END_STRUCT
END_TYPE

// RemoteComms/Modbus_Inputs
TYPE Modbus_Inputs :
STRUCT
	fillerTrigger : BOOL; // Filler Trigger - set high to trigger cycle in filler mode
	baggerInhibit : BOOL; // Bagger Inhibit - set high to prevent a bagger cycle
	collisionDetection : BOOL; // Collision Detection - set high to indicate potential trunk line package collision
	fillerOK : BOOL;
//	EnableBagger : BOOL;  //Unused
	reverseConveyor : BOOL;  // Reverse Exit Conveyor - set high to reverse direction of rear exit conveyor
	bagGrabbed : BOOL; // Bag Grabbed - Set high to indicate bag grabbed by automation
	heartbeat : BOOL; // Heartbeat - set and reset based on heartbeatResponse.
END_STRUCT
END_TYPE

// RemoteComms/Modbus_Outputs
TYPE Modbus_Outputs :
STRUCT
	baggerOK : BOOL; // Bagger OK - Set high when Not Faulted
	readyForFiller : BOOL; // Ready for Filler - set high when ready for filler 
	printerDataReady : BOOL; // Printer Data Ready - set high when priter has a label
	waitingForPrinter : BOOL; // Waiting for Printer - set high when bagger is paused in cycle waiting for a label
	cycleComplete : BOOL; // Cycle Complete - pulsed when bagger cycle is complete (opened bag)
	bagMade : BOOL; // Bag Made - pulsed when bag is sealed and bag is dropping
	bagMadePlusLabelRequired : BOOL; // Bag Made - pulsed when bag is sealed and bag is dropping and bagger needs a label
	bagsLow : BOOL;	// Bags Low - set high when bag level is low
	readyForGrab : BOOL; // Ready for Grab - set high when bagger is ready for automation to grab bag
	runExternalExitConveyor : BOOL; // Run External Exit Conveyor - set high when external exit conveyor is called for
	heartbeatResponse : BOOL; // Heartbeat response - set equal to heartbeat
END_STRUCT
END_TYPE

// RemoteComms/OPC_Faults
TYPE OPC_Faults :
STRUCT
	reverseFault : BOOL;
	bagFailedToOpen : BOOL;
	obstructionFault : BOOL;
END_STRUCT
END_TYPE

// RemoteComms/OPC_Inputs
TYPE OPC_Inputs :
STRUCT
	fillerTrigger : BOOL; // Filler Trigger - set high to trigger cycle in filler mode
	baggerInhibit : BOOL; // Bagger Inhibit - set high to prevent a bagger cycle
	collisionDetection : BOOL; // Collision Detection - set high to indicate potential trunk line package collision
	fillerOK : BOOL;
//	EnableBagger : BOOL;  //Unused
	reverseConveyor : BOOL;  // Reverse Exit Conveyor - set high to reverse direction of rear exit conveyor
	bagGrabbed : BOOL; // Bag Grabbed - Set high to indicate bag grabbed by automation
	heartbeat : BOOL; // Heartbeat - set and reset based on heartbeatResponse.
END_STRUCT
END_TYPE

// RemoteComms/OPC_Outputs
TYPE OPC_Outputs :
STRUCT
	baggerOK : BOOL; // Bagger OK - Set high when Not Faulted
	readyForFiller : BOOL; // Ready for Filler - set high when ready for filler 
	printerDataReady : BOOL; // Printer Data Ready - set high when priter has a label
	waitingForPrinter : BOOL; // Waiting for Printer - set high when bagger is paused in cycle waiting for a label
	cycleComplete : BOOL; // Cycle Complete - pulsed when bagger cycle is complete (opened bag)
	bagMade : BOOL; // Bag Made - pulsed when bag is sealed and bag is dropping
	bagMadePlusLabelRequired : BOOL; // Bag Made - pulsed when bag is sealed and bag is dropping and bagger needs a label
	bagsLow : BOOL;	// Bags Low - set high when bag level is low
	readyForGrab : BOOL; // Ready for Grab - set high when bagger is ready for automation to grab bag
	runExternalExitConveyor : BOOL; // Run External Exit Conveyor - set high when external exit conveyor is called for
	heartbeatResponse : BOOL; // Heartbeat response - set equal to heartbeat
	activeFaultsList : ARRAY[0..GlobalObjects.MAX_FAULTS] OF STRING; // Active Faults - list of active fault strings
	faultListTags : OPC_Faults;
END_STRUCT
END_TYPE

// Types/Alarm
TYPE Alarm :
STRUCT
	active : BOOL;
	acknowledged : BOOL;
	ackCommand : BOOL;
END_STRUCT
END_TYPE

// Types/CONFIG_VERSIONS
{attribute 'strict'}
{attribute 'qualified_only'}
TYPE CONFIG_VERSIONS :
(
	V_1_0,
	V_1_1,
	V_1_2,
	V_1_3,
	V_1_4,
	V_1_5,
	V_1_6,
	V_1_7,
	V_1_8,
	V_1_9,
	V_1_10,
	V_1_11,
	V_1_12,
	V_1_13,
	V_1_14,
	V_1_15,
	V_1_16,
	V_1_17,
	V_1_18,
	V_1_19,
	V_1_20,
	V_1_21,
	V_1_22,
	V_1_23,
	V_1_24,
	V_1_25,
	V_1_26,
	V_1_27,
	V_1_28,
	V_1_29,
	V_1_30,
	V_1_31,
	V_1_32,
	V_1_33,
	V_1_34,
	V_1_35,
	V_1_36,
	V_1_37,
	V_1_38,
	V_1_39,
	V_1_40,
	V_1_41,
	V_1_42,
	V_1_43,
	V_1_44,
	V_1_45,
	V_1_46,
	V_1_47,
	V_1_48,
	V_1_49,
	V_2_0,
	V_2_1,
	V_2_2,
	V_2_3,
	V_2_4,
	V_2_5,
	V_2_6,
	V_2_7,
	V_2_8,
	V_2_9,
	V_2_10,
	V_2_11,
	V_2_12,
	V_2_13,
	V_2_14,
	V_2_15,
	V_2_16,
	V_2_17,
	V_2_18,
	V_2_19,
	V_2_20,
	V_2_21,
	V_2_22,
	V_2_23,
	V_2_24,
	V_2_25,
	V_2_26,
	V_2_27,
	V_2_28,
	V_2_29,
	V_2_30,
	V_2_31,
	V_2_32,
	V_2_33,
	V_2_34,
	V_2_35,
	V_2_36,
	V_2_37,
	V_2_38,
	V_2_39,
	V_2_40,
	V_2_41,
	V_2_42,
	V_2_43,
	V_2_44,
	V_2_45,
	V_2_46,
	V_2_47,
	V_2_48,
	V_2_49
);
END_TYPE

// Types/CylinderFaultsType
TYPE CylinderFaultsType :
STRUCT
	failedToExtend : FaultType;        // Cylinder was commanded to extend but failed to reach the sensor
    failedToRetract : FaultType;      // Cylinder was commanded to retract but failed to reach the sensor
	sensorFault : FaultType;		// Both Extend and Retract sensors active at the same time
END_STRUCT
END_TYPE

// Types/DEVICE_MODES
{attribute 'qualified_only'}
{attribute 'strict'}
TYPE DEVICE_MODES :
(
	Manual := 0,	// Control only from service
	Auto := 1,		// Control only from main Bagger Program
	SemiAuto := 2	// Independent control (like as a test fixture)
);
END_TYPE

// Types/Fault
TYPE Fault :
STRUCT
    name : STRING[20];
    description : STRING[255];
END_STRUCT
END_TYPE

// Types/FaultType
TYPE FaultType :
STRUCT
	active : BOOL;
	acknowledged : BOOL;
	ackCommand : BOOL;
END_STRUCT
END_TYPE

// Types/IOMasterFaultsType
TYPE IOMasterFaultsType :
STRUCT
	commFail : FB_Fault(name := 'Communication Fail');	// IO Master to Controller Communication Failure
END_STRUCT
END_TYPE

// Types/LoadPlateFaultsType
TYPE LoadPlateFaultsType :
STRUCT
	failedToDischarge : FB_Fault(name := 'Failed to Discharge');        // Load Plate failed to reach Discharge Position
    failedToLoad : FB_Fault(name := 'Failed to Load');  // Load Plate failed to reach Loading Position
	sensorFault : FB_Fault(name := 'Failed to Sensor Fault');		// Both sensors active at the same time
END_STRUCT
END_TYPE

// Types/MAILER_MATERIAL
{attribute 'qualified_only'}
{attribute 'strict'}
TYPE MAILER_MATERIAL :
(
	poly := 0,
	paper := 1
);
END_TYPE

// Types/MODBUS_COMM_TYPE
{attribute 'strict'}
{attribute 'qualified_only'}
TYPE MODBUS_COMM_TYPE :
(
	ModbusTCP := 0,
	ModbusRTU := 1
);
END_TYPE

// Types/ModbusLongType
TYPE ModbusLongType :
STRUCT
    highWord : WORD;
    lowWord : WORD;
    displayValue : DINT;
    rawValue : DINT;
END_STRUCT
END_TYPE

// Types/MotorCommFault
TYPE MotorCommFault :
STRUCT
	timeOfFault : DATE_AND_TIME;
	message : STRING;
END_STRUCT
END_TYPE

// Types/ORIENTAL_OPERATION_TYPES
{attribute 'qualified_only'}
{attribute 'strict'}
TYPE ORIENTAL_OPERATION_TYPES :
(
    NoSetting := 0,
    AbsolutePositioning := 1,
    IncrementalPositioning := 2
);
END_TYPE

// Types/PressureBarFaultsType
TYPE PressureBarFaultsType :
STRUCT
	failedToOpen : FB_Fault(name := 'Pressure Bar Failed to Open');        // Pressure Bar was commanded to extend but failed to reach the sensor
    failedToClose : FB_Fault(name := 'Pressure Bar Failed to Close');      // Pressure Bar was commanded to retract but failed to reach the sensor
	sensorFault : FB_Fault(name := 'Pressure Bar Sensor Fault');		// Both the open and close sensors active at the same time
	obstructionDetected : FB_Fault(name := 'Pressure Bar Obstruction Detected');		// Pressure Bar detected an obstruction
	obstructionFailedToSwitch : FB_Fault(name := 'Pressure Bar Obstruction Detected'); // Pressure bar obstruction sensors should switch when closed
	lightCurtainViolation : FB_Fault(name := 'Light Curtain Violation');
END_STRUCT
END_TYPE

// Types/PRINT_SPEEDS
{attribute 'qualified_only'}
{attribute 'strict'}
TYPE PRINT_SPEEDS :
(
	Two_IPS := 2
);
END_TYPE

// Types/QX_PROGRAMS
{attribute 'strict'}
TYPE QX_PROGRAMS :
(
    HOME_HARD_STOP := 1
);
END_TYPE

// Types/ServiceCommands
TYPE ServiceCommands : 
STRUCT
	extendCommand : BOOL;
	retractCommand : BOOL;
	exhaustCommand : BOOL;
	extendedFeedback : BOOL;
	retractedFeedback : BOOL;
END_STRUCT
END_TYPE

// Types/STEP_SERVO_OPCODES
{attribute 'strict'}
{attribute 'qualified_only'}
//Taken from Host-Command-Reference pdf on Applied Motion website
TYPE STEP_SERVO_OPCODES :
(
	ALARM_RESET := 16#BA,     
	START_JOGGING := 16#96,     
	STOP_JOGGING := 16#D8,     
	ENCODER_FUNCTION := 16#D6,     //0
	ENCODER_POSITION := 16#98,     //Position
	FEED_TO_DOUBLE_SENSOR := 16#69,     //I/O Point 1 Condition 1 I/O Point 2 Condition 2
	FOLLOW_ENCODER := 16#CC,     //I/O Point Condition
	FEED_TO_LENGTH := 16#66,     
	FEED_TO_SENSOR_WITH_MASK_DISTANCE := 16#6A,     //I/O Point Condition
	FEED_AND_SET_OUTPUT := 16#68,     //I/O Point Condition
	FEED_TO_POSITION := 16#67,     
	FEED_TO_SENSOR := 16#6B,     //I/O Point Condition
	FEED_TO_SENSOR_WITH_SAFETY_DISTANCE := 16#6C,     //I/O Point Condition
	JOG_DISABLE := 16#A3,     
	JOG_ENABLE := 16#A2,     
	MOTOR_DISABLE := 16#9E,     
	MOTOR_ENABLE := 16#9F,     
	SEEK_HOME := 16#6E,     //I/O Point Condition
	SET_POSITION := 16#A5,     //Position
	FILTER_INPUT := 16#C0,     //I/O Point Filter Time
	FILTER_SELECT_INPUTS := 16#D3,     
	STEP_FILTER_FREQ := 16#06,     //Freq
	ANALOG_DEADBAND := 16#D2,     //0.001 V
	ALARM_RESET_INPUT := 16#46,     //Function ('1'..'3') I/O Point
	ALARM_OUTPUT := 16#47,     //Function ('1'..'3') I/O Point
	ANALOG_SCALING := 16#D1,     
	DEFINE_LIMITS := 16#42,     //1..3
	SET_OUTPUT := 16#8B,     //I/O Point Condition
	WAIT_FOR_INPUT := 16#70,     
	QUEUE_LOAD_AND_EXECUTE := 16#78,     //1..12
	WAIT_TIME := 16#6F,     //0.01 sec
	STOP_MOVE_KILL_BUFFER := 16#E1,    
	STOP_MOVE_KILL_BUFFER_NORMAL_DECEL := 16#E2,
	STOP_MOVE := 16#B5  // Might work, might not     
);
END_TYPE

// Types/StepServoFaultsType
TYPE StepServoFaultsType :
STRUCT
	positionLimit : FB_Fault(name := 'Motor exceeded position limit - following error');        // Motor exceeded position limit - following error
	CCWLimit : FB_Fault(name := 'Counter-Clockwise Limit Reached'); // Counter-Clockwise Limit Reached
	CWLimit : FB_Fault(name := 'Clockwise Limit Reached');		// Clockwise Limit Reached
    overTemp : FB_Fault(name := 'Motor Over Temperature Limit');      // Motor Over Temperature Limit
    internalVoltage : FB_Fault(name := 'Internal Voltage Fault');      // Internal Voltage Fault
    overVoltage    : FB_Fault(name := 'Overvoltage Fault');      // Overvoltage Fault
	underVoltage : FB_Fault(name := 'Undervoltage Fault'); 	// Undervoltage Fault
    overCurrent : FB_Fault(name := 'Motor Overcurrent');      // Motor Overcurrent
    openMotorWinding : FB_Fault(name := 'Motor Detected Open Winding');      // Motor Detected Open Winding
    badEncoder : FB_Fault(name := 'Motor Encoder Failure');      // Motor Encoder Failure
	noMove : FB_Fault(name := 'No Move After Command');
	currentFoldback : FB_Fault(name := 'Current Foldback');
	commFail : FB_Fault(name := 'Drive to Controller Communication Failure');	// Drive to Controller Communication Failure
	notHomed : FB_Fault(name := 'Drive is not homed'); // Drive is not homed
END_STRUCT
END_TYPE

// FBs/DelayDwellFB/DELAY_DWELL_STATES
{attribute 'qualified_only'}
{attribute 'strict'}
TYPE DELAY_DWELL_STATES :
(
	Idle := 0,
	Delay := 1,
	Dwell := 2,
	ResettingDwell := 10,
	ManualOn := 20,
	ManualOff := 21
);
END_TYPE

// FBs/FunctionalAreas/StateMachine
TYPE StateMachine :
STRUCT
	head : HEAD_STATES;
	sb : Substate; // Substate 'Sub' cant be used
END_STRUCT
END_TYPE

// FBs/FunctionalAreas/Substate
TYPE Substate :
STRUCT
	sealSeparate : SEAL_SEPARATE_STATES;
    releaseFeed : RELEASE_FEED_STATES;
    openBag : BAG_OPEN_ASSIST_STATES;
	finishCycle : FINISH_CYCLE_STATES;
	automation : AUTOMATION_STATES;
	printOutOfCycle : PRINT_OUT_OF_CYCLE_STATES;
END_STRUCT
END_TYPE

// Function Blocks/Diagnostics/stateRateKeyPair
TYPE stateRateKeyPair :
STRUCT
	stateID:INT:=-1;
	stateName:STRING:='';
	cycleArray:ARRAY[0..20] OF TIME;
END_STRUCT
END_TYPE

// Function Blocks/SolenoidValves/ValveSelection
{attribute 'qualified_only'}
{attribute 'strict'}
TYPE ValveSelection :
(
	PressureBar := 0,
	SealBar := 1,
	HPA_LPA := 2,
	LoadPlate := 3,
	BagOpenFingers := 4,
	PrintHead := 5,
	Vacuum := 6,
	SealFlattenersVerticalAxis := 7,
	LoadShelf := 8,
	Blank := 999
);
END_TYPE

// Motion/Base/AXIS_STATE
{attribute 'qualified_only'}
{attribute 'strict'}
TYPE AXIS_STATE :
(
	AS_PowerOff := 0,
	AS_ErrorStop := 1,
	AS_Stopping := 2,
	AS_Standstill := 3,
	AS_DiscreteMotion := 4,
	AS_ContinuousMotion := 5,
	AS_Homing := 7
);
END_TYPE

// Motion/Base/MC_ERROR
{attribute 'qualified_only'}
{attribute 'strict'}
TYPE MC_ERROR :
(
	NO_ERROR := 0,
	DRIVE_COMM_FAIL := 1,
	DRIVE_FAULTED := 2,
	AXIS_NOT_READY := 3,
	AXIS_ERROR_DURING_COMMAND := 4,
	R_NO_ERROR_TO_RESET := 5
);
END_TYPE

// Motion/Base/OP_MODE
{attribute 'qualified_only'}
{attribute 'strict'}
TYPE OP_MODE :
(
	OP_UNKNOWN := 0, // The Operating Mode is Unknown
	OP_HOMING := 1, // Homing Mode
	OP_VELOCITY := 2, // Velocity Mode
	OP_POSITION := 3 // Position Mode
);
END_TYPE

// Testing/FB_CrevisSerial/eSerialStates
{attribute 'qualified_only'}
{attribute 'strict'}
TYPE eSerialStates :
(
	Idle := 0,
	ClearReadBuffer := 1,
	writeOutBuffer := 10,
	writingOutBuffer := 11,
	waitForResponse := 12,
	getResponse := 13,
	gettingResponse := 14, 
	Done := 100
);
END_TYPE

// Types/Factoy Selection/AuxiliaryIOSelection
{attribute 'qualified_only'}
{attribute 'strict'}
TYPE AuxiliaryIOSelection :
(
	NotInstalled := 0,
	AuxIOStandard := 1
);
END_TYPE

// Types/Factoy Selection/BagDeflatorSelection
{attribute 'qualified_only'}
{attribute 'strict'}
TYPE BagDeflatorSelection :
(
	NotInstalled := 0,
	IBDStandard := 1,
	IBDWithHingedPlate := 2,
	MotorizedIBD := 3
);
END_TYPE

// Types/Factoy Selection/BagOpenFingersSelection
{attribute 'qualified_only'}
{attribute 'strict'}
TYPE BagOpenFingersSelection :
(
	NotInstalled := 0,
	PneumaticWithBagOpenSensors := 1
);
END_TYPE

// Types/Factoy Selection/BCVSelection
{attribute 'qualified_only'}
{attribute 'strict'}
TYPE BCVSelection :
(
	NotInstalled := 0,
	VisionBased := 1,
	LaserScanner := 2,
	TwoDimensional := 3
);
END_TYPE

// Types/Factoy Selection/ExteralConveyorSelection
{attribute 'qualified_only'}
{attribute 'strict'}
TYPE ExteralConveyorSelection :
(
	NotInstalled := 0,
	ExternalExitConveyor := 1
);
END_TYPE

// Types/Factoy Selection/FeedToSealSelection
{attribute 'qualified_only'}
{attribute 'strict'}
TYPE FeedToSealSelection :
(
	NotInstalled := 0,
	FeedToSealStandard := 1
);
END_TYPE

// Types/Factoy Selection/FillerSelection
{attribute 'qualified_only'}
{attribute 'strict'}
TYPE FillerSelection :
(
	NotInstalled := 0,
	StandardFiller := 1,
	EZFeed := 2
);
END_TYPE

// Types/Factoy Selection/FunnelSelection
{attribute 'qualified_only'}
{attribute 'strict'}
TYPE FunnelSelection :
(
	NotInstalled := 0,
	FunnelWithSensors := 1,
	FunnelWithoutSensors := 2,
	TwoStageFunnelWithSensors := 3,
	BagLoadingTray := 4
);
END_TYPE

// Types/Factoy Selection/IntegratedConveyorSelection
{attribute 'qualified_only'}
{attribute 'strict'}
TYPE IntegratedConveyorSelection :
(
	NotInstalled := 0,
	RearExit := 1
);
END_TYPE

// Types/Factoy Selection/LabelPrinterSelection
{attribute 'qualified_only'}
{attribute 'strict'}
TYPE LabelPrinterSelection :
(
	NotInstalled := 0,
	ZebraPrinter203DPI := 1,
	ZebraPrinter300DPI := 2,
	PrintAndApply203DPI := 3,
	PrintAndApply300DPI := 4
);
END_TYPE

// Types/Factoy Selection/LightCurtainsSelection
{attribute 'qualified_only'}
{attribute 'strict'}
TYPE LightCurtainsSelection :
(
	NotInstalled := 0,
	LoadingAreaLightCurtains := 1
);
END_TYPE

// Types/Factoy Selection/ModelSelection
{attribute 'qualified_only'}
{attribute 'strict'}
TYPE ModelSelection :
(
	Pro18_1174 := 0,
	Pro24_1182 := 1,
	Pro18_1183 := 2,
	Pro24_1196 := 3
);
END_TYPE

// Types/Factoy Selection/PackageEjectionSelection
{attribute 'qualified_only'}
{attribute 'strict'}
TYPE PackageEjectionSelection :
(
	NotInstalled := 0,
	RearRetractingLoadPlate := 1,
	LabelSideUp := 2,
	RearRetractWithRetractShelf := 3
);
END_TYPE

// Types/Factoy Selection/PalmButtonSelection
{attribute 'qualified_only'}
{attribute 'strict'}
TYPE PalmButtonSelection :
(
	NotInstalled := 0,
	SinglePalmButton := 1,
	DualPalmButton := 2,
	LightedPalmButton := 3,
	LightedPalmButtonAdvanced := 4,
	DualLightedPalmButtonAdvanced := 5
);
END_TYPE

// Types/Factoy Selection/SealAreaOptionSelectionEnum
{attribute 'qualified_only'}

TYPE SealAreaOptionSelectionEnum :
(
	NotInstalled 				  := 0,
	MotorizedSealFlatteners 	  := 1,
	PerfBreaker 				  := 2,
	SealFlattenersWithPerfBreaker := 3
);
END_TYPE

// Types/HMI Types/PressureBarHMI
TYPE PressureBarHMI :
STRUCT
	openDelay : UINT;
	closeDelay : UINT;
	passthroughSetting : REAL;
	lowPressureAirDwell : REAL;
	highPressureAirDwell : REAL;
END_STRUCT
END_TYPE

// Types/States/BAG_DELIVERY_MOVE_STATES
{attribute 'strict'}
{attribute 'qualified_only'}
TYPE BAG_DELIVERY_MOVE_STATES :
(
	Idle := 0,
	SetToPointToPointMode := 10,
	AckPointToPointMode := 1,
	WaitAfterSettingOutputOff := 11,
	MoveMotor := 12,
	WaitAfterMovingMotor := 13,
	SetToTorqueMode := 14,
	AckTorqueMode := 2,
	WaitAfterSettingOutputOn := 15,
	Fault := 99
);
END_TYPE

// Types/States/BCR_STATES
{attribute 'strict'}
{attribute 'qualified_only'}
TYPE BCR_STATES :
(
	Idle := 0,
	WaitForOffset := 10,
	TriggerReader := 11,
	WaitingForResult := 12,
	Resetting := 13
);
END_TYPE

// Types/States/EZFEED_STATES_1
{attribute 'strict'}
{attribute 'qualified_only'}
TYPE EZFEED_STATES_1 :
(
	Idle := 0,
	IndexingFlightMode := 10,
	IndexingPartsMode := 11,
	IndexDwell := 12,
	WaitForBaggerCycleComplete := 13,
	PartsStarved := 20,
	Fault := 99
);
END_TYPE

// Types/States/FILLER_STATES
{attribute 'strict'}
{attribute 'qualified_only'}
TYPE FILLER_STATES :
(
	Idle := 0,
	CycleBaggerToActiveFiller := 10,
	WaitingForFiller := 11,
	Dropping := 13,
	BaggerCycling := 14,
	Fault := 99
);
END_TYPE

// Types/States/GRABBER_STATES
{attribute 'strict'}
{attribute 'qualified_only'}
TYPE GRABBER_STATES :
(
	Idle := 0,
	OpenGrippers := 10,
	MoveGrippersOut := 11,
	MovingGrippersOut := 12,
	GrippersMovedOut :=13,
	MoveGantryUp := 20,
	MovingGantryUp := 21,
	GantryMovedUp := 22,
	MoveGrippersIn := 30,
	MovingGrippersIn := 31,
	GrippersMovedIn := 32,
	Ready := 40,
	GrabBag := 50,
	MoveGantryDown := 60,
	MovingGantryDown := 61,
	GantryMovedDown := 62,
	ReleaseBag := 70,
	Fault := 99
);
END_TYPE

// Types/States/JAW_HOMING_STATES
{attribute 'strict'}
{attribute 'qualified_only'}
TYPE JAW_HOMING_STATES :
(
    Idle := 0,
    MoveForwardFromSensor := 10,
    MovingForwardFromSensor := 11,
	ClearToHome := 12,
    StartHoming := 13,
    Homing := 14,
    HomeComplete := 15,
	MoveToTwoInches := 16, 
	MovingToTwoInches := 17,
	SetLimits := 18
	
);
END_TYPE

// Types/States/JOG_STATES
{attribute 'strict'}
{attribute 'qualified_only'}
TYPE JOG_STATES :
(
    Idle := 0,
    JogForwardDIRequest := 10,
    JogForwardOpcodeRequest := 11,
    JoggingForward := 12,
    JogReverseDIRequest := 20,
    JogReverseOpcodeRequest := 21,
    JoggingReverse := 22,
    StoppingJog := 30
);
END_TYPE

// Types/States/MOVE_MODBUS_COMMAND_STATES
{attribute 'strict'}
{attribute 'qualified_only'}
TYPE MOVE_MODBUS_COMMAND_STATES :
(
	Idle := 0,
	SendParameters := 10,
	WaitAfterParametersSent := 11,
	SendOpcode := 20,
	WaitAfterOpcodeSent := 21,
	SendCommand := 31,
	WaitAfterCommandSent := 32,
	SendClearCommand := 40,
	WaitAfterSendClearCommand := 41,
	Fault := 99
);
END_TYPE

// Types/States/OPCODE_MODBUS_COMMAND_STATES
{attribute 'strict'}
{attribute 'qualified_only'}
TYPE OPCODE_MODBUS_COMMAND_STATES :
(
	Idle := 0,
	SendOpcodeAndParameters := 10,
	WaitAfterOpcodeAndParametersSent := 11,
	Fault := 99
);
END_TYPE

// Types/States/PASSTHROUGH_SERVO_STATES
{attribute 'strict'}
{attribute 'qualified_only'}
TYPE PASSTHROUGH_SERVO_STATES :
(
	Idle := 0,
	HomingRequired := 1,
	StartHoming := 10,
	Homing := 11,
	HomeComplete := 12,
	MovePassthroughOut := 20,
	MovingPassthroughOut := 21,
	PassthroughMovedOut := 22,
	ExtendHighPressureOnceMovedOut := 23,
	ExhaustPressureBarOnceMovedOut := 24,
	MovePassthroughIn := 30,
	MovingPassthroughIn := 31,
	PassthroughMovedIn := 32,
	Ready := 40,
	Fault := 99
);
END_TYPE

// Types/States/SOLENOID_TEST_STATES
{attribute 'qualified_only'}
{attribute 'strict'}
TYPE SOLENOID_TEST_STATES :
(
	Extended := 0,
	Retracted := 1,
	FailedToExtend := 2,
	Idle := 3
);
END_TYPE

// Types/States/VACUUM_PICKER_STATES
{attribute 'strict'}
{attribute 'qualified_only'}
TYPE VACUUM_PICKER_STATES :
(
	Idle := 0,
	Home := 1, 
	Homing := 2, 
	Homed := 3,
	XAxisMoveIn := 10,
	XAxisMovingIn := 11, 
	XaxisMovedIn := 12,
	VacuumTurnOn := 20,
	VacuumHeadDown := 30,
	YAxisMoveDown := 31,
	VacuumHeadAndYAxisMovingDown := 32,
	VacuumHeadAndYAxisMovedDown := 33,
	VacuumTurnOff := 40,
	ConveyorTurnOn := 50,
	ConveyorMoving := 51,
	ConveyorDone := 52,

	Fault := 99,
	Ready := 100,
	Manual := 101
);
END_TYPE

// Globals
{attribute 'qualified_only'}
VAR_GLOBAL
    firstScan : BOOL; //First Scan Bit
    pressureBarServoCommsType : MODBUS_COMM_TYPE;  //Comm path to Pressure Bar Servo - 0 = TCP, 1 = RTU
    STEPS_PER_INCH : INT;  //Steps Per Inch for Pressure Bar Servos
    maximumPassthough : REAL := 9.0;
	SystemLog : FB_InternalLogger;
	jawMovingIn : BOOL;
	passthroughChangedFromJog : BOOL;
	machinePowerOK : BOOL;
END_VAR

VAR_GLOBAL CONSTANT
    STEPS_PER_INCH_SEAL_FLATTENER_HORIZONTAL_AXIS_MOTOR  : INT := 2500;
    STEPS_PER_INCH_SEAL_FLATTENER_VERTICAL_AXIS_MOTOR : INT := 2890;        //Steps per inch for NEMA 17 seal flattener finger motor
    STEPS_PER_INCH_BIG_MOTOR : INT := 21872;        //Steps per inch for NEMA 17 motor
    STEPS_PER_INCH_SMALL_MOTOR : INT := 19600;        //Steps per inch for NEMA 11 motor
    STEPS_PER_INCH_SHOW_MOTOR : INT := 18900;        //Steps per inch for NEMA 11 motor
    STEPS_PER_INCH_PRINTER : INT := 4498;            //Steps per inch for printer step servo
    STEPS_PER_INCH_20_DEGREE_BAG_DELIVERY : INT := 5093; // Steps per inch for 20 degree bag delivery motors
	STEPS_PER_INCH_PRO24_BAG_DELIVERY : INT := 4428; // Steps per inch for 20 degree bag delivery motors
	STEPS_PER_INCH_ADJUSTABLE_PASSTHROUGH : INT := 3030;  // Steps per inch for the Adjustable Passthrough motor
	STEPS_PER_INCH_TFBelt : INT := 3030;  // Steps per inch for the Adjustable Passthrough motor
	STEPS_PER_INCH_TFLS : INT := 10000;  // Steps per inch for the Adjustable Passthrough motor
	STEPS_PER_INCH_PRO24_BD : INT := 5914; 
	VELOCITY_IPS_MULTIPLIER_ELECTRIC_4BD: REAL := 70;
	STEPS_PER_INCH_PRO24_PAPER_FRONT : INT:=10030;
	STEPS_PER_INCH_PRO24_PAPER_REAR : INT:=10010;
    VELOCITY_IPS_MULTIPLIER_ELECTRIC: REAL := 53;
	VELOCITY_IPS_MULTIPLIER_PNEUMATIC: REAL := 61;
    PASSTHROUGH_ZERO_OFFSET : REAL := 2;            //Zero offset for passthough (minimum passthough)
    MAX_BAG_WIDTH : REAL := 18;                //Passthrough setting
	AMP_MOTOR_RPI : INT := 10;
	MAX_LOGGED_ITEMS : UINT := 500;	// Max items to be logged
	MAXIMUM_PASSTHROUGH_PRO18 : REAL := 9.0;
	MAXIMUM_PASSTHROUGH_PRO24 : REAL := 12.0;
END_VAR

VAR_GLOBAL
    headCycleCount : DINT;                 // Head Cycle Counts
	headCycleCount2 : DINT;                 // Head Cycle Counts
    bagGrabberCycleCount : DINT;         // Bag Grabber Cycle Counts
    solenoidCycleCount1 : DINT;         // Solenoid Cycle Cycle Counts (first solenoid)
    motorizedSealFlattenersCount : DINT;         // MSF Cycle Counts
    bagOpenFingersCount : DINT;        // Bag Open Finger Cycles
    sealFlattenerFingersCount : DINT;  // Seal Flattener Fingers Cycle Count
    electricPressureBarCount : DINT;    // Electric Pressure bar Cycle count
    sealBarCount : DINT;                 // Seal bar Cycle count
    bagDeliveryCycleCount : DINT;        // Bag Delivery Cycle Count
    printerCycleCounts : DINT;            // Printer Cycle Counts
    bagsMadeCount : DINT;                // Bags Made
    passthroughChangeCount : DINT;        // Passthrough Changes
	passthroughChangeDistance : UDINT;	// Passthrough Distance Changes in .1 Inches
	solenoidCycleCount2 : DINT;     	// Solenoid Cycle Cycle Counts (Strech SX)	
	solenoidFailureCount2 : UDINT;		// Solenoid Failure Count (Strech SX)
	pickAndPlaceCycleCount : UDINT;		// Pick and place cycle count
	passthroughChangeCount2 : DINT;        // Passthrough Changes
	passthroughChangeDistance2 : UDINT;	// Passthrough Distance Changes in .1 Inches
	bagFailedToGrabBothFingersCount : UDINT; // Both Fingers failed to grab bag
	bagFailedToGrabRightFingerCount : UDINT; // Right Bag Open Finger Failed to Grab Bag
	bagFailedToGrabLeftFingerCount : UDINT; // Left Bag Open Finger Failed to Grab Bag
	successfulBagOpenCount : UDINT;			// Successful Bag Open Count
	rejectedBagCount : UDINT;				// Rejected bag count 
    dryCycleCount  :UDINT;                   // Dry cycle count
	lastPrinterDelta : TIME := T#100MS;
	factoryTestComplete : BOOL;		// 1000 bags test done
END_VAR

// HMIData
// All HMI data is presented through this GVL
{attribute 'qualified_only'}
{attribute 'global_init_slot' := '50001'}
VAR_GLOBAL // PERSISTENT RETAIN
	initiateCycle : BOOL;  // Initiate Cycle Pushbutton
	ackAllFaults : BOOL; // Acknowledge All Faults from HMI
	makeReady : BOOL;
	jobLoaded : BOOL;
    stopMachine : BOOL;
	version : STRING;
	inCycle : BOOL;
	batchEnable : BOOL;
	autoEnable : BOOL;
	autoModeDwell : REAL;
	batchSetting : UDINT := 10;
	batchCount : UDINT;
	batchReset : BOOL;
	headCycleCount : UDINT;
	pressureBarOpenDelay : REAL;
	pressureBarCloseDelay : REAL;
	pressureBarPositionBuffer: DINT := 50;
	passthroughSetting : REAL := 5.0;
	passthroughOffset : REAL;
	passthroughPosition : REAL;
	lpaDwell : REAL;
	hpaDwell : REAL;
	sealBarDwell : REAL;
	sealBarTemperatureSetting : UDINT;
	sealBarTemperature : UDINT;
	sealFlattenersPosition : REAL;
	bagSkirtLength : REAL := 1.35;
	bagLength : REAL := 23.5;
	bagWidth : REAL := 17.5;
	bagThickness : REAL := 2.5;
	bagTensionSetting : REAL := 0.6;  // Bag takeup tension setting in amps
	bagDropTime : REAL;
	bagForwardSpeed : UDINT := 55;
	bagReverseSpeed : UDINT := 3;
	bagEdgePhotoeyeCovered : BOOL;
	printSpeed : UDINT := 6;
	printLength : REAL := 8.0;
	printOffset : REAL := 2.0;
	printOutOfCycleEnable : BOOL;
	printerCycleSelection : PrinterCycleSelection;
	fillerCountSetting : UDINT;
	fillerCurrentCount : UDINT;
	fillerDropTime : REAL;
	fillerEnable : BOOL; 
	loadPlateInUse : BOOL;
	loadPlateDelay : REAL;
	loadPlateDwell : REAL;
	rearLoadPlateShakerDelay : REAL;
	rearLoadPlateShakerDwell : REAL;
	rearLoadPlateShakerOnDuration : REAL;
	rearLoadPlateShakerOffDuration : REAL;
	rearloadPlateShakerStart : SHAKER_START_SELECTION;
	frontLoadPlateShakerDelay : REAL;
	frontLoadPlateShakerDwell : REAL;
	frontLoadPlateShakerOnDuration : REAL;
	frontLoadPlateShakerOffDuration : REAL;
	frontloadPlateShakerStart : SHAKER_START_SELECTION;
	loadShelfDelay : REAL := 0.1;
	loadShelfDwell : REAL := 1.5;
	loadShelfShakerDelay : REAL;
	loadShelfShakerDwell : REAL;
	loadShelfShakerOnDuration : REAL;
	loadShelfShakerOffDuration : REAL;
	loadShelfShakerStart : SHAKER_START_SELECTION;
	exitConveyorDwell : REAL;
	vacuumDwell : REAL := 0.25;
	IBDDeflateDwellTime  : REAL := 0.75;
	IBDClosePosition : REAL := 0;
	IBDPackageEjectAssistDelayTime : REAL;
	IBDPackageEjectAssistDwellTime : REAL := 0.8;
	funnelInUse : BOOL;								// Funnel Enable/Disable
	funnelOpenDelay : REAL := 0.25;					// Funnel Open Delay after pressure bar open
	funnelOpeningTime : REAL := 0.5;				// For funnel w/o sensors only : Time required to consider funnel open after command to open
	funnelClosingTime : REAL := 0.5;				// For funnel w/o sensors only : Time required to consider funnel closed after command to close
	stagingFunnelOpenDelay : REAL := 0.25;					// Funnel Open Delay after pressure bar open
	stagingFunnelOpeningTime : REAL := 0.5;				// For funnel w/o sensors only : Time required to consider funnel open after command to open
	stagingFunnelClosingTime : REAL := 0.5;				// For funnel w/o sensors only : Time required to consider funnel closed after command to close
	externalExitConveyorDwell : REAL;
	barcodeGoodReadCount : UDINT;
	barcodeBadReadCount : UDINT;
	barcodeBadReadFaultSetting : UDINT;
	barcodeStartPosition : REAL;
	barcodeScanDistance : REAL := 1.0;
	barcodeVerifierInUse : BOOL;
	barcodeLastReadString : STRING[100];
	barcodeScanDuration : REAL := 2.5;                // Used when 2D barcode is selected
	lastCycleTime : REAL;
	averageCycleTime : REAL;
	resetAverageCycleTime : BOOL;
	bagOpenRetrySetting : INT := 3;
	bagOpenRetryCount : INT;
	bagOpenFeedNewBagSetting : INT := 1;
	bagOpenFeedNewBagCount : INT;
	bagOpenEnable : BOOL := TRUE;
	currentJobID : INT;
	separateBeforeSeal : BOOL;
	activateDemoMode : BOOL;
	printerInUse : BOOL;
	printerInstalled : BOOL;
	lpaDuringBagFeedEnable : BOOL := TRUE;
	lpaBagEjectAssistEnable : BOOL := TRUE;
	infeedConveyorRunningMode : BOOL;  			//0 = Indexing, 1 = Continuous
	infeedConveyorCountingMode : BOOL;			// 0 = Flight, 1 = Parts
	infeedIndexDwellTimer : REAL := 0.25;
	infeedFlightCountTarget : DINT := 5;
	infeedFlightCountActual : DINT;
	infeedPartsCountTarget : DINT := 10;
	infeedPartsCountActual : DINT;
	infeedEmptyPartsSetting : DINT := 10;
	infeedEmptyPartsActual : DINT;
	printAndApplyTriggerDelayWithLOTAR : REAL := 0;
	printAndApplyTriggerDelayWithoutLOTAR : REAL := 0;
	printAndApplyConveyorDwell : REAL := 5.0;
	printAndApplyProductToPhotoeyeTime : REAL := 4.0;
	printAndApplyWaitForLabelTimeout : REAL := 15.0;
	enableDryCycle : BOOL;          // Enable dry cycle
	baggerNeedsClearing : BOOL;
	baggerClearedAck : BOOL;
	calculatedCyclesPerMinute : REAL;
	sealFlattenersInUse : BOOL := TRUE;
	collisonDetectionDwell : REAL := 1.0;
	packageAtExitRunoffDwell : REAL := 1.0;
	IBDOffset : REAL := 3.0;
	pressureBarBagFeedPosition : REAL := 2.0;
	pressureBarInPosition : REAL := 0;
	feedToSealSetpoint : REAL := 0.0;
	feedToSealInUse : BOOL := FALSE;
	reverseConveyor : BOOL;
	enablePerfBreaker : BOOL;
	enablePaperBagger : BOOL;
	mailerMaterial : MAILER_MATERIAL;
	labelsQueuedUpFaultEnable : BOOL := FALSE;
	remoteCommsHeartbeatEnable : BOOL;
	auxIOSource : AuxIOSource := (Physical := TRUE);
	movePbarByHandWhileLoadingEnable : BOOL;
	paperTensionSetting : DINT := 60;
	polyTensionSetting : DINT := 50;
	
	(*Service Stuff*)
	lpaServiceOn : BOOL;
	lpaServiceOff : BOOL;
	lpaServicePulse : BOOL;
	hpaServiceOn :BOOL;
	hpaServicePulse : BOOL;
	exitConveyorStart : BOOL;
	exitConveyorStop : BOOL;
	exitConveyorJog : BOOL;
	exitConveyorJogTime : TIME;
	exitConveyorStartDwell : BOOL;
	pressureBarService : ServiceCommands;
	loadPlateService : ServiceCommands;
	forwardLoadPlateService : ServiceCommands;
	rearLoadPlateService : ServiceCommands;
	loadShelfService : ServiceCommands;
	IBDService : ServiceCommands;
	accumulatingFunnel : ServiceCommands;
	funnelService : ServiceCommands;
	baggerHeadService : ServiceCommands;
	perfBreakerService: ServiceCommands;
	jogBagForward : BOOL;
	jogBagReverse : BOOL;
	jogPassthroughForward : BOOL;
	jogPassthroughReverse : BOOL;
	sealBarServiceCycle : BOOL;
	sealBarServiceRetract : BOOL;
	sealBarServiceExtend : BOOL;
	bagOpenFingersServiceGrab : BOOL;
	bagOpenFingersServiceRelease : BOOL;
	sealFlattenersServiceRaise : BOOL;
	sealFlattenersServiceLower : BOOL;
	sealFlattenersServiceJogIn : BOOL;
	sealFlattenersServiceJogOut : BOOL;
	sealFlattenersManualPositionSetting : REAL;
	sealFlattenersMoveToManualPos : BOOL;
	passthroughManualPositionSetting : REAL;
	passthroughMoveToManualPos : BOOL;
	factoryTestMode : BOOL;
	vacuumServiceOn : BOOL;
	vacuumServiceOff : BOOL;
	printHeadServiceRaise : BOOL;
	printHeadServiceLower : BOOL;
	externalExitConveyorStart : BOOL;
	externalExitConveyorStop : BOOL;
	externalExitConveyorJog : BOOL;
	externalExitConveyorStartDwell : BOOL;
	triggerBarcodeReaderService : BOOL;
	
	(*Factoy Config*)
	bofSelection : BagOpenFingersSelection := BagOpenFingersSelection.PneumaticWithBagOpenSensors;
	sealAreaOptionSelection : SealAreaOptionSelectionEnum := SealAreaOptionSelectionEnum.MotorizedSealFlatteners;
	printerSelection : LabelPrinterSelection := LabelPrinterSelection.ZebraPrinter203DPI;
	integratedExitConveyorSelection : IntegratedConveyorSelection := IntegratedConveyorSelection.RearExit;
	externalExitConveyorSelection : ExteralConveyorSelection := ExteralConveyorSelection.NotInstalled;
	feedToSealBagSelection : FeedToSealSelection := FeedToSealSelection.NotInstalled;
	packageEjectSelection : PackageEjectionSelection := PackageEjectionSelection.RearRetractingLoadPlate;
	packageEjectDisabledPosition : PackageEjectionDisabledPosition := PackageEjectionDisabledPosition.LoadingPosition;
	independentBagDeflatorSelection : BagDeflatorSelection := BagDeflatorSelection.NotInstalled;
	cycleStartButtonSelection : PalmButtonSelection := PalmButtonSelection.DualPalmButton;
	barcodeVerifierSelection : BCVSelection := BCVSelection.NotInstalled;
	lightCurtainSelection : LightCurtainsSelection := LightCurtainsSelection.NotInstalled;
	baggerModelSelection : ModelSelection;
	baggerProfileSelection : BaggerProfile := BaggerProfile.Standard;
	auxIOConfig : AuxIOConfiguration;
	fillerFactorySelection : FillerSelection;
	funnelFactorySelection : FunnelSelection;
	murrIOConfigVersion : CONFIG_VERSIONS := CONFIG_VERSIONS.V_1_4;
	printerConfigVersion : CONFIG_VERSIONS := CONFIG_VERSIONS.V_1_2;
	frontFilmFeedMotorConfigVersion : CONFIG_VERSIONS := CONFIG_VERSIONS.V_1_0;
	rearUnwindMotorConfigVersion : CONFIG_VERSIONS := CONFIG_VERSIONS.V_1_3;
	sealFlattenerMotorConfigVersion : CONFIG_VERSIONS := CONFIG_VERSIONS.V_1_0;
    shakerInstalled : BOOL;
	
	(*Warnings*)
	printerRibbonLow : Warning;
	printerNotReady : Warning;
	waitingForPrinter : Warning;
	sealBarNotAtTemperature : Warning;
	recoveryModeActive : Warning;
	jobLoadRequired : Warning;
	baggerNotReady : Warning;
	demoModeIsActive : Warning;
	factoryTestModeActive : Warning;
	machineNotTested : Warning;
	packageEjectGuardRemoved : Warning;
	bagLevelLow : Warning;
	fillerModeCycleStartOnly : Warning;
	baggerInhibited : Warning;
	packageBlockingTrunkline : Warning;
	infeedConveyorOutOfParts : Warning;
	mayCycleUnexpectedly : Warning;
	printAndApplyRibbonLow : Warning;
	printAndApplyWaitingForApply : Warning;
	printAndApplyWaitingForLabel : Warning;
	printAndApplyBypassed : Warning;
	dryCycleActive : Warning;
	lightCurtainsBlocked : Warning;
	batchCountDone : Warning;
	remoteCommsHeartbeatLost: Warning;
	stagingFunnelAndPerfBreakerEnabled : Warning;
	
	(*Faults*)
	(*Misc*)
	pressureBarState : STRING;
    heartbeat : UDINT;
    (*Counters*)
    baggerCycles : FB_CycleCounter;
	bagOpenFingerCycles : FB_CycleCounter;
	bagsMade : FB_CycleCounter;
	sealBarCycles : FB_CycleCounter;
	pressureBarCycles : FB_CycleCounter;
	passthroughChanges : FB_CycleCounter;
	loadPlateCycles : FB_CycleCounter;
	printerCycles : FB_CycleCounter;
	motorizedSealFlattenerCycles : FB_CycleCounter;
	bagOpenRetryTotal : FB_CycleCounter;
	bagsRejectedTotal : FB_CycleCounter;
	resettableBagsMade : FB_CycleCounter;
	
	(*Predictive Maint.*)
	airFilterClean : FB_PredictiveMaint := (target := 30000, count := 0, name := 'Clean Air Filter');
	driveRollerClean : FB_PredictiveMaint := (target := 20000, count := 0, name := 'Clean Drive Rollers', units := 'Inches of Bag');
	printHeadClean : FB_PredictiveMaint := (target := 10000, count := 0, name := 'Clean Print Head', units := 'Printer Cycles');
	pressureBarGuideShaftGuides : FB_PredictiveMaint := (target := 0, count := 127888, name := 'Replace Guide Shafts');
	
	pressureBarLeak : FB_CylinderLeak := (maximumStrokeTime := 5.0, name := 'Pressure Bar Stroke', units := 'Seconds');
	loadPlateLeak : FB_CylinderLeak := (maximumStrokeTime := 2.0, name := 'Load Plate Stroke', units := 'Seconds');
	
	msfHorizontalMotorTemp : FB_DriveTemp := (maxTemp := 60.0, name := 'MSF Motor Temp.', units := 'deg C');
	bagDeliveryMotorTemp : FB_DriveTemp := (maxTemp := 60.0, name := 'Bag Delivery Motor Temp.', units := 'deg C');
	passthroughMotorTemp : FB_DriveTemp := (maxTemp := 60.0, name := 'Passthrough Motor Temp.', units := 'deg C');
	
	(*Info*)
	faultActive : BOOL;
	

END_VAR

VAR_GLOBAL CONSTANT
	murrIOConfigVersionMax : CONFIG_VERSIONS := CONFIG_VERSIONS.V_1_5;
	printerConfigVersionMax : CONFIG_VERSIONS := CONFIG_VERSIONS.V_1_2;
	frontFilmFeedMotorConfigVersionMax : CONFIG_VERSIONS := CONFIG_VERSIONS.V_1_0;
	rearUnwindMotorConfigVersionMax : CONFIG_VERSIONS := CONFIG_VERSIONS.V_1_3;
	sealFlattenerMotorConfigVersionMax : CONFIG_VERSIONS := CONFIG_VERSIONS.V_1_0;
END_VAR

